// TIA Portal project "andres-c程序测试" (V14)

(* hardware
DEVICE "S7-1200 station_1"  S7-1200 Station
   slot 0: "Rack_0"  Rack  V1.0
   slot 1: "PLC_14工位_1200"  CPU 1215C DC/DC/DC  6ES7 215-1AG40-0XB0  V4.2
DEVICE "ET 200SP station_2"  ET 200SP-Station
   slot 0: "机架_0"  6ES5 710-8MAx1
   slot 0: "IO device_2"  IM155-6 PN ST  6ES7 155-6AU00-0BN0  V3.3
   slot 1: "DI 16x24VDC ST_1"  DI 16x24VDC ST  6ES7 131-6BH00-0BA0  V1.1
      slot 1: "DI 16x24VDC ST_1"  DI 16x24VDC ST
   slot 2: "DI 16x24VDC ST_2"  DI 16x24VDC ST  6ES7 131-6BH00-0BA0  V1.1
      slot 1: "DI 16x24VDC ST_2"  DI 16x24VDC ST
   slot 3: "DI 16x24VDC ST_3"  DI 16x24VDC ST  6ES7 131-6BH00-0BA0  V1.1
      slot 1: "DI 16x24VDC ST_3"  DI 16x24VDC ST
   slot 4: "DI 16x24VDC ST_4"  DI 16x24VDC ST  6ES7 131-6BH00-0BA0  V1.1
      slot 1: "DI 16x24VDC ST_4"  DI 16x24VDC ST
   slot 5: "DI 16x24VDC ST_5"  DI 16x24VDC ST  6ES7 131-6BH00-0BA0  V1.1
      slot 1: "DI 16x24VDC ST_5"  DI 16x24VDC ST
   slot 6: "DI 16x24VDC ST_6"  DI 16x24VDC ST  6ES7 131-6BH00-0BA0  V1.1
      slot 1: "DI 16x24VDC ST_6"  DI 16x24VDC ST
   slot 7: "DI 16x24VDC ST_7"  DI 16x24VDC ST  6ES7 131-6BH00-0BA0  V1.1
      slot 1: "DI 16x24VDC ST_7"  DI 16x24VDC ST
   slot 8: "DI 16x24VDC ST_8"  DI 16x24VDC ST  6ES7 131-6BH00-0BA0  V1.1
      slot 1: "DI 16x24VDC ST_8"  DI 16x24VDC ST
   slot 9: "DI 16x24VDC ST_9"  DI 16x24VDC ST  6ES7 131-6BH00-0BA0  V1.1
      slot 1: "DI 16x24VDC ST_9"  DI 16x24VDC ST
   slot 10: "DI 16x24VDC ST_10"  DI 16x24VDC ST  6ES7 131-6BH00-0BA0  V1.1
      slot 1: "DI 16x24VDC ST_10"  DI 16x24VDC ST
   slot 11: "DQ 16x24VDC/0.5A ST_2"  DQ 16x24VDC/0.5A ST  6ES7 132-6BH00-0BA0  V1.1
      slot 1: "DQ 16x24VDC/0.5A ST_2"  DQ 16x24VDC/0.5A ST
   slot 12: "DQ 16x24VDC/0.5A ST_3"  DQ 16x24VDC/0.5A ST  6ES7 132-6BH00-0BA0  V1.1
      slot 1: "DQ 16x24VDC/0.5A ST_3"  DQ 16x24VDC/0.5A ST
   slot 13: "DQ 16x24VDC/0.5A ST_4"  DQ 16x24VDC/0.5A ST  6ES7 132-6BH00-0BA0  V1.1
      slot 1: "DQ 16x24VDC/0.5A ST_4"  DQ 16x24VDC/0.5A ST
   slot 14: "DQ 16x24VDC/0.5A ST_5"  DQ 16x24VDC/0.5A ST  6ES7 132-6BH00-0BA0  V1.1
      slot 1: "DQ 16x24VDC/0.5A ST_5"  DQ 16x24VDC/0.5A ST
   slot 15: "DQ 16x24VDC/0.5A ST_6"  DQ 16x24VDC/0.5A ST  6ES7 132-6BH00-0BA0  V1.1
      slot 1: "DQ 16x24VDC/0.5A ST_6"  DQ 16x24VDC/0.5A ST
   slot 16: "DQ 16x24VDC/0.5A ST_1"  DQ 16x24VDC/0.5A ST  6ES7 132-6BH00-0BA0  V1.1
      slot 1: "DQ 16x24VDC/0.5A ST_1"  DQ 16x24VDC/0.5A ST
   slot 17: "DQ 16x24VDC/0.5A ST_7"  DQ 16x24VDC/0.5A ST  6ES7 132-6BH00-0BA0  V1.1
      slot 1: "DQ 16x24VDC/0.5A ST_7"  DQ 16x24VDC/0.5A ST
   slot 18: "DQ 16x24VDC/0.5A ST_8"  DQ 16x24VDC/0.5A ST  6ES7 132-6BH00-0BA0  V1.1
      slot 1: "DQ 16x24VDC/0.5A ST_8"  DQ 16x24VDC/0.5A ST
   slot 19: "AQ 4xU/I ST_1"  AQ 4xU/I ST  6ES7 135-6HD00-0BA1  V1.1
      slot 1: "AQ 4xU/I ST_1"  AQ 4xU/I ST
   slot 20: "服务器模块_1"  服务器模块  6ES7 193-6PA00-0AA0  V1.0
      slot 1: "服务器模块_1"  服务器模块
   slot 127: "PROFINET 总线适配器 CU"  PROFINET Interface  6ES7 193-6AR00-0AA0  V0.0
      slot 1: "Port_1"  6ES7 193-6AR00-0AA0  V0.0
      slot 2: "Port_2"  6ES7 193-6AR00-0AA0  V0.0
*)

// ===== PLC "PLC_14工位_1200"  CPU 1215C DC/DC/DC =====

VAR_GLOBAL   // PLC tag table "默认变量表"
   "Tag_1" AT %M0.0 : Bool;
   "初次扫描OB100保持位" AT %M0.1 : Bool;
   "给上位机发送数据" AT %M0.2 : Bool;
   "Tag_4" AT %M0.3 : Bool;
   "1#手动Z轴下降" AT %M10.0 : Bool;
   "14S01" AT %I0.0 : Bool;   // 1#机械手X轴定位接近1
   "14S02" AT %I0.1 : Bool;   // 1#机械手X轴定位接近2
   "14S03" AT %I0.2 : Bool;   // 1#机械手X轴减速接近
   "14L01" AT %I0.3 : Bool;   // 1#机械手X轴机械限位
   "14S04" AT %I0.4 : Bool;   // 1#机械手z轴原点光电
   "14L02" AT %I0.5 : Bool;   // 1#机械手z轴机械限位
   "14S05" AT %I0.6 : Bool;   // 1#机械手W轴原点光电
   "14L03" AT %I0.7 : Bool;   // 1#机械手W轴机械限位
   "14S06" AT %I1.0 : Bool;   // 1#机械手抓取光电
   "14S07" AT %I1.1 : Bool;   // 1#W轴上砖位
   "14S08" AT %I1.2 : Bool;   // 1#W轴停止位
   "14S09" AT %I1.3 : Bool;   // 1#机械手抓取极限光电
   "14P02" AT %I1.4 : Bool;   // 1#机械手负压检测1
   "14P03" AT %I1.5 : Bool;   // 1#机械手负压检测2
   "14P04" AT %I1.6 : Bool;   // 1#机械手负压检测3
   "14P05" AT %I1.7 : Bool;   // 1#机械手负压检测4
   "14S10" AT %I2.0 : Bool;   // 2#机械手X轴定位接近1
   "14S11" AT %I2.1 : Bool;   // 2#机械手X轴定位接近2
   "14S12" AT %I2.2 : Bool;   // 2#机械手X轴减速接近
   "14L04" AT %I2.3 : Bool;   // 2#机械手X轴机械限位
   "14S13" AT %I2.4 : Bool;   // 2#机械手z轴原点光电
   "14L05" AT %I2.5 : Bool;   // 2#机械手z轴机械限位
   "14S14" AT %I2.6 : Bool;   // 2#机械手W轴原点光电
   "14L06" AT %I2.7 : Bool;   // 2#机械手W轴机械限位
   "14S15" AT %I3.0 : Bool;   // 2#机械手抓取光电
   "14S16" AT %I3.1 : Bool;   // 2#机械手W上砖待命位
   "14S17" AT %I3.2 : Bool;   // 2#机械手W轴停止位
   "14S18" AT %I3.3 : Bool;   // 2#机械手抓取极限光电
   "14P06" AT %I3.4 : Bool;   // 2#机械手负压检测1
   "14P07" AT %I3.5 : Bool;   // 2#机械手负压检测2
   "14P08" AT %I3.6 : Bool;   // 2#机械手负压检测3
   "14P09" AT %I3.7 : Bool;   // 2#机械手负压检测4
   "14S19" AT %I4.0 : Bool;   // 3#机械手X轴定位接近1
   "14S20" AT %I4.1 : Bool;   // 3#机械手X轴定位接近2
   "14S21" AT %I4.2 : Bool;   // 3#机械手X轴减速接近
   "14L07" AT %I4.3 : Bool;   // 3#机械手X轴机械限位
   "14S22" AT %I4.4 : Bool;   // 3#机械手z轴原点光电
   "141L08" AT %I4.5 : Bool;   // 3#机械手z轴机械限位
   "14S23" AT %I4.6 : Bool;   // 3#机械手W轴原点光电
   "14L09" AT %I4.7 : Bool;   // 3#机械手W轴机械限位
   "14S24" AT %I5.0 : Bool;   // 3#机械手抓取光电
   "14S25" AT %I5.1 : Bool;   // 3#机械手W上砖待命位
   "14S26" AT %I5.2 : Bool;   // 3#机械手W停止位
   "14S27" AT %I5.3 : Bool;   // 3#机械手抓取极限光电
   "14P10" AT %I5.4 : Bool;   // 3#机械手负压检测1
   "14P11" AT %I5.5 : Bool;   // 3#机械手负压检测2
   "14P12" AT %I5.6 : Bool;   // 3#机械手负压检测3
   "14P13" AT %I5.7 : Bool;   // 3#机械手负压检测4
   "14S28" AT %I6.0 : Bool;   // 4#机械手X轴定位接近1
   "14S29" AT %I6.1 : Bool;   // 4#机械手X轴定位接近2
   "14S30" AT %I6.2 : Bool;   // 4#机械手X轴减速接近
   "14L10" AT %I6.3 : Bool;   // 4#机械手X轴机械限位
   "14S31" AT %I6.4 : Bool;   // 4#机械手z轴原点光电
   "14L11" AT %I6.5 : Bool;   // 4#机械手z轴机械限位
   "14S32" AT %I6.6 : Bool;   // 4#机械手W轴原点光电
   "14L12" AT %I6.7 : Bool;   // 4#机械手W轴机械限位
   "14S33" AT %I7.0 : Bool;   // 4#机械手抓取光电
   "14S34" AT %I7.1 : Bool;   // 4#机械手上砖待命位
   "14S35" AT %I7.2 : Bool;   // 4#机械手W停止位
   "14S36" AT %I7.3 : Bool;   // 4#机械手抓取极限光电
   "14P14" AT %I7.4 : Bool;   // 4#机械手负压检测1
   "14P15" AT %I7.5 : Bool;   // 4#机械手负压检测2
   "14P16" AT %I7.6 : Bool;   // 4#机械手负压检测3
   "14P17" AT %I7.7 : Bool;   // 4#机械手负压检测4
   "14SB1" AT %I8.0 : Bool;   // 一级品分级按钮
   "14SB2" AT %I8.1 : Bool;   // 二级品分级按钮
   "14SB3" AT %I8.2 : Bool;   // 换花色旋钮
   "14S37" AT %I8.3 : Bool;   // 队列光电1
   "14S38" AT %I8.4 : Bool;   // 队列光电2
   "14P01" AT %I8.5 : Bool;   // 设备压力检测
   "14S39" AT %I8.6 : Bool;   // 1#3#库位安全光电
   "14S40" AT %I8.7 : Bool;   // 2#4#库位安全光电
   "14S41" AT %I9.0 : Bool;   // 7#9#库位安全光电
   "14S42" AT %I9.1 : Bool;   // 8#10#库位安全光电
   "14S43" AT %I9.2 : Bool;   // 1#库位栈板检测光电
   "14S44" AT %I9.3 : Bool;   // 2#库位栈板检测光电
   "14S45" AT %I9.4 : Bool;   // 1#库位安全检测光电
   "14S46" AT %I9.5 : Bool;   // 2#库位安全检测光电
   "14SB7" AT %I9.6 : Bool;   // 1#库位按钮
   "14SB8" AT %I9.7 : Bool;   // 2#库位按钮
   "14S47" AT %I10.0 : Bool;   // 3#库位栈板检测光电
   "14S48" AT %I10.1 : Bool;   // 4#库位栈板检测光电
   "14S49" AT %I10.2 : Bool;   // 3#库位安全检测光电
   "14S50" AT %I10.3 : Bool;   // 4#库位安全检测光电
   "14SB9" AT %I10.4 : Bool;   // 3#库位按钮
   "14SB10" AT %I10.5 : Bool;   // 4#库位按钮
   "14S51" AT %I10.6 : Bool;   // 5#库位栈板检测光电
   "14S52" AT %I10.7 : Bool;   // 6#库位栈板检测光电
   "14S53" AT %I11.0 : Bool;   // 5#库位安全检测光电
   "14S54" AT %I11.1 : Bool;   // 6#库位安全检测光电
   "14SB11" AT %I11.2 : Bool;   // 5#库位按钮
   "14SB12" AT %I11.3 : Bool;   // 6#库位按钮
   "14S55" AT %I11.4 : Bool;   // 7#库位栈板检测光电
   "14S56" AT %I11.5 : Bool;   // 8#库位栈板检测光电
   "14S57" AT %I11.6 : Bool;   // 7#库位安全检测光电
   "14S58" AT %I11.7 : Bool;   // 8#库位安全检测光电
   "14SB13" AT %I12.0 : Bool;   // 7#库位按钮
   "14SB14" AT %I12.1 : Bool;   // 8#库位按钮
   "14SB25" AT %I12.2 : Bool;   // 输送线启动按钮
   "14S59" AT %I12.3 : Bool;   // 输送线对中光电
   "14SB26" AT %I12.4 : Bool;   // 输送线停止按钮
   "11S73" AT %I12.5 : Bool;   // 队列光电3
   "11S74" AT %I12.6 : Bool;   // 队列光电4
   "输送线变频器报警" AT %I12.7 : Bool;   // 输送线变频器报警
   "14M01MB" AT %I13.0 : Bool;   // M01变频器报警
   "14M02MB" AT %I13.1 : Bool;   // M02变频器报警
   "14M04MB" AT %I13.2 : Bool;   // M04变频器报警
   "14M05MB" AT %I13.3 : Bool;   // M05变频器报警
   "14M07MB" AT %I13.4 : Bool;   // M07变频器报警
   "14M08MB" AT %I13.5 : Bool;   // M08变频器报警
   "14M10MB" AT %I13.6 : Bool;   // M10变频器报警
   "14M11MB" AT %I13.7 : Bool;   // M11变频器报警
   "14SB15" AT %I14.0 : Bool;   // 主控柜启动按钮
   "14SB16" AT %I14.1 : Bool;   // 主控柜停止按钮
   "14SB17" AT %I14.2 : Bool;   // 主控柜复位按钮
   "14SB18" AT %I14.3 : Bool;   // 主控柜消音按钮
   "14EM" AT %M65.0 : Bool;   // 主控柜急停按钮
   "14SA01" AT %I14.5 : Bool;   // 主控柜启动激活
   "14SA02" AT %I14.6 : Bool;   // 主控柜停止激活
   "14SA03" AT %I14.7 : Bool;   // 主控柜复位激活
   "14M13MB" AT %I15.0 : Bool;   // M13变频器报警
   "14M14MB" AT %I15.1 : Bool;   // M14变频器报警
   "14M03MB" AT %I15.2 : Bool;   // M03伺服控制器报警
   "14M06MB" AT %I15.3 : Bool;   // M06伺服控制器报警
   "14M09MB" AT %I15.4 : Bool;   // M09伺服控制器报警
   "14M12MB" AT %I15.5 : Bool;   // M12伺服控制器报警
   "14M15MB" AT %I15.6 : Bool;   // M15伺服控制器报警
   "备用" AT %I15.7 : Bool;
   "视觉拍照光电" AT %I16.0 : Bool;
   "备用(2)" AT %I16.1 : Bool;
   "备用(3)" AT %I16.2 : Bool;
   "14S60" AT %I16.3 : Bool;   // 9#库位栈板检测
   "14S61" AT %I16.4 : Bool;   // 10#库位栈板检测
   "14S62" AT %I16.5 : Bool;   // 9#库位安全检测
   "14S63" AT %I16.6 : Bool;   // 10#库位安全检测
   "SB21" AT %I16.7 : Bool;   // 9#库位启动按钮
   "SB22" AT %I17.0 : Bool;   // 10#库位启动按钮
   "备用(4)" AT %I17.1 : Bool;
   "备用(5)" AT %I17.2 : Bool;
   "备用(6)" AT %I17.3 : Bool;
   "备用(7)" AT %I17.4 : Bool;
   "14EM02" AT %I17.5 : Bool;   // 输送线入口急停1
   "14EM03" AT %I17.6 : Bool;   // 输送线入口急停2
   "14EM04" AT %I17.7 : Bool;   // 输送线出口急停
   "KA1" AT %Q0.0 : Bool;   // 灯塔-红色
   "KA2" AT %Q0.1 : Bool;   // 灯塔-绿色
   "KA3" AT %Q0.2 : Bool;   // 灯塔-黄色
   "KA4" AT %Q0.3 : Bool;   // 灯塔-蓝色
   "KA5" AT %Q0.4 : Bool;   // 灯塔-蜂鸣器
   "%Q0.5" AT %Q0.5 : Bool;   // 主控柜开始按钮指示灯
   "%Q0.6" AT %Q0.6 : Bool;   // 主控柜停止按钮指示灯
   "%Q0.7" AT %Q0.7 : Bool;   // 主控柜复位按钮指示灯
   "%Q1.0" AT %Q1.0 : Bool;   // 对中气缸电磁阀
   "%Q1.1" AT %Q1.1 : Bool;   // 主控柜运行指示灯
   "%Q1.2" AT %Q1.2 : Bool;   // 主控柜停止指示灯
   "%Q1.3" AT %Q1.3 : Bool;   // 主控柜复位指示灯
   "%Q1.4" AT %Q1.4 : Bool;   // 输送线电机
   "%Q1.5" AT %Q1.5 : Bool;   // 输送线喷码机
   "%Q1.6" AT %Q1.6 : Bool;   // 输送线启动指示灯
   "%Q1.7" AT %Q1.7 : Bool;   // 输送线停止指示灯
   "14M01LI1" AT %Q2.0 : Bool;   // 1#机械手X轴正转
   "14M01LI2" AT %Q2.1 : Bool;   // 1#机械手X轴反转
   "14M01LI3" AT %Q2.2 : Bool;   // 1#机械手X轴低速
   "14M02FWD" AT %Q2.3 : Bool;   // 1#机械手Z轴正转
   "14M02REV" AT %Q2.4 : Bool;   // 1#机械手Z轴反转
   "14M02X1" AT %Q2.5 : Bool;   // 1#Z轴速度端子1
   "14M02X2" AT %Q2.6 : Bool;   // 1#Z轴速度端子2
   "14M02X3" AT %Q2.7 : Bool;   // 1#Z轴速度端子3
   "14KAV02" AT %Q3.0 : Bool;   // 1#机械手吸真空阀关
   "14KAV03" AT %Q3.1 : Bool;   // 1#机械手吸真空阀开
   "14M04LI1" AT %Q3.2 : Bool;   // 2#机械手X轴正转
   "14M04LI2" AT %Q3.3 : Bool;   // 2#机械手X轴反转
   "14M04LI3" AT %Q3.4 : Bool;   // 2#机械手X轴低速
   "14M05FWD" AT %Q3.5 : Bool;   // 2#机械手Z轴正转
   "14M05REV" AT %Q3.6 : Bool;   // 2#机械手Z轴反转
   "14M05X1" AT %Q3.7 : Bool;   // 2#Z轴速度端子1
   "14M05X2" AT %Q4.0 : Bool;   // 2#Z轴速度端子2
   "14M05X3" AT %Q4.1 : Bool;   // 2#Z轴速度端子3
   "14KAV05" AT %Q4.2 : Bool;   // 2#机械手吸真空阀关
   "14KAV06" AT %Q4.3 : Bool;   // 2#机械手吸真空阀开
   "14M07LI1" AT %Q4.4 : Bool;   // 3#机械手X轴正转
   "14M07LI2" AT %Q4.5 : Bool;   // 3#机械手X轴反转
   "14M07LI3" AT %Q4.6 : Bool;   // 3#机械手X轴低速
   "14M08FWD" AT %Q4.7 : Bool;   // 3#机械手Z轴正转
   "14M08REV" AT %Q5.0 : Bool;   // 3#机械手Z轴反转
   "14M08X1" AT %Q5.1 : Bool;   // 3#Z轴速度端子1
   "14M08X2" AT %Q5.2 : Bool;   // 3#Z轴速度端子2
   "14M08X3" AT %Q5.3 : Bool;   // 3#Z轴速度端子3
   "14KAV07" AT %Q5.4 : Bool;   // 3#机械手吸真空阀关
   "14KAV08" AT %Q5.5 : Bool;   // 3#机械手吸真空阀开
   "14M10LI1" AT %Q5.6 : Bool;   // 4#机械手X轴正转
   "14M10LI2" AT %Q5.7 : Bool;   // 4#机械手X轴反转
   "14M10LI3" AT %Q6.0 : Bool;   // 4#机械手X轴低速
   "14M11FWD" AT %Q6.1 : Bool;   // 4#机械手Z轴正转
   "14M11REV" AT %Q6.2 : Bool;   // 4#机械手Z轴反转
   "14M11X1" AT %Q6.3 : Bool;   // 4#Z轴速度端子1
   "14M11X2" AT %Q6.4 : Bool;   // 4#Z轴速度端子2
   "14M11X3" AT %Q6.5 : Bool;   // 4#Z轴速度端子3
   "14KAV09" AT %Q6.6 : Bool;   // 4#机械手吸真空阀关
   "14KAV10" AT %Q6.7 : Bool;   // 4#机械手吸真空阀开
   "14KAM01B" AT %Q7.0 : Bool;   // 1#机械手X轴抱闸
   "14KAM02B" AT %Q7.1 : Bool;   // 1#机械手Z轴抱闸
   "14KAM04B" AT %Q7.2 : Bool;   // 2#机械手X轴抱闸
   "14KAM05B" AT %Q7.3 : Bool;   // 2#机械手Z轴抱闸
   "14KAM07B" AT %Q7.4 : Bool;   // 3#机械手X轴抱闸
   "14KAM08B" AT %Q7.5 : Bool;   // 3#机械手Z轴抱闸
   "14KAM10B" AT %Q7.6 : Bool;   // 4#机械手X轴抱闸
   "14KAM11B" AT %Q7.7 : Bool;   // 4#机械手Z轴抱闸
   "11连锁" AT %Q8.0 : Bool;   // 11连锁
   "14HL2" AT %Q8.1 : Bool;   // 一级分级指示灯
   "14HL3" AT %Q8.2 : Bool;   // 二级分级指示灯
   "14HL4" AT %Q8.3 : Bool;   // 换花色指示灯
   "14HL5" AT %Q8.4 : Bool;   // 1#机械手库位按钮指示灯
   "14HL6" AT %Q8.5 : Bool;   // 2#机械手库位按钮指示灯
   "14HL7" AT %Q8.6 : Bool;   // 3#机械手库位按钮指示灯
   "14HL8" AT %Q8.7 : Bool;   // 4#机械手库位按钮指示灯
   "14HL9" AT %Q9.0 : Bool;   // 5#机械手库位按钮指示灯
   "14HL10" AT %Q9.1 : Bool;   // 6#机械手库位按钮指示灯
   "14HL11" AT %Q9.2 : Bool;   // 7#机械手库位按钮指示灯
   "14HL12" AT %Q9.3 : Bool;   // 8#机械手库位按钮指示灯
   "14HL13" AT %Q9.4 : Bool;   // 1#库位黄色灯
   "14HL14" AT %Q9.5 : Bool;   // 1#库位红色灯
   "14HL15" AT %Q9.6 : Bool;   // 2#库位黄色灯
   "14HL16" AT %Q9.7 : Bool;   // 2#库位红色灯
   "14HL17" AT %Q10.0 : Bool;   // 3#库位黄色灯
   "14HL18" AT %Q10.1 : Bool;   // 3#库位红色灯
   "14HL19" AT %Q10.2 : Bool;   // 4#库位黄色灯
   "14HL20" AT %Q10.3 : Bool;   // 4#库位红色灯
   "14HL21" AT %Q10.4 : Bool;   // 5#库位黄色灯
   "14HL22" AT %Q10.5 : Bool;   // 5#库位红色灯
   "14HL23" AT %Q10.6 : Bool;   // 6#库位黄色灯
   "14HL24" AT %Q10.7 : Bool;   // 6#库位红色灯
   "14HL25" AT %Q11.0 : Bool;   // 7#库位黄色灯
   "14HL26" AT %Q11.1 : Bool;   // 7#库位红色灯
   "14HL27" AT %Q11.2 : Bool;   // 8#库位黄色灯
   "14HL28" AT %Q11.3 : Bool;   // 8#库位红色灯
   "Q11.4" AT %Q11.4 : Bool;   // 1#伺服电机启动
   "Q11.5" AT %Q11.5 : Bool;   // 2#伺服电机启动
   "Q11.6" AT %Q11.6 : Bool;   // 3#伺服电机启动
   "Q11.7" AT %Q11.7 : Bool;   // 4#伺服电机启动
   "Q12.0" AT %Q12.0 : Bool;   // 5#伺服电机启动
   "14M13LI1" AT %Q12.1 : Bool;   // 5#机械手X轴正转
   "14M13LI2" AT %Q12.2 : Bool;   // 5#机械手X轴反转
   "14M13LI3" AT %Q12.3 : Bool;   // 5#机械手X轴低速
   "14M14FWD" AT %Q12.4 : Bool;   // 5#机械手Z轴正转
   "14M14REV" AT %Q12.5 : Bool;   // 5#机械手Z轴反转
   "14M14X1" AT %Q12.6 : Bool;   // 5#Z轴速度端子1
   "14M14X2" AT %Q12.7 : Bool;   // 5#Z轴速度端子2
   "14M14X3" AT %Q13.0 : Bool;   // 5#Z轴速度端子3
   "14KAV11" AT %Q13.1 : Bool;   // 5#机械手吸真空阀关
   "14KAV12" AT %Q13.2 : Bool;   // 5#机械手吸真空阀开
   "14HL38" AT %Q13.3 : Bool;   // 9#库位按钮指示灯
   "14HL39" AT %Q13.4 : Bool;   // 10#库位按钮指示灯
   "14HL40" AT %Q13.5 : Bool;   // 9#库位绿灯
   "14HL41" AT %Q13.6 : Bool;   // 9#库位红灯
   "14HL42" AT %Q13.7 : Bool;   // 10#库位绿灯
   "1#机械手Z轴速度写入值" AT %QW256 : Word;
   "2#机械手Z轴速度写入值" AT %QW258 : Word;
   "3#机械手Z轴速度写入值" AT %QW260 : Word;
   "4#机械手Z轴速度写入值" AT %QW262 : Word;
   "1#手动破真空阀开" AT %M11.0 : Bool;
   "2#手动破真空阀开" AT %M13.0 : Bool;
   "Tag_42" AT %M6.0 : Bool;
   "4#Z轴编码器清零" AT %M7.0 : Bool;
   "System_Byte" AT %MB1 : Byte;
   "FirstScan" AT %M1.0 : Bool;
   "DiagStatusUpdate" AT %M1.1 : Bool;
   "AlwaysTRUE" AT %M1.2 : Bool;
   "AlwaysFALSE" AT %M1.3 : Bool;
   "2#Z轴编码器清零" AT %M7.1 : Bool;
   "3#Z轴编码器清零" AT %M7.2 : Bool;
   "1#Z轴编码器清零" AT %M7.3 : Bool;
   "3#手动X轴1库移动" AT %M14.3 : Bool;
   "1#机械手系统运行标志" AT %M9.0 : Bool;
   "3#机械手系统运行标志" AT %M9.2 : Bool;
   "2#机械手系统运行标志" AT %M9.1 : Bool;
   "4#机械手系统运行标志" AT %M9.3 : Bool;
   "1#手动Z轴上升" AT %M10.1 : Bool;
   "1#手动X轴2库移动" AT %M10.2 : Bool;
   "1#手动X轴1库移动" AT %M10.3 : Bool;
   "1#手动W轴前移" AT %M10.4 : Bool;
   "1#手动W轴回原位" AT %M10.5 : Bool;
   "1#手动吸盘电磁阀打开" AT %M10.6 : Bool;
   "1#手动吸盘电磁阀关闭" AT %M10.7 : Bool;
   "2#手动Z轴下降" AT %M12.0 : Bool;
   "2#手动Z轴上升" AT %M12.1 : Bool;
   "2#手动X轴2库移动" AT %M12.2 : Bool;
   "2#手动X轴1库移动" AT %M12.3 : Bool;
   "2#手动W轴前移" AT %M12.4 : Bool;
   "2#手动W轴回原位" AT %M12.5 : Bool;
   "2#手动吸盘电磁阀打开" AT %M12.6 : Bool;
   "2#手动吸盘电磁阀关闭" AT %M12.7 : Bool;
   "3#手动Z轴下降" AT %M14.0 : Bool;
   "3#手动Z轴上升" AT %M14.1 : Bool;
   "3#手动X轴2库移动" AT %M14.2 : Bool;
   "3#手动W轴前移" AT %M14.4 : Bool;
   "3#手动W轴回原位" AT %M14.5 : Bool;
   "3#手动吸盘电磁阀打开" AT %M14.6 : Bool;
   "3#手动吸盘电磁阀关闭" AT %M14.7 : Bool;
   "3#手动破真空阀开" AT %M15.0 : Bool;
   "4#手动Z轴下降" AT %M16.0 : Bool;
   "4#手动Z轴上升" AT %M16.1 : Bool;
   "4#手动X轴2库移动" AT %M16.2 : Bool;
   "4#手动X轴1库移动" AT %M16.3 : Bool;
   "4#手动W轴前移" AT %M16.4 : Bool;
   "4#手动W轴回原位" AT %M16.5 : Bool;
   "4#手动吸盘电磁阀打开" AT %M16.6 : Bool;
   "4#手动吸盘电磁阀关闭" AT %M16.7 : Bool;
   "6#手动Z轴下降" AT %M17.0 : Bool;
   "1#手动Z轴撞击限位下" AT %M11.2 : Bool;
   "1#手动Z轴撞击限位上" AT %M11.3 : Bool;
   "1#手动X轴A库撞击限位" AT %M11.4 : Bool;
   "1#手动X轴B库撞击限位" AT %M11.5 : Bool;
   "1#手动W轴前撞击限位" AT %M11.6 : Bool;
   "1#手动W轴后撞击限位" AT %M11.7 : Bool;
   "Tag_7" AT %M13.1 : Bool;
   "Tag_19" AT %M13.2 : Bool;
   "Tag_62" AT %M13.3 : Bool;
   "Tag_63" AT %M13.4 : Bool;
   "Tag_66" AT %M13.5 : Bool;
   "Tag_68" AT %M13.6 : Bool;
   "Tag_69" AT %M15.1 : Bool;
   "Tag_72" AT %M15.2 : Bool;
   "Tag_73" AT %M15.3 : Bool;
   "Tag_74" AT %M15.4 : Bool;
   "Tag_75" AT %M15.5 : Bool;
   "Tag_76" AT %M15.6 : Bool;
   "6#手动Z轴上升" AT %M17.1 : Bool;
   "6#手动X轴2库移动" AT %M17.2 : Bool;
   "6#手动X轴1库移动" AT %M17.3 : Bool;
   "6#手动W轴前移" AT %M17.4 : Bool;
   "6#手动W轴回原位" AT %M17.5 : Bool;
   "6#手动吸盘电磁阀打开" AT %M17.6 : Bool;
   "1#机械手系统复位标志" AT %M9.4 : Bool;
   "2#机械手系统复位标志" AT %M9.5 : Bool;
   "3#机械手系统复位标志" AT %M9.6 : Bool;
   "4#机械手系统复位标志" AT %M9.7 : Bool;
   "Clock_Byte" AT %MB3 : Byte;
   "Clock_10Hz" AT %M3.0 : Bool;
   "Clock_5Hz" AT %M3.1 : Bool;
   "Clock_2.5Hz" AT %M3.2 : Bool;
   "Clock_2Hz" AT %M3.3 : Bool;
   "Clock_1.25Hz" AT %M3.4 : Bool;
   "Clock_1Hz" AT %M3.5 : Bool;
   "Clock_0.625Hz" AT %M3.6 : Bool;
   "Clock_0.5Hz" AT %M3.7 : Bool;
   "1#机械手系统急停限位标志" AT %M60.0 : Bool;
   "2#机械手系统急停限位标志" AT %M60.1 : Bool;
   "3#机械手系统急停限位标志" AT %M60.2 : Bool;
   "4#机械手系统急停限位标志" AT %M60.3 : Bool;
   "1#1压力开关报警" AT %M61.0 : Bool;
   "1#2压力开关报警" AT %M61.1 : Bool;
   "1#3压力开关报警" AT %M61.2 : Bool;
   "1#4压力开关报警" AT %M61.3 : Bool;
   "2#1压力开关报警" AT %M61.4 : Bool;
   "2#2压力开关报警" AT %M61.5 : Bool;
   "2#3压力开关报警" AT %M61.6 : Bool;
   "2#4压力开关报警" AT %M61.7 : Bool;
   "3#1压力开关报警" AT %M62.0 : Bool;
   "3#2压力开关报警" AT %M62.1 : Bool;
   "3#3压力开关报警" AT %M62.2 : Bool;
   "3#4压力开关报警" AT %M62.3 : Bool;
   "4#1压力开关报警" AT %M62.4 : Bool;
   "4#2压力开关报警" AT %M62.5 : Bool;
   "4#3压力开关报警" AT %M62.6 : Bool;
   "4#4压力开关报警" AT %M62.7 : Bool;
   "1#机械手单独复位标志位" AT %M63.0 : Bool;
   "2#机械手单独复位标志位" AT %M63.1 : Bool;
   "3#机械手单独复位标志位" AT %M63.2 : Bool;
   "4#机械手单独复位标志位" AT %M63.3 : Bool;
   "启动按钮激活标志位" AT %M64.0 : Bool;
   "停止按钮激活标志位" AT %M64.1 : Bool;
   "复位按钮激活标志位" AT %M64.2 : Bool;
   "复位按钮激活标志位复位" AT %M64.3 : Bool;
   "砖到分级位指示" AT %M66.0 : Bool;
   "Tag_100" AT %M66.1 : Bool;
   "1#库安全光电报警" AT %M68.0 : Bool;
   "2#库安全光电报警" AT %M68.1 : Bool;
   "3#库安全光电报警" AT %M68.2 : Bool;
   "4#库安全光电报警" AT %M68.3 : Bool;
   "6#库安全光电报警" AT %M68.5 : Bool;
   "5#库安全光电报警" AT %M68.4 : Bool;
   "7#库安全光电报警" AT %M68.6 : Bool;
   "8#库安全光电报警" AT %M68.7 : Bool;
   "1#找待命位速度" AT %M69.0 : Bool;
   "蜂鸣器报警标志位1" AT %M65.1 : Bool;
   "蜂鸣器报警标志位2" AT %M65.2 : Bool;
   "蜂鸣器报警标志位3" AT %M65.3 : Bool;
   "蜂鸣器报警标志位4" AT %M65.4 : Bool;
   "蜂鸣器报警标志位5" AT %M65.5 : Bool;
   "蜂鸣器报警标志位6" AT %M65.6 : Bool;
   "2#找待命位速度" AT %M69.1 : Bool;
   "3#找待命位速度" AT %M69.2 : Bool;
   "4#找待命位速度" AT %M69.3 : Bool;
   "14EM01" AT %I14.4 : Bool;   // 主控柜急停按钮
   "蜂鸣器报警标志位7" AT %M65.7 : Bool;
   "输送线停止" AT %M69.4 : Bool;
   "Tag_116" AT %M70.0 : Bool;
   "输送线启动标志位" AT %M70.1 : Bool;
   "漏砖喷码标志位" AT %M70.2 : Bool;
   "Tag_125" AT %M600.0 : Bool;
   "Tag_126" AT %M600.1 : Bool;
   "Tag_127" AT %M600.2 : Bool;
   "Tag_128" AT %M600.3 : Bool;
   "1#抓取编码值" AT %MD610 : DWord;
   "1#抓取输送线编码值" AT %MD614 : DWord;
   "2#抓取编码值" AT %MD618 : DWord;
   "2#抓取输送线编码值" AT %MD622 : DWord;
   "3#抓取编码值" AT %MD626 : DWord;
   "3#抓取输送线编码值" AT %MD630 : DWord;
   "4#抓取编码值" AT %MD634 : DWord;
   "4#抓取输送线编码值" AT %MD638 : DWord;
   "高速计数器1" AT %ID1000 : DWord;
   "高速计数器2" AT %ID1004 : DWord;
   "高速计数器3" AT %ID1008 : DWord;
   "高速计数器4" AT %ID1012 : DWord;
   "高速计数器5" AT %ID1016 : DWord;
   "高速计数器6" AT %ID1020 : DWord;
   "Tag_11" AT %MD24 : DInt;
   "Tag_13" AT %MD20 : DInt;
   "Tag_14" AT %MD28 : Real;
   "Tag_129" AT %MD32 : DWord;
   "输送线编码值清零" AT %M7.4 : Bool;
   "Tag_2" AT %MD36 : Real;
   "Tag_5" AT %M6.1 : Bool;
   "Tag_6" AT %M6.2 : Bool;
   "Tag_9" AT %M6.3 : Bool;
   "Tag_10" AT %M700.0 : Bool;
   "Tag_15" AT %MD702 : DInt;
   "Tag_16" AT %M700.1 : Bool;
   "Tag_17" AT %MD706 : DInt;
   "14S72" AT %I18.0 : Bool;   // 5#机械手X轴定位接近1
   "14S73" AT %I18.1 : Bool;   // 5#机械手X轴定位接近2
   "14S74" AT %I18.2 : Bool;   // 5#机械手X轴减速接近
   "14L16" AT %I18.3 : Bool;   // 5#机械手X轴机械限位
   "14S75" AT %I18.4 : Bool;   // 5#机械手z轴原点光电
   "14L17" AT %I18.5 : Bool;   // 5#机械手z轴机械限位
   "14L76" AT %I18.6 : Bool;   // 5#机械手W轴原点光电
   "14L18" AT %I18.7 : Bool;   // 5#机械手W轴机械限位
   "14S77" AT %I19.0 : Bool;   // 5#机械手抓取光电
   "14S78" AT %I19.1 : Bool;   // 5#机械手W上砖待命位
   "14S79" AT %I19.2 : Bool;   // 5#机械手W轴停止位
   "14S80" AT %I19.3 : Bool;   // 5#机械手抓取极限光电
   "14P22" AT %I19.4 : Bool;   // 5#机械手负压检测1
   "14P23" AT %I19.5 : Bool;   // 5#机械手负压检测2
   "14P24" AT %I19.6 : Bool;   // 5#机械手负压检测3
   "14P25" AT %I19.7 : Bool;   // 5#机械手负压检测4
   "14S81" AT %I20.0 : Bool;
   "14S82" AT %I20.1 : Bool;
   "14S83" AT %I20.2 : Bool;
   "14L19" AT %I20.3 : Bool;
   "14S84" AT %I20.4 : Bool;
   "14L20" AT %I20.5 : Bool;
   "14S85" AT %I20.6 : Bool;
   "14L21" AT %I20.7 : Bool;
   "14S86" AT %I21.0 : Bool;
   "14S87" AT %I21.1 : Bool;
   "14S88" AT %I21.2 : Bool;
   "14S89" AT %I21.3 : Bool;
   "14P26" AT %I21.4 : Bool;
   "14P27" AT %I21.5 : Bool;
   "14P28" AT %I21.6 : Bool;
   "14P29" AT %I21.7 : Bool;
   "14HL43" AT %Q14.0 : Bool;   // 备用
   "%Q14.1" AT %Q14.1 : Bool;   // 备用
   "%Q14.2" AT %Q14.2 : Bool;   // 5#机械手Z轴抱闸
   "%Q14.3" AT %Q14.3 : Bool;   // 5#伺服启停
   "%Q14.4" AT %Q14.4 : Bool;
   "%Q14.5" AT %Q14.5 : Bool;   // 10#库位红灯
   "%Q14.6" AT %Q14.6 : Bool;   // 5#机械手X轴抱闸
   "等级漏按蜂鸣器" AT %Q14.7 : Bool;
   "%Q15.0" AT %Q15.0 : Bool;
   "%Q15.1" AT %Q15.1 : Bool;
   "%Q15.2" AT %Q15.2 : Bool;
   "%Q15.3" AT %Q15.3 : Bool;
   "%Q15.4" AT %Q15.4 : Bool;
   "%Q15.5" AT %Q15.5 : Bool;
   "%Q15.6" AT %Q15.6 : Bool;
   "视觉拍照触发" AT %Q15.7 : Bool;
   "Tag_12" AT %MB510 : Byte;
   "5#Z轴编码器清零" AT %M7.5 : Bool;
   "5#机械手Z轴速度写入值" AT %QW264 : Word;
   "6#机械手Z轴速度写入值" AT %QW266 : Word;
   "7#机械手Z轴速度写入值" AT %QW268 : Word;
   "5#手动Z轴下降" AT %M18.0 : Bool;
   "5#手动Z轴上升" AT %M18.1 : Bool;
   "5#手动X轴2库移动" AT %M18.2 : Bool;
   "5#手动X轴1库移动" AT %M18.3 : Bool;
   "5#手动W轴前移" AT %M18.4 : Bool;
   "5#手动W轴回原位" AT %M18.5 : Bool;
   "5#手动吸盘电磁阀打开" AT %M18.6 : Bool;
   "5#手动吸盘电磁阀关闭" AT %M18.7 : Bool;
   "6#手动吸盘电磁阀关闭" AT %M17.7 : Bool;
   "7#手动Z轴下降" AT %M19.0 : Bool;
   "7#手动Z轴上升" AT %M19.1 : Bool;
   "7#手动X轴2库移动" AT %M19.2 : Bool;
   "7#手动X轴1库移动" AT %M19.3 : Bool;
   "7#手动W轴前移" AT %M19.4 : Bool;
   "7#手动W轴回原位" AT %M19.5 : Bool;
   "7#手动吸盘电磁阀打开" AT %M19.6 : Bool;
   "5#机械手单独复位标志位" AT %M63.4 : Bool;
   "5#机械手系统运行标志" AT %M8.0 : Bool;
   "5#机械手系统复位标志" AT %M8.4 : Bool;
   "5#机械手系统急停限位标志" AT %M60.4 : Bool;
   "5#1压力开关报警" AT %M71.0 : Bool;
   "5#2压力开关报警" AT %M71.1 : Bool;
   "5#3压力开关报警" AT %M71.2 : Bool;
   "5#4压力开关报警" AT %M71.3 : Bool;
   "9#库安全光电报警" AT %M80.0 : Bool;
   "10#库安全光电报警" AT %M80.1 : Bool;
   "7#手动吸盘电磁阀关闭" AT %M19.7 : Bool;
   "6#机械手单独复位标志位" AT %M63.5 : Bool;
   "6#机械手系统运行标志" AT %M8.1 : Bool;
   "6#机械手系统复位标志" AT %M8.5 : Bool;
   "6#机械手系统急停限位标志" AT %M60.5 : Bool;
   "6#1压力开关报警" AT %M71.4 : Bool;
   "6#2压力开关报警" AT %M71.5 : Bool;
   "6#3压力开关报警" AT %M71.6 : Bool;
   "6#4压力开关报警" AT %M71.7 : Bool;
   "11#库安全光电报警" AT %M80.2 : Bool;
   "12#库安全光电报警" AT %M80.3 : Bool;
   "7#机械手单独复位标志位" AT %M63.6 : Bool;
   "7#机械手系统运行标志" AT %M8.2 : Bool;
   "7#机械手系统复位标志" AT %M8.6 : Bool;
   "7#机械手系统急停限位标志" AT %M60.6 : Bool;
   "7#1压力开关报警" AT %M72.0 : Bool;
   "7#2压力开关报警" AT %M72.1 : Bool;
   "7#3压力开关报警" AT %M72.2 : Bool;
   "7#4压力开关报警" AT %M72.3 : Bool;
   "13#库安全光电报警" AT %M80.4 : Bool;
   "14#库安全光电报警" AT %M80.5 : Bool;
   "6#Z轴编码器清零" AT %M7.6 : Bool;
   "7#Z轴编码器清零" AT %M7.7 : Bool;
   "Tag_20" AT %ID100 : DInt;
   "Tag_8" AT %MD700 : DWord;
   "Tag_18" AT %MD710 : DWord;
   "Tag_21" AT %MD714 : DWord;
   "Tag_22" AT %MD718 : DWord;
   "Tag_23" AT %Q109.0 : Bool;
   "Tag_24" AT %Q108.0 : Bool;
   "Tag_25" AT %Q120.0 : Bool;
   "Tag_26" AT %Q121.0 : Bool;
   "Tag_27" AT %ID116 : DInt;
   "Tag_28" AT %MB500 : Byte;
   "16机拥堵" AT %MB501 : Byte;
   "16可否进砖=》14" AT %MB502 : Byte;
   "询问16可否砖放行" AT %MB511 : Byte;
   "Tag_29" AT %M650.0 : Bool;
   "Tag_30" AT %M650.1 : Bool;
   "Tag_31" AT %MD651 : DWord;
   "Tag_32" AT %M650.2 : Bool;
   "和18发送数据" AT %M0.4 : Bool;
   "Tag_3" AT %MD550 : DInt;
   "Tag_33" AT %MD554 : DInt;
   "Tag_34" AT %MB586 : Byte;
   "Tag_35" AT %MB587 : Byte;
   "Tag_36" AT %M580.0 : Bool;
   "Tag_37" AT %MD580 : DInt;
   "Tag_38" AT %MD584 : DInt;
   "Tag_39" AT %M590.0 : Bool;
   "Tag_40" AT %M590.1 : Bool;
   "Tag_41" AT %M595.0 : Bool;
   "Tag_43" AT %MB512 : Byte;
   "Tag_44" AT %M588.0 : Bool;
   "Tag_45" AT %M81.0 : Bool;
   "Tag_46" AT %M81.1 : Bool;
   "Tag_47" AT %M81.2 : Bool;
   "Tag_48" AT %M81.3 : Bool;
   "Tag_49" AT %M81.4 : Bool;
   "Tag_50" AT %M81.5 : Bool;
   "Tag_51" AT %M81.6 : Bool;
   "Tag_52" AT %M81.7 : Bool;
   "Tag_53" AT %M82.0 : Bool;
   "Tag_54" AT %M82.1 : Bool;
   "Tag_55" AT %M82.2 : Bool;
   "Tag_56" AT %M82.3 : Bool;
   "Tag_57" AT %M82.4 : Bool;
   "Tag_58" AT %M82.5 : Bool;
   "5#找待命位速度" AT %M69.5 : Bool;
   "Tag_59" AT %MB631 : Byte;
   "通讯发送" AT %M0.5 : Bool;
   "Tag_60" AT %MB600 : Byte;
   "Tag_61" AT %MB601 : Byte;
   "Tag_64" AT %MB602 : Byte;
   "Tag_65" AT %MB700 : Byte;
   "Tag_67" AT %MB701 : Byte;
   "Tag_70" AT %MB702 : Byte;
   "备用(1)" AT %Q16.0 : Bool;
   "Tag_71" AT %MB703 : Byte;
   "Tag_77" AT %MB705 : Byte;
   "Tag_78" AT %MB704 : Byte;
   "Tag_79" AT %MB509 : Byte;
   "Tag_80" AT %MB706 : Byte;
   "Tag_81" AT %MW800 : Int;
   "输送带运行给16" AT %QB212 : Byte;
   "询问16可否放砖" AT %QB211 : Byte;
   "16段机拥堵" AT %IB211 : Byte;
   "14是否能放砖到16" AT %IB212 : Byte;
   "Tag_82" AT %I210.0 : Bool;
   "Tag_83" AT %I210.1 : Bool;
END_VAR

DATA_BLOCK "定义时间继电器"   // DB14
{ S7_Optimized_Access := 'FALSE' }
VERSION : 0.1
   VAR
      T1 : IEC_TIMER;
      T_Time_1 : Time := T#1000ms;
      T2 : IEC_TIMER;
      T_Time_2 : Time := T#1000ms;
      T3 : IEC_TIMER;
      T_Time_3 : Time := T#0ms;
      T4 : IEC_TIMER;
      T_Time_4 : Time;
      T5 : IEC_TIMER;
      T200 : IEC_TIMER;   // 使用
      T_Time_200 : Time;
      T201 : IEC_TIMER;   // 使用
      T_Time_201 : Time;
      T202 : IEC_TIMER;   // 使用
      T_Time_202 : Time;
      T203 : IEC_TIMER;   // 使用
      T_Time_203 : Time;
      T204 : IEC_TIMER;   // 使用
      T_Time_204 : Time;
      T205 : IEC_TIMER;   // 使用
      T_Time_205 : Time;
      T206 : IEC_TIMER;
      T_Time_206 : Time;
      T207 : IEC_TIMER;   // 使用
      T_Time_207 : Time;
      T208 : IEC_TIMER;   // 使用
      T_Time_208 : Time;
      T209 : IEC_TIMER;   // 使用
      T_Time_209 : Time;
      T210 : IEC_TIMER;   // 使用
      T_Time_210 : Time;
      T211 : IEC_TIMER;   // 使用
      T_Time_211 : Time;
      T212 : IEC_TIMER;   // 使用
      T_Time_212 : Time;
      T213 : IEC_TIMER;   // 使用
      T_Time_213 : Time;
      T214 : IEC_TIMER;   // 使用
      T_Time_214 : Time;
      T215 : IEC_TIMER;   // 使用
      T_Time_215 : Time;
      T216 : IEC_TIMER;
      T_Time_216 : Time;
      T217 : IEC_TIMER;
      T_Time_217 : Time;
      T218 : IEC_TIMER;   // 使用
      T_Time_218 : Time;
      T219 : IEC_TIMER;   // 使用
      T_Time_219 : Time;
      T220 : IEC_TIMER;
      T_Time_220 : Time;
      T221 : IEC_TIMER;   // 使用
      T_Time_221 : Time;
      T222 : IEC_TIMER;   // 使用
      T_Time_222 : Time;
      T223 : IEC_TIMER;   // 使用
      T_Time_223 : Time;
      T224 : IEC_TIMER;   // 使用
      T_Time_224 : Time;
      T225 : IEC_TIMER;   // 使用
      T_Time_225 : Time;
      T226 : IEC_TIMER;   // 使用
      T_Time_226 : Time;
      T227 : IEC_TIMER;   // 使用
      T_Time_227 : Time;
      T228 : IEC_TIMER;   // 使用
      T_Time_228 : Time;
      T229 : IEC_TIMER;   // 使用
      T_Time_229 : Time;
      T230 : IEC_TIMER;   // 使用
      T_Time_230 : Time;
      T231 : IEC_TIMER;   // 使用
      T_Time_231 : Time;
      T232 : IEC_TIMER;   // 使用
      T_Time_232 : Time;
      T233 : IEC_TIMER;   // 使用
      T_Time_233 : Time;
      T234 : IEC_TIMER;   // 使用
      T_Time_234 : Time;
      T235 : IEC_TIMER;
      T_Time_235 : Time;
      T236 : IEC_TIMER;
      T_Time_236 : Time;
      T237 : IEC_TIMER;
      T_Time_237 : Time;
      T238 : IEC_TIMER;
      T_Time_238 : Time;
      T239 : IEC_TIMER;
      T_Time_239 : Time;
      T240 : IEC_TIMER;
      T_Time_240 : Time;
      T241 : IEC_TIMER;
      T_Time_241 : Time;
      T242 : IEC_TIMER;
      T_Time_242 : Time;
      T243 : IEC_TIMER;
      T_Time_243 : Time;
      T244 : IEC_TIMER;
      T_Time_244 : Time;
      T245 : IEC_TIMER;
      T_Time_245 : Time;
      T246 : IEC_TIMER;
      T_Time_246 : Time;
      T247 : IEC_TIMER;
      T_Time_247 : Time;
      T248 : IEC_TIMER;
      T_Time_248 : Time;
      T249 : IEC_TIMER;
      T_Time_249 : Time;
      T250 : IEC_TIMER;
      T_Time_250 : Time;
      T251 : IEC_TIMER;
      T_Time_251 : Time;
      T252 : IEC_TIMER;
      T_Time_252 : Time;
      T253 : IEC_TIMER;
      T_Time_253 : Time;
      T254 : IEC_TIMER;
      T_Time_254 : Time;
      T255 : IEC_TIMER;
      T_Time_255 : Time;
      T256 : IEC_TIMER;
      T_Time_256 : Time;
   END_VAR
BEGIN
END_DATA_BLOCK

DATA_BLOCK "P_N_"   // DB24
{ S7_Optimized_Access := 'FALSE' }
VERSION : 0.1
   VAR
      "P-" : Bool;   // 1
      P_ : Bool;   // 1
      "P-_1" : Bool;   // 1
      P_1 : Bool;   // 1
      "P-_2" : Bool;   // 1
      P_2 : Bool;   // 1
      "P-_3" : Bool;   // 1
      P_3 : Bool;   // 1
      "P-_4" : Bool;   // 1
      P_4 : Bool;   // 1
      "P-_5" : Bool;   // 1
      P_5 : Bool;   // 1
      "P-_6" : Bool;   // 1
      P_6 : Bool;   // 1
      "P-_7" : Bool;   // 1
      P_7 : Bool;   // 1
      "P-_8" : Bool;   // 1
      P_8 : Bool;   // 1
      "P-_9" : Bool;   // 1
      P_9 : Bool;   // 1
      "P-_10" : Bool;   // 1
      P_10 : Bool;
      "P-_11" : Bool;
      P_11 : Bool;
      "P-_12" : Bool;
      P_12 : Bool;
      "P-_13" : Bool;
      P_13 : Bool;
      "P-_14" : Bool;
      P_14 : Bool;
      P_15 : Bool;
      P_16 : Bool;
      P_17 : Bool;
      P_18 : Bool;
      P_19 : Bool;
      P_20 : Bool;
      P_21 : Bool;
      P_22 : Bool;
      P_23 : Bool;
      P_24 : Bool;
      P_25 : Bool;
      P_26 : Bool;
      P_27 : Bool;
      P_28 : Bool;
      P_29 : Bool;
      P_30 : Bool;
      P_31 : Bool;
      P_32 : Bool;   // 1
      P_33 : Bool;   // 1
      P_34 : Bool;   // 1
      P_35 : Bool;   // 1
      P_36 : Bool;
      P_37 : Bool;
      P_38 : Bool;
      P_39 : Bool;   // 1
      P_40 : Bool;   // 1
      P_41 : Bool;   // 1
      P_42 : Bool;   // 1
      P_43 : Bool;
      P_44 : Bool;   // 1
      P_45 : Bool;   // 1
      P_46 : Bool;   // 1
      P_47 : Bool;   // 1
      P_48 : Bool;   // 1
      P_49 : Bool;   // 1
      P_50 : Bool;
      P_51 : Bool;
      P_52 : Bool;
      P_53 : Bool;
      P_54 : Bool;
      Static_1 : Byte;
   END_VAR
BEGIN
END_DATA_BLOCK

// folder: 14工位

DATA_BLOCK "1#机械手_DB"   // DB10
{ S7_Optimized_Access := 'TRUE' }
VERSION : 0.1
// stored: InstanceOfName 库位动作流程
"库位动作流程"
BEGIN
END_DATA_BLOCK

DATA_BLOCK "2#机械手_DB"   // DB11
{ S7_Optimized_Access := 'TRUE' }
VERSION : 0.1
// stored: InstanceOfName 库位动作流程
"库位动作流程"
BEGIN
END_DATA_BLOCK

DATA_BLOCK "3#机械手_DB"   // DB12
{ S7_Optimized_Access := 'TRUE' }
VERSION : 0.1
// stored: InstanceOfName 库位动作流程
"库位动作流程"
BEGIN
END_DATA_BLOCK

DATA_BLOCK "4#机械手_DB"   // DB13
{ S7_Optimized_Access := 'TRUE' }
VERSION : 0.1
// stored: InstanceOfName 库位动作流程
"库位动作流程"
BEGIN
END_DATA_BLOCK

DATA_BLOCK "编码器参数数据"   // DB19
{ S7_Optimized_Access := 'FALSE' }
VERSION : 0.1
   VAR
      "1#busy" : Bool;
      "1#status" : Word;
      "2#busy" : Bool;
      "2#status" : Word;
      "3#busy" : Bool;
      "3#status" : Word;
      "4#busy" : Bool;
      "4#status" : Word;
      "5#busy" : Bool;
      "5#status" : Word;
      "6#busy" : Bool;
      "6#status" : Word;
      "通讯断开次数-上位机" : DInt;
   END_VAR
BEGIN
END_DATA_BLOCK

DATA_BLOCK "Z轴速度"   // DB21
{ S7_Optimized_Access := 'FALSE' }
VERSION : 0.1
   VAR
      X轴是否走曲线 : DInt;
   END_VAR
BEGIN
END_DATA_BLOCK

DATA_BLOCK "W轴速度"   // DB23
{ S7_Optimized_Access := 'FALSE' }
VERSION : 0.1
   VAR
      "1#W轴最大速" : Real := 100000.0;   // 最大速度 1#机械手
      "1#W轴设定速度" : Real;   // 速度设定 1#机械手
      VSET1 : Real;   // 1#机械手
      VSET2 : Real;   // 1#机械手
      VSET3 : Real;   // 1#机械手
      Vact : Real;   // 1#机械手
      "1#W轴加减速时间" : DInt;   // 加减速时间 1#机械手
      "A" : Real;   // 1#机械手
      p : Array[0..7] of Bool;   // 1#机械手
      start : Bool;   // 开关 1#机械手
      脉冲累计 : Real;   // 脉冲累计 1#机械手
      "1#步进回中间位脉冲值" : Real;
      "1#步进电机累计脉冲" : Real;
      备用 : DInt;
      备用_1 : DInt;
      备用_2 : DInt;
      备用_3 : DInt;
      "2#W轴最大速" : Real := 100000.0;   // 最大速度 2#机械手
      "2#W轴设定速度" : Real := 0.0;   // 速度设定 2#机械手
      VSET4 : Real := 0.0;   // 2#机械手
      VSET5 : Real := 0.0;   // 2#机械手
      VSET6 : Real := 0.0;   // 2#机械手
      Vact_1 : Real := 0.0;   // 2#机械手
      "2#W轴加减速时间" : DInt := 0;   // 加减速时间 2#机械手
      A_1 : Real := 0.0;   // 2#机械手
      p_1 : Array[0..7] of Bool;   // 2#机械手
      start_1 : Bool := false;   // 开关 2#机械手
      脉冲累计_1 : Real;   // 脉冲累计 2#机械手
      "2#步进回中间位脉冲值" : Real;
      "2#步进电机累计脉冲" : Real;
      备用_4 : DInt := 0;
      备用_5 : DInt := 0;
      备用_6 : DInt := 0;
      备用_7 : DInt := 0;
      "3#W轴最大速" : Real := 100000.0;   // 最大速度 3#机械手
      "3#W轴设定速度" : Real := 0.0;   // 速度设定 3#机械手
      VSET7 : Real := 0.0;   // 3#机械手
      VSET8 : Real := 0.0;   // 3#机械手
      VSET9 : Real := 0.0;   // 3#机械手
      Vact_2 : Real := 0.0;   // 3#机械手
      "3#W轴加减速时间" : DInt := 0;   // 加减速时间 3#机械手
      A_2 : Real := 0.0;   // 3#机械手
      p_2 : Array[0..7] of Bool;   // 3#机械手
      start_2 : Bool := false;   // 开关 3#机械手
      脉冲累计_12 : Real;   // 脉冲累计 3#机械手
      "3#步进回中间位脉冲值" : Real;
      "3#步进电机累计脉冲" : Real;
      备用_8 : DInt := 0;
      备用_9 : DInt := 0;
      备用_10 : DInt := 0;
      备用_11 : DInt := 0;
      "4#W轴最大速" : Real := 100000.0;   // 最大速度 4#机械手
      "4#W轴设定速度" : Real := 0.0;   // 速度设定 4#机械手
      VSET10 : Real := 0.0;   // 4#机械手
      VSET11 : Real := 0.0;   // 4#机械手
      VSET12 : Real := 0.0;   // 4#机械手
      Vact_3 : Real := 0.0;   // 4#机械手
      "4#W轴加减速时间" : DInt := 0;   // 加减速时间 4#机械手
      A_3 : Real := 0.0;   // 4#机械手
      p_3 : Array[0..7] of Bool;   // 4#机械手
      start_3 : Bool := false;   // 开关 4#机械手
      脉冲累计_18 : Real;   // 脉冲累计 4#机械手
      "4#步进回中间位脉冲值" : Real;
      "4#步进电机累计脉冲" : Real;
      备用_12 : DInt := 0;
      备用_13 : DInt := 0;
      备用_14 : DInt := 0;
      备用_15 : DInt := 0;
      步进电机同步线速度停止脉冲 : Real;
      步进电机前往取砖位脉冲 : Real;
      步进电机带载运行速度 : Real;
      步进电机空载运行速度 : Real;
      "伺服同步速度-暂时使用" : DInt := 6000;
   END_VAR
BEGIN
END_DATA_BLOCK

DATA_BLOCK "5#机械手_DB"   // DB27
{ S7_Optimized_Access := 'TRUE' }
VERSION : 0.1
// stored: InstanceOfName 库位动作流程
"库位动作流程"
BEGIN
END_DATA_BLOCK

DATA_BLOCK "1#手动_DB"   // DB37
{ S7_Optimized_Access := 'TRUE' }
VERSION : 0.1
// stored: InstanceOfName 手动
"手动"
BEGIN
END_DATA_BLOCK

DATA_BLOCK "2#手动_DB"   // DB38
{ S7_Optimized_Access := 'TRUE' }
VERSION : 0.1
// stored: InstanceOfName 手动
"手动"
BEGIN
END_DATA_BLOCK

DATA_BLOCK "3#手动_DB"   // DB39
{ S7_Optimized_Access := 'TRUE' }
VERSION : 0.1
// stored: InstanceOfName 手动
"手动"
BEGIN
END_DATA_BLOCK

DATA_BLOCK "4#手动_DB"   // DB40
{ S7_Optimized_Access := 'TRUE' }
VERSION : 0.1
// stored: InstanceOfName 手动
"手动"
BEGIN
END_DATA_BLOCK

DATA_BLOCK "5#手动_DB"   // DB41
{ S7_Optimized_Access := 'TRUE' }
VERSION : 0.1
// stored: InstanceOfName 手动
"手动"
BEGIN
END_DATA_BLOCK

// folder: System blocks/Program resources

DATA_BLOCK "14PLC_PC_1_DB"   // DB5
{ S7_Optimized_Access := 'TRUE' }
AUTHOR : SIMATIC
FAMILY : MC7Plus
NAME : TC_IP_v4
VERSION : 1.0
// stored: InstanceOfName TCON_IP_v4
"TCON_IP_v4"
BEGIN
   InterfaceId := 64;
   ID := 1;
   LocalPort := 2004;
   RemoteAddress.ADDR[1] := 192;
   RemoteAddress.ADDR[2] := 168;
   RemoteAddress.ADDR[4] := 100;
END_DATA_BLOCK

// folder: 通讯

DATA_BLOCK "数据接收"   // DB1
{ S7_Optimized_Access := 'FALSE' }
VERSION : 0.1
   VAR
      通信交换 : Bool;   // 交换位 (0、1变化)
      测试模式 : Bool;   // 测试模式（0、测试 1、正常）
      询问可否砖放行 : Bool;   // （1询问 0停止）
      输送手动调试 : Bool;   // 输送线手动
      PC状态 : Byte;   // PC状态（0正常1等待2手动）
      Z轴减速距离 : Int;   // Z轴机械手减速值 脉冲值
      Z轴待命值 : Int;   // Z轴起始位置 待命位置
      X轴提前回待命脉冲值 : Int;   // X轴提前回待命位脉冲
      Z轴提前下降脉冲值 : Int;   // 取砖X轴提前下降 脉冲设定
      备用1 : DInt;
      备用2 : DInt;
      备用3 : DInt;
      备用4 : DInt;
      库位方向_1 : Bool;   // 1号机械手抓取方向 （0《1-A》，0《1-B》）
      单独复位_1 : Bool;   // 1#机械手单独复位（0复位 1完成）
      库位满_1 : Bool;   // 1#库位库满（0满 1不满）
      库位满_2 : Bool;   // 2#库位库满（0满 1不满）
      条码读取状态_1 : Bool;   // 1#库条码读取（1成功0失败）
      条码读取状态_2 : Bool;   // 2#库条码读取（1成功0失败）
      手自动状态_1 : Bool;   // 1号机械手手动 （0手动，1自动）
      开真空_1 : Bool;   // 真空电磁阀 （0打开，1关闭）
      手动前后_1 : Byte;   // 伺服 （0.停止 1.前 2.后）
      手动左右_1 : Byte;   // X轴 （0.停止 1左，2右）
      手动上下_1 : Byte;   // Z轴 （0.停止 1上，2下）
      取砖完成等待_1 : Byte;   // 0等待，1放库位 2放皮带
      抓放指令_1 : Byte;   // 取放砖指令 （0.停止 1取，2放）
      Z轴高速转低速脉冲_1 : Int;   // 1#Z轴高速转低速脉冲
      抓放目标值_1 : DInt;   // 1#抓取目标脉冲（输送线脉冲）
      备用5 : DInt;
      备用6 : DInt;
      备用7 : DInt;
      备用8 : DInt;
      库位方向_2 : Bool;   // 2号机械手抓取方向 （0《1-A》，0《1-B》）
      单独复位_2 : Bool;   // 2#机械手单独复位（0复位 1完成）
      库位满_3 : Bool;   // 3#库位库满（0满 1不满）
      库位满_4 : Bool;   // 4#库位库满（0满 1不满）
      条码读取状态_3 : Bool;   // 3#库条码读取（1成功0失败）
      条码读取状态_4 : Bool;   // 4#库条码读取（1成功0失败）
      手自动状态_2 : Bool;   // 2号机械手手动 （0手动，1自动）
      开真空_2 : Bool;   // 真空电磁阀 （0打开，1关闭）
      手动前后_2 : Byte;   // 伺服 （0.停止 1.前 2.后）
      手动左右_2 : Byte;   // X轴 （0.停止 1左，2右）
      手动上下_2 : Byte;   // Z轴 （0.停止 1上，2下）
      取砖完成等待_2 : Byte;   // 0等待，1放库位 2放皮带
      抓放指令_2 : Byte;   // 取放砖指令 （0.停止 1取，2放）
      Z轴高速转低速脉冲_2 : Int;   // 2#Z轴高速转低速脉冲
      抓放目标值_2 : DInt;   // 2#抓取目标脉冲（输送线脉冲）
      备用9 : DInt;
      备用10 : DInt;
      备用11 : DInt;
      备用12 : DInt;
      库位方向_3 : Bool;   // 3号机械手抓取方向 （0《1-A》，0《1-B》）
      单独复位_3 : Bool;   // 3#机械手单独复位（0复位 1完成）
      库位满_5 : Bool;   // 5#库位库满（0满 1不满）
      库位满_6 : Bool;   // 6#库位库满（0满 1不满）
      条码读取状态_5 : Bool;   // 5#库条码读取（1成功0失败）
      条码读取状态_6 : Bool;   // 6#库条码读取（1成功0失败）
      手自动状态_3 : Bool;   // 3号机械手手动 （0手动，1自动）
      开真空_3 : Bool;   // 真空电磁阀 （0打开，1关闭）
      手动前后_3 : Byte;   // 伺服 （0.停止 1.前 2.后）
      手动左右_3 : Byte;   // X轴 （0.停止 1左，2右）
      手动上下_3 : Byte;   // Z轴 （0.停止 1上，2下）
      取砖完成等待_3 : Byte;   // 0等待，1放库位 2放皮带
      抓放指令_3 : Byte;   // 取放砖指令 （0.停止 1取，2放）
      Z轴高速转低速脉冲_3 : Int;   // 3#Z轴高速转低速脉冲
      抓放目标值_3 : DInt;   // 3#抓取目标脉冲（输送线脉冲）
      备用13 : DInt;
      备用14 : DInt;
      备用15 : DInt;
      备用16 : DInt;
      库位方向_4 : Bool;   // 4号机械手抓取方向 （0《1-A》，0《1-B》）
      单独复位_4 : Bool;   // 4#机械手单独复位（0复位 1完成）
      库位满_7 : Bool;   // 7#库位库满（0满 1不满）
      库位满_8 : Bool;   // 8#库位库满（0满 1不满）
      条码读取状态_7 : Bool;   // 7#库条码读取（1成功0失败）
      条码读取状态_8 : Bool;   // 8#库条码读取（1成功0失败）
      手自动状态_4 : Bool;   // 4号机械手手动 （0手动，1自动）
      开真空_4 : Bool;   // 真空电磁阀 （0打开，1关闭）
      手动前后_4 : Byte;   // 伺服 （0.停止 1.前 2.后）
      手动左右_4 : Byte;   // X轴 （0.停止 1左，2右）
      手动上下_4 : Byte;   // Z轴 （0.停止 1上，2下）
      取砖完成等待_4 : Byte;   // 0等待，1放库位 2放皮带
      抓放指令_4 : Byte;   // 取放砖指令 （0.停止 1取，2放）
      Z轴高速转低速脉冲_4 : Int;   // 4#Z轴高速转低速脉冲
      抓放目标值_4 : DInt;   // 4#抓取目标脉冲（输送线脉冲）
      备用17 : DInt;
      备用18 : DInt;
      备用19 : DInt;
      备用20 : DInt;
      库位方向_5 : Bool;   // 5号机械手抓取方向 （0《1-A》，0《1-B》）
      单独复位_5 : Bool;   // 5#机械手单独复位（0复位 1完成）
      库位满_9 : Bool;   // 9#库位库满（0满 1不满）
      库位满_10 : Bool;   // 10#库位库满（0满 1不满）
      条码读取状态_9 : Bool;   // 9#库条码读取（1成功0失败）
      条码读取状态_10 : Bool;   // 10#库条码读取（1成功0失败）
      手自动状态_5 : Bool;   // 5号机械手手动 （0手动，1自动）
      开真空_5 : Bool;   // 真空电磁阀 （0打开，1关闭）
      手动前后_5 : Byte;   // 伺服 （0.停止 1.前 2.后）
      手动左右_5 : Byte;   // X轴 （0.停止 1左，2右）
      手动上下_5 : Byte;   // Z轴 （0.停止 1上，2下）
      取砖完成等待_5 : Byte;   // 0等待，1放库位 2放皮带
      抓放指令_5 : Byte;   // 取放砖指令 （0.停止 1取，2放）
      Z轴高速转低速脉冲_5 : Int;   // 5#Z轴高速转低速脉冲
      抓放目标值_5 : DInt;   // 5#抓取目标脉冲（输送线脉冲）
      备用21 : DInt;
      备用22 : DInt;
      备用23 : DInt;
      备用24 : DInt;
   END_VAR
BEGIN
END_DATA_BLOCK

DATA_BLOCK "数据发送"   // DB2
{ S7_Optimized_Access := 'FALSE' }
VERSION : 0.1
   VAR
      队列光电1 : Bool;   // 输送线分级进砖光电
      队列光电2 : Bool;
      队列光电3 : Bool;
      队列光电4 : Bool;   // 输送线编码器记值光电（1有，0无）
      "16机连锁" : Bool;   // （1连锁 0解除）
      上位机是否放砖到16 : Bool;   // （0. 放砖 1.不能放砖）
      设备报警 : Array[0..15] of Bool;
      瓷砖等级 : Byte;   // 瓷砖等级判断（一级1二级2三级3）
      换花色 : Byte;   // 换花色
      系统状态 : Byte;   // 系统参数（1正常，2复位，3急停）
      进砖起始编码值 : DInt;   // 砖起始位置编码值
      输送线实时值 : DInt;   // 输送线编码器实时值（10万清零）
      备用 : DInt;
      备用_1 : DInt;
      备用_2 : DInt;
      备用_3 : DInt;
      放砖动作完成_1 : Bool;   // 1号机械手放砖完成（1有，0无）
      取砖动作完成_1 : Bool;   // 1号机械手吸取到位光电（1有0无）
      机械手就绪_1 : Bool;   // 1号机械手待命位置（1有0无）
      放砖确认等待_1 : Bool;   // 放砖模式（1#机械手放砖等待）给上位机1
      库位安全报警_1 : Bool;   // 1#库位安全光电报警
      库位安全报警_2 : Bool;   // 2#库位安全光电报警
      机械手报警_1 : Array[0..15] of Bool;
      机械手复位状态_1 : Byte;   // 1#机械手复位状态（1复位2完成3报警）
      Z轴编码实时值_1 : DInt;   // 1#机械手编码器实时值
      备用_4 : DInt;
      备用_5 : DInt;
      备用_6 : DInt;
      备用_7 : DInt;
      放砖动作完成_2 : Bool;   // 2号机械手放砖完成（1有，0无）
      取砖动作完成_2 : Bool;   // 2号机械手吸取到位光电（1有0无）
      机械手就绪_2 : Bool;   // 2号机械手待命位置（1有0无）
      放砖确认等待_2 : Bool;   // 放砖模式（1#机械手放砖等待）给上位机1
      库位安全报警_3 : Bool;   // 3#库位安全光电报警
      库位安全报警_4 : Bool;   // 4#库位安全光电报警
      机械手报警_2 : Array[0..15] of Bool;
      机械手复位状态_2 : Byte;   // 2#机械手复位状态（1复位2完成3报警）
      Z轴编码实时值_2 : DInt;   // 2#机械手编码器实时值
      备用_8 : DInt;
      备用_9 : DInt;
      备用_10 : DInt;
      备用_11 : DInt;
      放砖动作完成_3 : Bool;   // 3号机械手放砖完成（1有，0无）
      取砖动作完成_3 : Bool;   // 3号机械手吸取到位光电（1有0无）
      机械手就绪_3 : Bool;   // 3号机械手待命位置（1有0无）
      放砖确认等待_3 : Bool;   // 放砖模式（1#机械手放砖等待）给上位机1
      库位安全报警_5 : Bool;   // 5#库位安全光电报警
      库位安全报警_6 : Bool;   // 6#库位安全光电报警
      机械手报警_3 : Array[0..15] of Bool;
      机械手复位状态_3 : Byte;   // 3#机械手复位状态（1复位2完成3报警）
      Z轴编码实时值_3 : DInt;   // 3#机械手编码器实时值
      备用_12 : DInt;
      备用_13 : DInt;
      备用_14 : DInt;
      备用_15 : DInt;
      放砖动作完成_4 : Bool;   // 4号机械手放砖完成（1有，0无）
      取砖动作完成_4 : Bool;   // 4号机械手吸取到位光电（1有0无）
      机械手就绪_4 : Bool;   // 4号机械手待命位置（1有0无）
      放砖确认等待_4 : Bool;   // 放砖模式（1#机械手放砖等待）给上位机1
      库位安全报警_7 : Bool := 0;   // 7#库位安全光电报警
      库位安全报警_8 : Bool;   // 8#库位安全光电报警
      机械手报警_4 : Array[0..15] of Bool;
      机械手复位状态_4 : Byte;   // 4#机械手复位状态（1复位2完成3报警）
      Z轴编码实时值_4 : DInt;   // 4#机械手编码器实时值
      备用_16 : DInt;
      备用_17 : DInt;
      备用_18 : DInt;
      备用_19 : DInt;
      放砖动作完成_5 : Bool;   // 5号机械手放砖完成（1有，0无）
      取砖动作完成_5 : Bool;   // 5号机械手吸取到位光电（1有0无）
      机械手就绪_5 : Bool;   // 5号机械手待命位置（1有0无）
      放砖确认等待_5 : Bool;   // 放砖模式（1#机械手放砖等待）给上位机1
      库位安全报警_9 : Bool;   // 9#库位安全光电报警
      库位安全报警_10 : Bool;   // 10#库位安全光电报警
      机械手报警_5 : Array[0..15] of Bool;
      机械手复位状态_5 : Byte;   // 5#机械手复位状态（1复位2完成3报警）
      Z轴编码实时值_5 : DInt;   // 5#机械手编码器实时值
      备用_20 : DInt;
      备用_21 : DInt;
      备用_22 : DInt;
      备用_23 : DInt;
   END_VAR
BEGIN
END_DATA_BLOCK

DATA_BLOCK "端口数据1"   // DB3
{ S7_Optimized_Access := 'FALSE' }
VERSION : 0.1
   VAR
      TCON_DONE1 : Bool;   // 建立通讯1
      TCON_BUSY1 : Bool;   // 建立通讯1
      TCON_ERROR1 : Bool;   // 建立通讯1
      TCON_STATUS1 : Word;   // 建立通讯1
      TDISCON_DONE1 : Bool;   // 断开通讯1
      TDISCON_BUSY1 : Bool;   // 断开通讯1
      TDISCON_ERROR1 : Bool;   // 断开通讯1
      TDISCON_STATUS1 : Word;   // 断开通讯1
      TSEND_DONE1 : Bool;   // 发送数据1
      TSEND_BUSY1 : Bool;   // 发送数据1
      TSEND_ERROR1 : Bool;   // 发送数据1
      TSEND_STATUS1 : Word;   // 发送数据1
      TRCV_NDR1 : Bool;   // 接收数据1
      TRCV_BUSY1 : Bool;   // 接收数据1
      TRCV_ERROR1 : Bool;   // 接收数据1
      TRCV_STATUS1 : Word;   // 接收数据1
      TRCV_RCVD_LEN1 : Word;   // 接收数据1
      TCON_DONE2 : Bool;   // 建立通讯2
      TCON_BUSY2 : Bool;   // 建立通讯2
      TCON_ERROR2 : Bool;   // 建立通讯2
      TCON_STATUS2 : Word;   // 建立通讯2
      TSEND_DONE2 : Bool;   // 发送数据2
      TSEND_BUSY2 : Bool;   // 发送数据2
      TSEND_ERROR2 : Bool;   // 发送数据2
      TSEND_STATUS2 : Word;   // 发送数据2
      TRCV_NDR2 : Bool;   // 接收数据2
      TRCV_BUSY2 : Bool;   // 接收数据2
      TRCV_ERROR2 : Bool;   // 接收数据2
      TRCV_STATUS2 : Word;   // 接收数据2
      TRCV_RCVD_LEN2 : Word;   // 接收数据2
      TCON_DONE3 : Bool;
      TCON_BUSY3 : Bool;
      TCON_ERROR3 : Bool;
      TCON_STATUS3 : Word;
      TDISCON_DONE3 : Bool;
      TDISCON_BUSY3 : Bool;
      TDISCON_ERROR3 : Bool;
      TDISCON_STATUS3 : Word;
      TSEND_DONE3 : Bool;
      TSEND_BUSY3 : Bool;
      TSEND_ERROR3 : Bool;
      TSEND_STATUS3 : Word;
      TRCV_NDR3 : Bool;
      TRCV_BUSY3 : Bool;
      TRCV_ERROR3 : Bool;
      TRCV_STATUS3 : Word;
      TRCV_RCVD_LEN3 : Word;
   END_VAR
BEGIN
END_DATA_BLOCK

DATA_BLOCK "1#PLC交换PC_DB"   // DB33
{ S7_Optimized_Access := 'TRUE' }
VERSION : 0.1
// stored: InstanceOfName PLC交换PC
"PLC交换PC"
BEGIN
END_DATA_BLOCK

DATA_BLOCK "2#PLC交换PC_DB"   // DB34
{ S7_Optimized_Access := 'TRUE' }
VERSION : 0.1
// stored: InstanceOfName PLC交换PC
"PLC交换PC"
BEGIN
END_DATA_BLOCK

DATA_BLOCK "3#PLC交换PC_DB"   // DB35
{ S7_Optimized_Access := 'TRUE' }
VERSION : 0.1
// stored: InstanceOfName PLC交换PC
"PLC交换PC"
BEGIN
END_DATA_BLOCK

DATA_BLOCK "4#PLC交换PC_DB"   // DB36
{ S7_Optimized_Access := 'TRUE' }
VERSION : 0.1
// stored: InstanceOfName PLC交换PC
"PLC交换PC"
BEGIN
END_DATA_BLOCK

DATA_BLOCK "5#PLC交换PC_DB"   // DB44
{ S7_Optimized_Access := 'TRUE' }
VERSION : 0.1
// stored: InstanceOfName PLC交换PC
"PLC交换PC"
BEGIN
END_DATA_BLOCK

// folder: 通讯/射频通信/射频通信

DATA_BLOCK "SP通信79通信块"   // DB49
{ S7_Optimized_Access := 'TRUE' }
AUTHOR : SIMATIC
FAMILY : MC7Plus
NAME : TC_IP_v4
VERSION : 1.0
// stored: InstanceOfName TCON_IP_v4
"TCON_IP_v4"
BEGIN
   InterfaceId := 64;
   ID := 9;
   RemotePort := 32000;
   ActiveEstablished := true;
   RemoteAddress.ADDR[1] := 192;
   RemoteAddress.ADDR[2] := 168;
   RemoteAddress.ADDR[4] := 79;
END_DATA_BLOCK

DATA_BLOCK "SP通信80通信块"   // DB50
{ S7_Optimized_Access := 'TRUE' }
AUTHOR : SIMATIC
FAMILY : MC7Plus
NAME : TC_IP_v4
VERSION : 1.0
// stored: InstanceOfName TCON_IP_v4
"TCON_IP_v4"
BEGIN
   InterfaceId := 64;
   ID := 8;
   RemotePort := 32000;
   ActiveEstablished := true;
   RemoteAddress.ADDR[1] := 192;
   RemoteAddress.ADDR[2] := 168;
   RemoteAddress.ADDR[4] := 80;
END_DATA_BLOCK

DATA_BLOCK "SP通信81通信块"   // DB51
{ S7_Optimized_Access := 'TRUE' }
AUTHOR : SIMATIC
FAMILY : MC7Plus
NAME : TC_IP_v4
VERSION : 1.0
// stored: InstanceOfName TCON_IP_v4
"TCON_IP_v4"
BEGIN
   InterfaceId := 64;
   ID := 7;
   RemotePort := 32000;
   ActiveEstablished := true;
   RemoteAddress.ADDR[1] := 192;
   RemoteAddress.ADDR[2] := 168;
   RemoteAddress.ADDR[4] := 81;
END_DATA_BLOCK

DATA_BLOCK "库位编码值"   // DB53
{ S7_Optimized_Access := 'FALSE' }
VERSION : 0.1
   VAR
      IO1 : Array[0..5] of Byte;
      IO2 : Array[0..5] of Byte;
      IO3 : Array[0..5] of Byte;
      IO4 : Array[0..5] of Byte;
      IO5 : Array[0..5] of Byte;
      IO6 : Array[0..5] of Byte;
      IO7 : Array[0..5] of Byte;
      IO8 : Array[0..5] of Byte;
      IO9 : Array[0..5] of Byte;
      IO10 : Array[0..5] of Byte;
      IO11 : Array[0..5] of Byte;
      IO12 : Array[0..5] of Byte;
      IO13 : Array[0..5] of Byte;
      IO14 : Array[0..5] of Byte;
      IO15 : Array[0..5] of Byte;
      IO16 : Array[0..5] of Byte;
      KU1 : Byte;
      KU2 : Byte;
      KU3 : Byte;
      KU4 : Byte;
      KU5 : Byte;
      KU6 : Byte;
      KU7 : Byte;
      KU8 : Byte;
      KU9 : Byte;
      KU10 : Byte;
      KU11 : Byte;
      KU12 : Byte;
      KU13 : Byte;
      KU14 : Byte;
      KU15 : Byte;
      KU16 : Byte;
   END_VAR
BEGIN
END_DATA_BLOCK

DATA_BLOCK "射频读取切换_DB80"   // DB60
{ S7_Optimized_Access := 'FALSE' }
VERSION : 0.1
// stored: InstanceOfName F2射频读取切换功能块
"F2射频读取切换功能块"
BEGIN
END_DATA_BLOCK

DATA_BLOCK "射频读取切换_DB81"   // DB69
{ S7_Optimized_Access := 'FALSE' }
VERSION : 0.1
// stored: InstanceOfName F2射频读取切换功能块
"F2射频读取切换功能块"
BEGIN
END_DATA_BLOCK

DATA_BLOCK "DB通信数据块"   // DB76
{ S7_Optimized_Access := 'FALSE' }
VERSION : 0.1
   VAR
      发送清除指令_79 : Bool;
      发送读取指令_79 : Bool;
      发送读UID指令_79 : Bool;
      建立通讯_79 : Bool;
      中断通讯_79 : Bool;
      通讯建立_79 : Bool;
      发送完成_79 : Bool;
      发送清除指令_80 : Bool;
      发送读取指令_80 : Bool;
      发送读UID指令_80 : Bool;
      建立通讯_80 : Bool;
      中断通讯_80 : Bool;
      通讯建立_80 : Bool;
      发送完成_80 : Bool;
      发送清除指令_81 : Bool;
      发送读取指令_81 : Bool;
      发送读UID指令_81 : Bool;
      建立通讯_81 : Bool;
      中断通讯_81 : Bool;
      通讯建立_81 : Bool;
      发送完成_81 : Bool;
      发送清除指令_82 : Bool;
      发送读取指令_82 : Bool;
      发送读UID指令_82 : Bool;
      建立通讯_82 : Bool;
      中断通讯_82 : Bool;
      通讯建立_82 : Bool;
      发送完成_82 : Bool;
   END_VAR
BEGIN
END_DATA_BLOCK

DATA_BLOCK "PLC数据接收79"   // DB77
{ S7_Optimized_Access := 'FALSE' }
VERSION : 0.1
   VAR
      System : Array[0..7] of Byte;
      IO1_Sta : Array[0..15] of Bool;
      IO1 : Array[0..5] of Byte;
      IO1_1 : Array[0..27] of Byte;
      IO2_Sta : Array[0..15] of Bool;
      IO2 : Array[0..5] of Byte;
      IO2_1 : Array[0..27] of Byte;
      IO3_Sta : Array[0..15] of Bool;
      IO3 : Array[0..5] of Byte;
      IO3_1 : Array[0..27] of Byte;
      IO4_Sta : Array[0..15] of Bool;
      IO4 : Array[0..5] of Byte;
      IO4_1 : Array[0..27] of Byte;
   END_VAR
BEGIN
END_DATA_BLOCK

DATA_BLOCK "射频读取切换_DB79"   // DB78
{ S7_Optimized_Access := 'FALSE' }
VERSION : 0.1
// stored: InstanceOfName F2射频读取切换功能块
"F2射频读取切换功能块"
BEGIN
END_DATA_BLOCK

DATA_BLOCK "PLC发送配置信息"   // DB79
{ S7_Optimized_Access := 'FALSE' }
VERSION : 0.1
   VAR
      VAR1 : Byte := 16#01;
      VAR2 : Byte;
      VAR3 : Byte;
      VAR4 : Byte;
      VAR5 : Byte;
      VAR6 : Byte;
      VAR7 : Byte;
      VAR8 : Byte;
      VAR9 : Byte;
      VAR10 : Byte;
      VAR11 : Byte;
      VAR12 : Byte;
      VAR13 : Byte;
      VAR14 : Byte;
      VAR15 : Byte;
      VAR16 : Byte;
      VAR17 : Byte := 16#01;
      VAR18 : Byte := 16#0b;
      VAR19 : Byte := 16#C8;
      VAR20 : Byte := 16#04;
      VAR21 : Byte := 16#03;
      VAR22 : Byte;
      VAR23 : Byte;
      VAR24 : Byte;
      VAR25 : Byte := 16#02;
      VAR26 : Byte := 16#0b;
      VAR27 : Byte := 16#C8;
      VAR28 : Byte := 16#04;
      VAR29 : Byte := 16#03;
      VAR30 : Byte := 16#0;
      VAR31 : Byte := 16#0;
      VAR32 : Byte := 16#0;
      VAR33 : Byte := 16#03;
      VAR34 : Byte := 16#0b;
      VAR35 : Byte := 16#C8;
      VAR36 : Byte := 16#04;
      VAR37 : Byte := 16#03;
      VAR38 : Byte := 16#0;
      VAR39 : Byte := 16#0;
      VAR40 : Byte := 16#0;
      VAR41 : Byte := 16#04;
      VAR42 : Byte := 16#0b;
      VAR43 : Byte := 16#C8;
      VAR44 : Byte := 16#04;
      VAR45 : Byte := 16#03;
      VAR46 : Byte := 16#0;
      VAR47 : Byte := 16#0;
      VAR48 : Byte := 16#0;
   END_VAR
BEGIN
END_DATA_BLOCK

DATA_BLOCK "PLC发送读用户数据指令"   // DB80
{ S7_Optimized_Access := 'FALSE' }
VERSION : 0.1
   VAR
      System : Array[0..7] of Byte;
      IO1 : Array[0..35] of Byte;
      IO2 : Array[0..35] of Byte;
      IO3 : Array[0..35] of Byte;
      IO4 : Array[0..35] of Byte;
   END_VAR
BEGIN
   IO2[0] := 16#18;
   IO1[0] := 16#18;
   IO4[0] := 16#18;
   IO3[0] := 16#18;
   IO1[1] := 16#20;
   IO2[1] := 16#20;
   IO3[1] := 16#20;
   IO4[1] := 16#20;
   System[0] := 16#02;
END_DATA_BLOCK

DATA_BLOCK "PLC发送清除数据指令"   // DB85
{ S7_Optimized_Access := 'FALSE' }
VERSION : 0.1
   VAR
      System : Array[0..7] of Byte;
      IO1 : Array[0..35] of Byte;
      IO2 : Array[0..35] of Byte;
      IO3 : Array[0..35] of Byte;
      IO4 : Array[0..35] of Byte;
   END_VAR
BEGIN
   IO2[0] := 16#00;
   IO1[0] := 16#00;
   IO4[0] := 16#00;
   IO3[0] := 16#00;
   IO1[1] := 16#0;
   IO2[1] := 16#0;
   IO3[1] := 16#0;
   IO4[1] := 16#0;
   System[0] := 16#02;
END_DATA_BLOCK

DATA_BLOCK "射频读取切换_DB82"   // DB86
{ S7_Optimized_Access := 'FALSE' }
VERSION : 0.1
// stored: InstanceOfName F2射频读取切换功能块
"F2射频读取切换功能块"
BEGIN
END_DATA_BLOCK

DATA_BLOCK "PLC数据接收80"   // DB87
{ S7_Optimized_Access := 'FALSE' }
VERSION : 0.1
   VAR
      System : Array[0..7] of Byte;
      IO1_Sta : Array[0..15] of Bool;
      IO1 : Array[0..5] of Byte;
      IO1_1 : Array[0..27] of Byte;
      IO2_Sta : Array[0..15] of Bool;
      IO2 : Array[0..5] of Byte;
      IO2_1 : Array[0..27] of Byte;
      IO3_Sta : Array[0..15] of Bool;
      IO3 : Array[0..5] of Byte;
      IO3_1 : Array[0..27] of Byte;
      IO4_Sta : Array[0..15] of Bool;
      IO4 : Array[0..5] of Byte;
      IO4_1 : Array[0..27] of Byte;
   END_VAR
BEGIN
END_DATA_BLOCK

DATA_BLOCK "PLC数据接收81"   // DB88
{ S7_Optimized_Access := 'FALSE' }
VERSION : 0.1
   VAR
      System : Array[0..7] of Byte;
      IO1_Sta : Array[0..15] of Bool;
      IO1 : Array[0..5] of Byte;
      IO1_1 : Array[0..27] of Byte;
      IO2_Sta : Array[0..15] of Bool;
      IO2 : Array[0..5] of Byte;
      IO2_1 : Array[0..27] of Byte;
      IO3_Sta : Array[0..15] of Bool;
      IO3 : Array[0..5] of Byte;
      IO3_1 : Array[0..27] of Byte;
      IO4_Sta : Array[0..15] of Bool;
      IO4 : Array[0..5] of Byte;
      IO4_1 : Array[0..27] of Byte;
   END_VAR
BEGIN
END_DATA_BLOCK

DATA_BLOCK "PLC数据接收82"   // DB89
{ S7_Optimized_Access := 'FALSE' }
VERSION : 0.1
   VAR
      System : Array[0..7] of Byte;
      IO1_Sta : Array[0..15] of Bool;
      IO1 : Array[0..5] of Byte;
      IO1_1 : Array[0..27] of Byte;
      IO2_Sta : Array[0..15] of Bool;
      IO2 : Array[0..5] of Byte;
      IO2_1 : Array[0..27] of Byte;
      IO3_Sta : Array[0..15] of Bool;
      IO3 : Array[0..5] of Byte;
      IO3_1 : Array[0..27] of Byte;
      IO4_Sta : Array[0..15] of Bool;
      IO4 : Array[0..5] of Byte;
      IO4_1 : Array[0..27] of Byte;
   END_VAR
BEGIN
END_DATA_BLOCK

DATA_BLOCK "SP通信82通信块"   // DB90
{ S7_Optimized_Access := 'TRUE' }
AUTHOR : SIMATIC
FAMILY : MC7Plus
NAME : TC_IP_v4
VERSION : 1.0
// stored: InstanceOfName TCON_IP_v4
"TCON_IP_v4"
BEGIN
   InterfaceId := 64;
   ID := 6;
   RemotePort := 32000;
   ActiveEstablished := true;
   RemoteAddress.ADDR[1] := 192;
   RemoteAddress.ADDR[2] := 168;
   RemoteAddress.ADDR[4] := 82;
END_DATA_BLOCK

DATA_BLOCK "PLC发送读取UID指令"   // DB91
{ S7_Optimized_Access := 'FALSE' }
VERSION : 0.1
   VAR
      System : Array[0..7] of Byte;
      IO1 : Array[0..35] of Byte;
      IO2 : Array[0..35] of Byte;
      IO3 : Array[0..35] of Byte;
      IO4 : Array[0..35] of Byte;
   END_VAR
BEGIN
   IO2[0] := 16#28;
   IO1[0] := 16#28;
   IO4[0] := 16#28;
   IO3[0] := 16#28;
   IO1[1] := 16#0;
   IO2[1] := 16#0;
   IO3[1] := 16#0;
   IO4[1] := 16#0;
   System[0] := 16#02;
END_DATA_BLOCK

// folder: (top level)

ORGANIZATION_BLOCK "Main"   // OB1, LAD, ProgramCycle
TITLE = "Main Program Sweep (Cycle)"
{ S7_Optimized_Access := 'TRUE' }
VERSION : 0.1
   VAR_INPUT
      Initial_Call : Bool;   // Initial call of this OB
      Remanence : Bool;   // =True, if remanent data are available
   END_VAR
BEGIN

REGION Network 1: 调用1#手
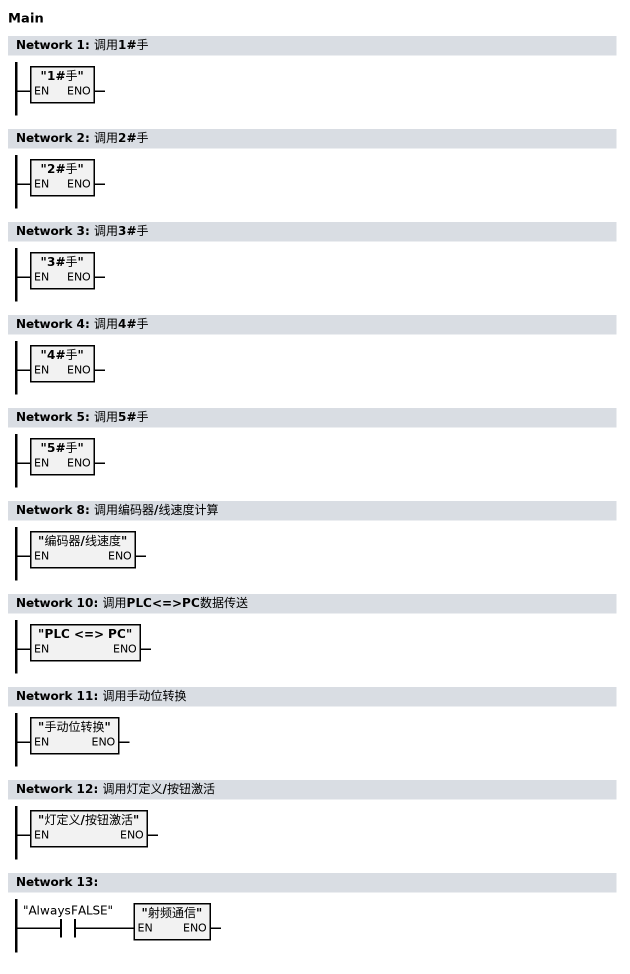
   RUNG wire#powerrail
      "1#手"()
   END_RUNG
   // the same network as SCL:
   "1#手"();
END_REGION

REGION Network 2: 调用2#手
   RUNG wire#powerrail
      "2#手"()
   END_RUNG
   // the same network as SCL:
   "2#手"();
END_REGION

REGION Network 3: 调用3#手
   RUNG wire#powerrail
      "3#手"()
   END_RUNG
   // the same network as SCL:
   "3#手"();
END_REGION

REGION Network 4: 调用4#手
   RUNG wire#powerrail
      "4#手"()
   END_RUNG
   // the same network as SCL:
   "4#手"();
END_REGION

REGION Network 5: 调用5#手
   RUNG wire#powerrail
      "5#手"()
   END_RUNG
   // the same network as SCL:
   "5#手"();
END_REGION

REGION Network 6: 调用6#手
END_REGION

REGION Network 7: 调用7#手
END_REGION

REGION Network 8: 调用编码器/线速度计算
   RUNG wire#powerrail
      "编码器/线速度"()
   END_RUNG
   // the same network as SCL:
   "编码器/线速度"();
END_REGION

REGION Network 9: 调用上位机通讯
END_REGION

REGION Network 10: 调用PLC<=>PC数据传送
   RUNG wire#powerrail
      "PLC <=> PC"()
   END_RUNG
   // the same network as SCL:
   "PLC <=> PC"();
END_REGION

REGION Network 11: 调用手动位转换
   RUNG wire#powerrail
      "手动位转换"()
   END_RUNG
   // the same network as SCL:
   "手动位转换"();
END_REGION

REGION Network 12: 调用灯定义/按钮激活
   RUNG wire#powerrail
      "灯定义/按钮激活"()
   END_RUNG
   // the same network as SCL:
   "灯定义/按钮激活"();
END_REGION

REGION Network 13
   RUNG wire#powerrail
      Contact( "AlwaysFALSE" )
      "射频通信"()
   END_RUNG
   // the same network as SCL:
   IF "AlwaysFALSE" THEN "射频通信"(); END_IF;
END_REGION
END_ORGANIZATION_BLOCK

ORGANIZATION_BLOCK "Cyclic interrupt_1"   // OB31, LAD, CyclicInterrupt
{ S7_Optimized_Access := 'TRUE' }
VERSION : 0.1
   VAR_INPUT
      Initial_Call : Bool;   // Initial call of this OB
      Event_Count : Int;   // Events discarded
   END_VAR
   VAR_TEMP   // added for the SCL form of the ladder/FBD networks
      _w1 : Bool;
   END_VAR
BEGIN

REGION Network 1
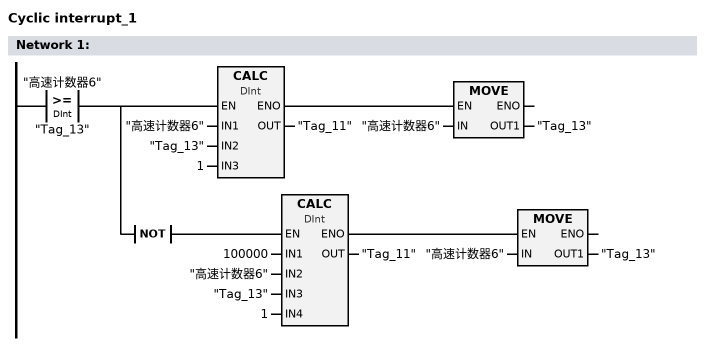
   #_w1 := "高速计数器6" >= "Tag_13";
   IF #_w1 THEN
       CALC(in1 := "高速计数器6", in2 := "Tag_13", in3 := 1, out => "Tag_11");
       "Tag_13" := "高速计数器6";
   END_IF;
   IF NOT #_w1 THEN
       CALC(in1 := 100000, in2 := "高速计数器6", in3 := "Tag_13", in4 := 1, out => "Tag_11");
       "Tag_13" := "高速计数器6";
   END_IF;
END_REGION
END_ORGANIZATION_BLOCK

ORGANIZATION_BLOCK "Rack or station failure"   // OB86, LAD, RackStationFailure
{ S7_Optimized_Access := 'TRUE' }
VERSION : 0.1
   VAR_INPUT
      LADDR : Hw_Io;   // Hardware identifier
      Event_Class : Byte;   // Event class
      Fault_ID : Byte;   // Fault identifier
   END_VAR
BEGIN
END_ORGANIZATION_BLOCK

ORGANIZATION_BLOCK "Startup"   // OB100, LAD, Startup
TITLE = "Complete Restart"
{ S7_Optimized_Access := 'TRUE' }
VERSION : 0.1
   VAR_INPUT
      LostRetentive : Bool;   // True if retentive data are lost
      LostRTC : Bool;   // True if date and time are lost
   END_VAR
BEGIN

REGION Network 1
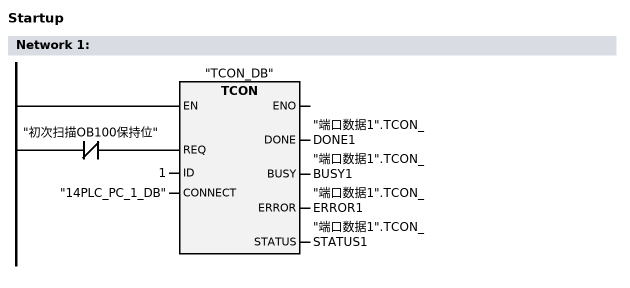
   "TCON_DB"(REQ := NOT "初次扫描OB100保持位",   // TCON
             ID := 1,
             CONNECT := "14PLC_PC_1_DB",
             DONE => "端口数据1".TCON_DONE1,
             BUSY => "端口数据1".TCON_BUSY1,
             ERROR => "端口数据1".TCON_ERROR1,
             STATUS => "端口数据1".TCON_STATUS1);
END_REGION
END_ORGANIZATION_BLOCK

// folder: 14工位

FUNCTION_BLOCK "库位动作流程"   // FB1, LAD
{ S7_Optimized_Access := 'TRUE' }
VERSION : 0.1
// 取砖流程    放砖流程  复位流程
   VAR_INPUT
      开始按钮 : Bool;
      停止按钮 : Bool;
      急停按钮 : Bool;
      复位按钮 : Bool;
      x轴定位接近1 : Bool;
      x轴定位接近2 : Bool;
      x轴减速光电 : Bool;
      X轴行程极限开关 : Bool;
      Z轴原点接近 : Bool;
      Z轴行程极限开关 : Bool;
      W轴原点接近 : Bool;
      W轴上砖待命位 : Bool;
      W轴运行停止位 : Bool;
      W轴吸取接近开关 : Bool;
      W轴吸取极限接近开关 : Bool;
      W轴行程极限开关 : Bool;
      W轴吸盘压力检测1 : Bool;
      W轴吸盘压力检测2 : Bool;
      W轴吸盘压力检测3 : Bool;
      W轴吸盘压力检测4 : Bool;
      A库位栈板检测 : Bool;
      A库位安全保护光电 : Bool;
      两A库间保护光电 : Bool;
      A库位启动按钮 : Bool;
      B库位栈板检测 : Bool;
      B库位安全保护光电 : Bool;
      两B库间保护光电 : Bool;
      B库位启动按钮 : Bool;
      上砖后正压打开时间 : Time;   // 放砖后正压打开时间定时器
      定位开关到位延时 : Time;   // x轴复位 定位开关到位延时
      "x轴复位 定位开关1无 定位开关2有延时" : Time;   // x轴复位 定位开关1无 定位开关2有 延时
      上砖取砖失败报警延时 : Time;   // 上砖取砖失败报警时间
      上砖去AB库取砖延时 : Time;   // 上砖去AB库取砖延时
      复位真空阀经时间后关闭延时 : Time;   // 复位流程真空阀经设定时间后关闭线圈
      皮带上方吸盘冲限位z轴上升时间 : Time;   // 皮带上方吸盘冲击限位z轴上升最大时间
      Z轴下降中途抱闸时间 : Time;   // Z轴下降中途抱闸时间
      "输送线上方停止按钮后 复位标志位时间" : Time;   // 输送线上方停止按钮后 复位标志位时间
      伺服停止后返回中间位延时 : Time;   // 伺服停止后返回中间位延时
      伺服库位放或取砖完成返回原点延时 : Time;   // 伺服电机库位放或取砖完成，返回原点位延时
      伺服同步线速延时输出时间 : Time;
      z轴下降抱闸延时打开时间 : Time;
      吸取到位稳定时间 : Time;
      机械手取放砖选择 : Byte;   // 机械手取放砖选择
      AB库抓取选择 : Bool;   // 1A库取放砖 2B库取放砖
      手动Z轴下降 : Bool;
      手动Z轴上升 : Bool;
      手动X轴2库移动 : Bool;
      手动X轴1库移动 : Bool;
      手动W轴前移 : Bool;
      手动W轴回原位 : Bool;
      手动吸盘电磁阀打开 : Bool;
      手动吸盘电磁阀关闭 : Bool;
      X轴变频器报警 : Bool;
      Z轴变频器报警 : Bool;
      W轴伺服报警 : Bool;
      输送线编码值抓取位置 : DInt;
      输送线编码器实时值 : DInt;
      Z轴编码器实时值 : DInt;
      Z轴待命位置编码值 : Int;
      机械手手自动标志 : Bool;
      Z轴高速转低速编码值 : DInt;
      X轴提前运行编码值 : DInt;
      机械手单独复位 : Bool;
      输送线变频器报警 : Bool;
      Z轴减速距离 : DInt;
      测试模式 : Bool;   // 1测试 2正常
      设备压力开关 : Bool;
      上位机状态 : Byte;
      "B#库满转" : Bool;
      "A#库满转" : Bool;
      取砖X轴提前下降设定值 : DInt;
      W轴伺服同步线速度值 : DInt;
      输送线启动 : Bool;
   END_VAR
   VAR_OUTPUT
      A库位启动按钮指示灯 : Bool;
      B库位启动按钮指示灯 : Bool;
      吸盘电磁阀打开 : Bool;
      吸盘电磁阀关闭 : Bool;
      x轴2库正转 : Bool;
      x轴1库反转 : Bool;
      x轴低速 : Bool;
      x轴抱闸 : Bool;
      z轴下降 : Bool;
      z轴上升 : Bool;
      z轴抱闸 : Bool;
      z轴1速 : Bool;
      z轴2速 : Bool;
      z轴3速 : Bool;
      "W轴伺服启动/停止" : Bool;
      W轴伺服速度模拟量 : Int;
      给上位机取砖成功寄存地址 : Bool;   // 给上位机发送取砖成功 1完成2未完成
      AB库给上位机发送放砖完成指令 : Bool;   // 给上位机发送放砖成功 1完成2未完成
      AB库放砖回原位完成给上位机发送完成指令 : Bool;   // 给上位机发送回原位成功 1完成2未完成
      放砖模式机械手放砖等待 : Bool;
      系统运行标志 : Bool;
      系统复位标志 : Bool;
      系统急停限位标志 : Bool;
      压力开关压力检测报警1 : Bool;
      压力开关压力检测报警2 : Bool;
      压力开关压力检测报警3 : Bool;
      压力开关压力检测报警4 : Bool;
      A库位安全光电报警 : Bool;
      B库位安全光电报警 : Bool;
      A库位安全光电报警toPC : Bool;
      B库位安全光电报警toPC : Bool;
      下砖周期标志位 : Bool;
      上砖周转标志位 : Bool;
      找待命位标志位 : Bool;
   END_VAR
   VAR
      下砖z轴待命位下降取砖 : Bool;
      z轴机械手取砖标志位 : Bool;
      z轴待命位置取砖到位中间变量 : Bool;
      下砖z轴抓取位置上升 : Bool;
      Z轴上升到位压力检测中间位 : Bool;
      吸盘压力开关检测 : Bool;
      真空阀打开标志位 : Bool;
      z轴取砖完成回待命位中间变量 : Bool;
      "X轴高速正转-待命位到2库" : Bool;   // 从待命位到A库
      x轴正转转低速中间变量 : Bool;
      "x轴正转转低速-待命位到2库" : Bool;
      x轴到达A库下方中间变量 : Bool;
      下砖z轴AB库位下降 : Bool;
      下砖z轴AB库位上升 : Bool;
      真空阀关闭标志位 : Bool;
      z轴A库上升到待命位中间变量 : Bool;
      x轴2库高速反转回工作位 : Bool;
      x轴A库回工作位转低速中间变量 : Bool;
      x轴2库回工作位反转转低速 : Bool;
      x轴A库回工作位到位中间变量 : Bool;
      x轴AB库回工作位完成标志位 : Bool;
      "X轴高速反转-待命位到1库" : Bool;
      "x轴反转转低速-待命位到1库" : Bool;
      x轴1库高速正转回工作位 : Bool;
      x轴1库回工作位正转转低速 : Bool;
      复位Z轴上升 : Bool;
      复位Z轴上升中间变量 : Bool;
      复位W轴回原位 : Bool;
      复位W轴回原位中间变量 : Bool;
      复位X轴回原位 : Bool;
      复位X轴回原位中间变量1 : Bool;
      复位X轴回原位中间变量2 : Bool;
      复位X轴经1库原点后回原位 : Bool;
      上砖X轴快速移动2库 : Bool;
      上砖X轴快速移动1库 : Bool;
      上砖x轴转低速中间变量1 : Bool;
      "上砖x轴正转转低速-待命位到2库" : Bool;
      "上砖x轴反转转低速-待命位到1库" : Bool;
      上砖x轴到达A库下方中间变量 : Bool;
      上砖z轴AB库位下降 : Bool;
      上砖z轴AB库置取砖到位中间变量 : Bool;
      上砖真空电磁阀打开 : Bool;
      上砖吸盘压力开关检测 : Bool;
      上砖Z轴取砖位置反转上升中间位 : Bool;
      上砖z轴AB库位位置上升 : Bool;
      上砖z轴取砖完成回待命位中间变量 : Bool;
      "上砖X轴高速反转2库-待命位" : Bool;
      "上砖X轴高速正转1库-待命位" : Bool;
      上砖x轴AB库回工作位转低速中间变量 : Bool;
      上砖x轴2库回工作位反转转低速 : Bool;
      上砖x轴1库回工作位正转转低速 : Bool;
      上砖x轴AB库回工作位到位中间变量 : Bool;
      上砖z轴待命位下降放砖 : Bool;
      上砖真空阀关闭标志位 : Bool;
      上抓z轴待命位下降到位中间变量 : Bool;
      上砖z轴待命位置上升 : Bool;
      上砖z轴待命位上升到位中间变量 : Bool;
      上砖设备放砖完成标志位 : Bool;
      设备报警标志位 : Bool;
      W轴待命位冲击限位处理 : Bool;
      设备启动标志位 : Bool;
      减速光电计数传送 : Word;
      X轴减速光电计数2次 : Bool;
      "2#库放砖标志位" : Bool;
      "1#库放砖标志位" : Bool;
      Z轴下降找待命位置 : Bool;
      z轴待命位正转下降取砖1 : Bool;
      Z轴上升找待命位置 : Bool;
      Z轴待命位置编码值范围 : DInt;
      z轴运行后不在找待命位 : Bool;
      输送线编码值抓取位置范围 : DInt;
      输送线编码值抓取位置范围超过5万 : DInt;
      X轴提前运行中间变量 : Bool;
      上砖z轴待命位下降放砖保持 : Bool;
      复位真空阀关闭 : Bool;
      Z轴下降中途抱闸标志位 : Bool;
      Z轴下降中途抱闸标志位上升沿 : Bool;
      Z轴下降中途抱闸编码值 : DInt;
      Z轴下降中途抱闸编码值范围 : DInt;
      吸盘压力开关检测上升沿 : Bool;
      X轴减速光电计数3次 : Bool;
      下砖Z轴提前下降中间变量 : Bool;
      下砖真空阀提前打开 : Bool;
      真空阀开上升沿 : Bool;   // 压力开关报警
      停止按钮记忆位 : Bool;
      停止按钮标志位 : Bool;
      A库光电报警SET位 : Bool;
      B库光电报警SET位 : Bool;
      上升沿_1 : Bool;
      上升沿_2 : Bool;
      上升沿_3 : Bool;
      X轴减速光电通断次数 : Int;
      下砖提前下降判断标志位 : Bool;
      Z轴上升转低速脉冲 : DInt;
      上砖切换W伺服去上砖位 : Bool;
      下砖切换W伺服回原位 : Bool;
      上位机发送自动就绪状态 : Bool;
      上下砖伺服同步线速度运行 : Bool;
      上下砖伺服返回下砖位置延时 : Bool;
      上下砖伺服返回下砖位置 : Bool;
      上下砖伺服回原点 : Bool;
      复位伺服回原点 : Bool;
      上砖正压打开时间定时器 : IEC_TIMER;
      下砖正压打开时间定时器 : IEC_TIMER;
      两定位开关到位延时定时器 : IEC_TIMER;
      x轴复位定位开关1无定位开关2有定时器 : IEC_TIMER;
      上砖取砖失败报警定时器 : IEC_TIMER;
      上砖去AB库取砖定时器 : IEC_TIMER;
      复位真空阀经设定时间关闭线圈定时器 : IEC_TIMER;
      皮带上吸盘冲限位z轴上升最大时间定时器 : IEC_TIMER;
      Z轴下降中途抱闸定时器 : IEC_TIMER;
      "输送线上停止按钮后 复位标志位定时器" : IEC_TIMER;
      伺服停止返回中间位定时器 : IEC_TIMER;
      "伺服库位放或取砖-返回原点定时器" : IEC_TIMER;
      伺服同步线速延时输出定时器 : IEC_TIMER;
      z轴下降抱闸打开延时定时器 : IEC_TIMER;
      周期时间定时器 : IEC_TIMER;
      下砖吸取接近稳定时间定时器 : IEC_TIMER;
      上砖吸取接近稳定时间定时器 : IEC_TIMER;
      上升沿 : Bool;
      上升沿_4 : Bool;
      上升沿_5 : Bool;
      上升沿_6 : Bool;
      上升沿_7 : Bool;
      上升沿_8 : Bool;
      上升沿_9 : Bool;
      上升沿_10 : Bool;
      上升沿_11 : Bool;
      上升沿_12 : Bool;
      上砖成功转换下砖模式标志位 : Bool;
      上砖成功转换下砖模式跳步标志位 : Bool;
      上砖z轴提前下降中间变量 : Bool;
      上砖提前下降判断标志位 : Bool;
      Z轴停止编码值 : DInt;
      Z轴停止编码值上限 : DInt;
      Z轴停止编码值下限 : DInt;
      周期时间定时器Q : Bool;
   END_VAR
   VAR_TEMP   // added for the SCL form of the ladder/FBD networks
      _w1 : Bool;
      _w2 : Bool;
      _w3 : Bool;
      _w4 : Bool;
      _w5 : Bool;
      _w6 : Bool;
      _w7 : Bool;
      _w8 : Bool;
      _w9 : Bool;
   END_VAR
BEGIN

REGION Network 1: PC改为手动模式 PC手动转换 机械手待命位置写自动写2 停止自动运行
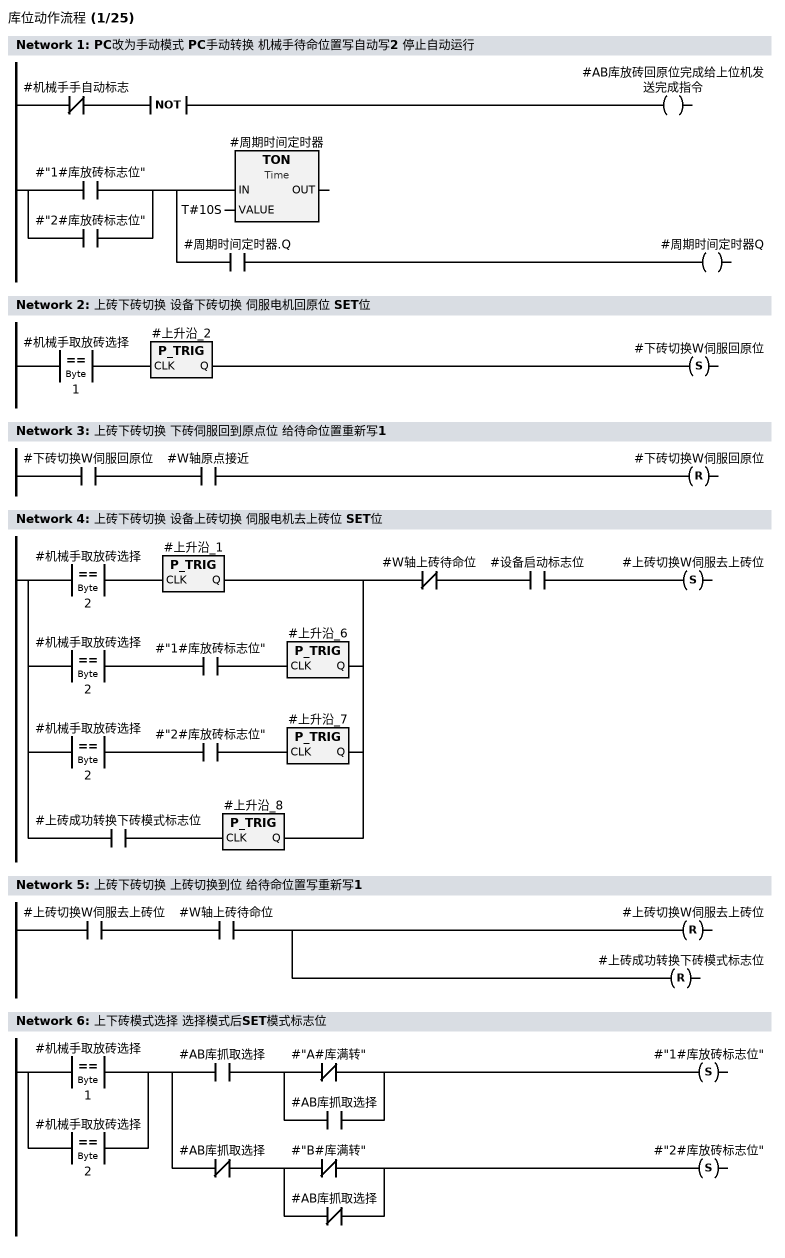
   #AB库放砖回原位完成给上位机发送完成指令 := NOT (NOT #机械手手自动标志);
   #_w1 := #"1#库放砖标志位" OR #"2#库放砖标志位";
   #周期时间定时器.TON(IN := #_w1, PT := T#10S);   // TON coil
   #周期时间定时器Q := #_w1 AND #周期时间定时器.Q;
END_REGION

REGION Network 2: 上砖下砖切换 设备下砖切换 伺服电机回原位 SET位
   RUNG wire#powerrail
      { S7_Templates := "SrcType := Byte" } EQ_Contact(in1 := #机械手取放砖选择, in2 := 1)
      P_Trig( #上升沿_2 )
      S_Coil( #下砖切换W伺服回原位 )
   END_RUNG
   // the same network as SCL:
   #_w1 := #机械手取放砖选择 = 1;
   #_w2 := #_w1 AND NOT #上升沿_2;   // rising edge
   #上升沿_2 := #_w1;
   IF #_w2 THEN #下砖切换W伺服回原位 := TRUE; END_IF;
END_REGION

REGION Network 3: 上砖下砖切换 下砖伺服回到原点位 给待命位置重新写1
   RUNG wire#powerrail
      Contact( #下砖切换W伺服回原位 )
      Contact( #W轴原点接近 )
      R_Coil( #下砖切换W伺服回原位 )
   END_RUNG
   // the same network as SCL:
   IF #下砖切换W伺服回原位 AND #W轴原点接近 THEN #下砖切换W伺服回原位 := FALSE; END_IF;
END_REGION

REGION Network 4: 上砖下砖切换 设备上砖切换 伺服电机去上砖位 SET位
   RUNG wire#powerrail
      { S7_Templates := "SrcType := Byte" } EQ_Contact(in1 := #机械手取放砖选择, in2 := 2)
      P_Trig( #上升沿_1 )
      wire#w1
      I_Contact( #W轴上砖待命位 )
      Contact( #设备启动标志位 )
      S_Coil( #上砖切换W伺服去上砖位 )
   END_RUNG
   RUNG wire#powerrail
      { S7_Templates := "SrcType := Byte" } EQ_Contact(in1 := #机械手取放砖选择, in2 := 2)
      Contact( #"1#库放砖标志位" )
      P_Trig( #上升沿_6 )
   END_RUNG wire#w1
   RUNG wire#powerrail
      { S7_Templates := "SrcType := Byte" } EQ_Contact(in1 := #机械手取放砖选择, in2 := 2)
      Contact( #"2#库放砖标志位" )
      P_Trig( #上升沿_7 )
   END_RUNG wire#w1
   RUNG wire#powerrail
      Contact( #上砖成功转换下砖模式标志位 )
      P_Trig( #上升沿_8 )
   END_RUNG wire#w1
   // the same network as SCL:
   #_w1 := #机械手取放砖选择 = 2;
   #_w2 := #_w1 AND NOT #上升沿_1;   // rising edge
   #上升沿_1 := #_w1;
   #_w3 := (#机械手取放砖选择 = 2) AND #"1#库放砖标志位";
   #_w4 := #_w3 AND NOT #上升沿_6;   // rising edge
   #上升沿_6 := #_w3;
   #_w5 := (#机械手取放砖选择 = 2) AND #"2#库放砖标志位";
   #_w6 := #_w5 AND NOT #上升沿_7;   // rising edge
   #上升沿_7 := #_w5;
   #_w7 := #上砖成功转换下砖模式标志位 AND NOT #上升沿_8;   // rising edge
   #上升沿_8 := #上砖成功转换下砖模式标志位;
   IF (#_w2 OR #_w4 OR #_w6 OR #_w7) AND NOT #W轴上砖待命位 AND #设备启动标志位 THEN #上砖切换W伺服去上砖位 := TRUE; END_IF;
END_REGION

REGION Network 5: 上砖下砖切换 上砖切换到位 给待命位置写重新写1
   RUNG wire#powerrail
      Contact( #上砖切换W伺服去上砖位 )
      Contact( #W轴上砖待命位 )
      wire#w1
      R_Coil( #上砖切换W伺服去上砖位 )
   END_RUNG
   RUNG wire#w1
      R_Coil( #上砖成功转换下砖模式标志位 )
   END_RUNG
   // the same network as SCL:
   #_w1 := #上砖切换W伺服去上砖位 AND #W轴上砖待命位;
   IF #_w1 THEN
       #上砖切换W伺服去上砖位 := FALSE;
       #上砖成功转换下砖模式标志位 := FALSE;
   END_IF;
END_REGION

REGION Network 6: 上下砖模式选择 选择模式后SET模式标志位
   RUNG wire#powerrail
      { S7_Templates := "SrcType := Byte" } EQ_Contact(in1 := #机械手取放砖选择, in2 := 1)
      wire#w1
      Contact( #AB库抓取选择 )
      wire#w2
      I_Contact( #"A#库满转" )
      wire#w3
      S_Coil( #"1#库放砖标志位" )
   END_RUNG
   RUNG wire#powerrail
      { S7_Templates := "SrcType := Byte" } EQ_Contact(in1 := #机械手取放砖选择, in2 := 2)
   END_RUNG wire#w1
   RUNG wire#w2
      Contact( #AB库抓取选择 )
   END_RUNG wire#w3
   RUNG wire#w1
      I_Contact( #AB库抓取选择 )
      wire#w4
      I_Contact( #"B#库满转" )
      wire#w5
      S_Coil( #"2#库放砖标志位" )
   END_RUNG
   RUNG wire#w4
      I_Contact( #AB库抓取选择 )
   END_RUNG wire#w5
   // the same network as SCL:
   #_w1 := (#机械手取放砖选择 = 1) OR (#机械手取放砖选择 = 2);
   IF #_w1 AND #AB库抓取选择 AND (NOT #"A#库满转" OR #AB库抓取选择) THEN #"1#库放砖标志位" := TRUE; END_IF;
   IF #_w1 AND NOT #AB库抓取选择 AND (NOT #"B#库满转" OR NOT #AB库抓取选择) THEN #"2#库放砖标志位" := TRUE; END_IF;
END_REGION

REGION Network 7: 设备上砖吸取成功，等待放砖， PC发指令回库位
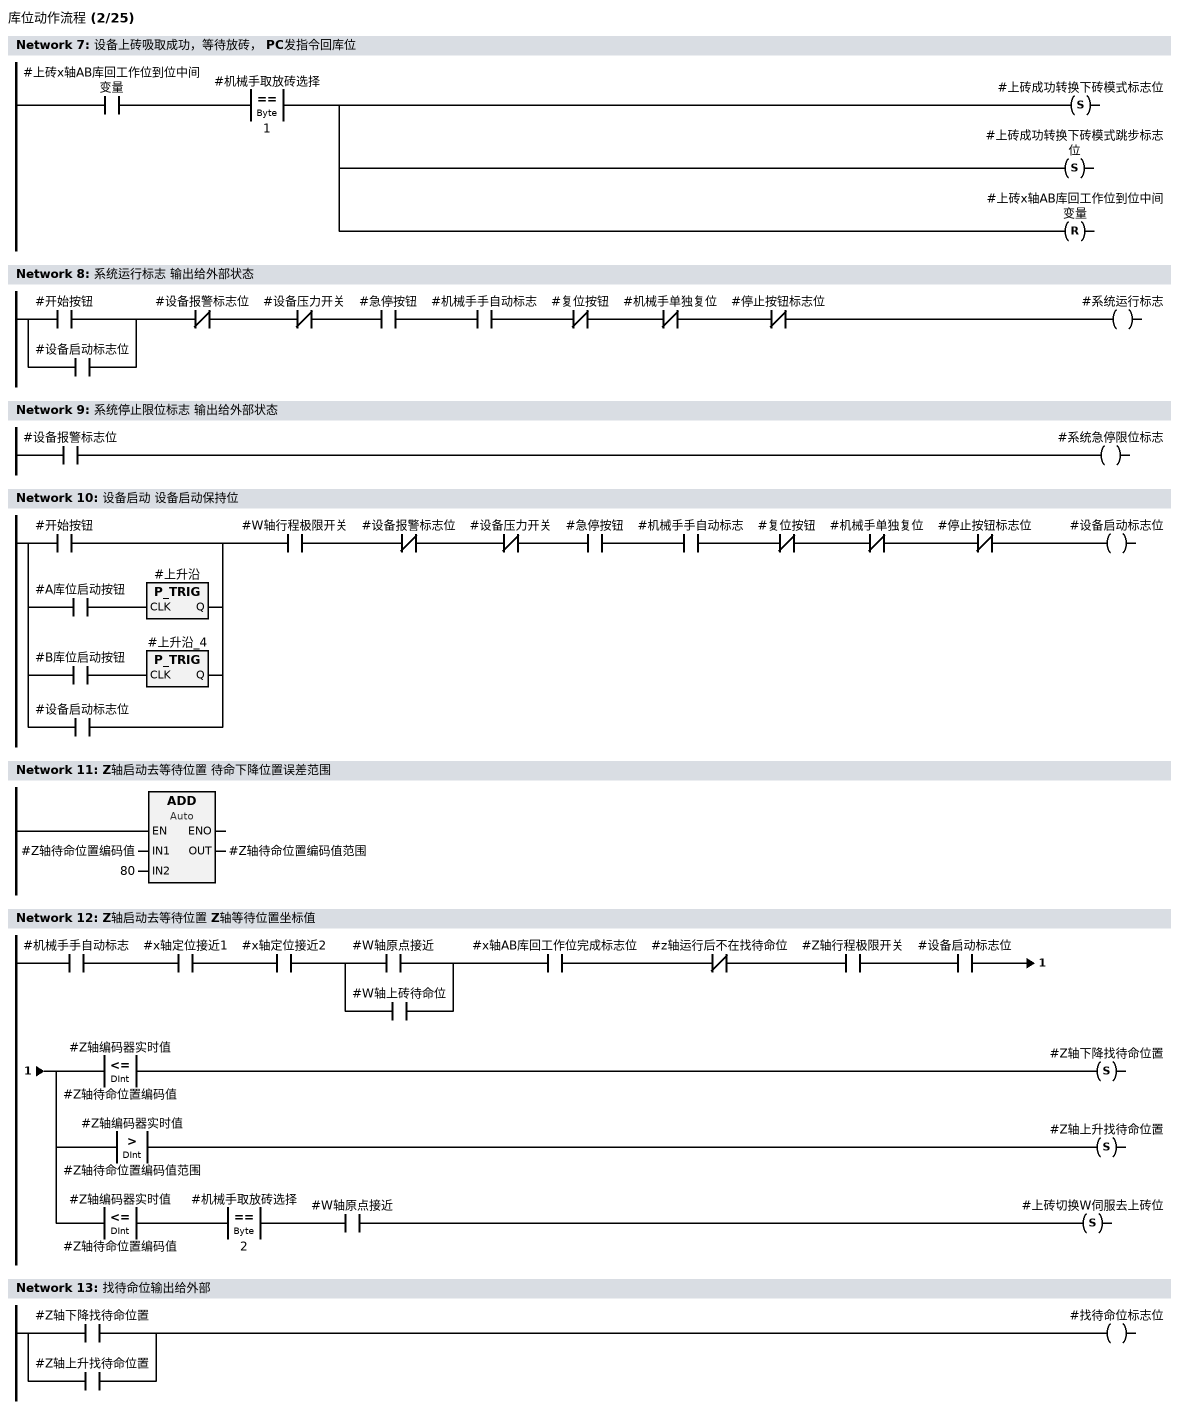
   RUNG wire#powerrail
      Contact( #上砖x轴AB库回工作位到位中间变量 )
      { S7_Templates := "SrcType := Byte" } EQ_Contact(in1 := #机械手取放砖选择, in2 := 1)
      wire#w1
      S_Coil( #上砖成功转换下砖模式标志位 )
   END_RUNG
   RUNG wire#w1
      S_Coil( #上砖成功转换下砖模式跳步标志位 )
   END_RUNG
   RUNG wire#w1
      R_Coil( #上砖x轴AB库回工作位到位中间变量 )
   END_RUNG
   // the same network as SCL:
   IF #上砖x轴AB库回工作位到位中间变量 AND (#机械手取放砖选择 = 1) THEN
       #上砖成功转换下砖模式标志位 := TRUE;
       #上砖成功转换下砖模式跳步标志位 := TRUE;
       #上砖x轴AB库回工作位到位中间变量 := FALSE;
   END_IF;
END_REGION

REGION Network 8: 系统运行标志 输出给外部状态
   RUNG wire#powerrail
      Contact( #开始按钮 )
      wire#w1
      I_Contact( #设备报警标志位 )
      I_Contact( #设备压力开关 )
      Contact( #急停按钮 )
      Contact( #机械手手自动标志 )
      I_Contact( #复位按钮 )
      I_Contact( #机械手单独复位 )
      I_Contact( #停止按钮标志位 )
      Coil( #系统运行标志 )
   END_RUNG
   RUNG wire#powerrail
      Contact( #设备启动标志位 )
   END_RUNG wire#w1
   // the same network as SCL:
   #系统运行标志 := (#开始按钮 OR #设备启动标志位) AND NOT #设备报警标志位 AND NOT #设备压力开关 AND #急停按钮 AND #机械手手自动标志 AND NOT #复位按钮 AND NOT #机械手单独复位 AND NOT #停止按钮标志位;
END_REGION

REGION Network 9: 系统停止限位标志 输出给外部状态
   RUNG wire#powerrail
      Contact( #设备报警标志位 )
      Coil( #系统急停限位标志 )
   END_RUNG
   // the same network as SCL:
   #系统急停限位标志 := #设备报警标志位;
END_REGION

REGION Network 10: 设备启动 设备启动保持位
   RUNG wire#powerrail
      Contact( #开始按钮 )
      wire#w1
      Contact( #W轴行程极限开关 )
      I_Contact( #设备报警标志位 )
      I_Contact( #设备压力开关 )
      Contact( #急停按钮 )
      Contact( #机械手手自动标志 )
      I_Contact( #复位按钮 )
      I_Contact( #机械手单独复位 )
      I_Contact( #停止按钮标志位 )
      Coil( #设备启动标志位 )
   END_RUNG
   RUNG wire#powerrail
      Contact( #A库位启动按钮 )
      P_Trig( #上升沿 )
   END_RUNG wire#w1
   RUNG wire#powerrail
      Contact( #B库位启动按钮 )
      P_Trig( #上升沿_4 )
   END_RUNG wire#w1
   RUNG wire#powerrail
      Contact( #设备启动标志位 )
   END_RUNG wire#w1
   // the same network as SCL:
   #_w1 := #A库位启动按钮 AND NOT #上升沿;   // rising edge
   #上升沿 := #A库位启动按钮;
   #_w2 := #B库位启动按钮 AND NOT #上升沿_4;   // rising edge
   #上升沿_4 := #B库位启动按钮;
   #设备启动标志位 := (#开始按钮 OR #_w1 OR #_w2 OR #设备启动标志位) AND #W轴行程极限开关 AND NOT #设备报警标志位 AND NOT #设备压力开关 AND #急停按钮 AND #机械手手自动标志 AND NOT #复位按钮 AND NOT #机械手单独复位 AND NOT #停止按钮标志位;
END_REGION

REGION Network 11: Z轴启动去等待位置 待命下降位置误差范围
   RUNG wire#powerrail
      Add(in1 := #Z轴待命位置编码值, in2 := 80, out => #Z轴待命位置编码值范围)
   END_RUNG
   // the same network as SCL:
   #Z轴待命位置编码值范围 := #Z轴待命位置编码值 + 80;
END_REGION

REGION Network 12: Z轴启动去等待位置 Z轴等待位置坐标值
   RUNG wire#powerrail
      Contact( #机械手手自动标志 )
      Contact( #x轴定位接近1 )
      Contact( #x轴定位接近2 )
      wire#w1
      Contact( #W轴原点接近 )
      wire#w2
      Contact( #x轴AB库回工作位完成标志位 )
      I_Contact( #z轴运行后不在找待命位 )
      Contact( #Z轴行程极限开关 )
      Contact( #设备启动标志位 )
      wire#w3
      { S7_Templates := "SrcType := DInt" } LE_Contact(in1 := #Z轴编码器实时值, in2 := #Z轴待命位置编码值)
      S_Coil( #Z轴下降找待命位置 )
   END_RUNG
   RUNG wire#w1
      Contact( #W轴上砖待命位 )
   END_RUNG wire#w2
   RUNG wire#w3
      { S7_Templates := "SrcType := DInt" } GT_Contact(in1 := #Z轴编码器实时值, in2 := #Z轴待命位置编码值范围)
      S_Coil( #Z轴上升找待命位置 )
   END_RUNG
   RUNG wire#w3
      { S7_Templates := "SrcType := DInt" } LE_Contact(in1 := #Z轴编码器实时值, in2 := #Z轴待命位置编码值)
      { S7_Templates := "SrcType := Byte" } EQ_Contact(in1 := #机械手取放砖选择, in2 := 2)
      Contact( #W轴原点接近 )
      S_Coil( #上砖切换W伺服去上砖位 )
   END_RUNG
   // the same network as SCL:
   #_w1 := #机械手手自动标志 AND #x轴定位接近1 AND #x轴定位接近2 AND (#W轴原点接近 OR #W轴上砖待命位) AND #x轴AB库回工作位完成标志位 AND NOT #z轴运行后不在找待命位 AND #Z轴行程极限开关 AND #设备启动标志位;
   IF #_w1 AND (#Z轴编码器实时值 <= #Z轴待命位置编码值) THEN #Z轴下降找待命位置 := TRUE; END_IF;
   IF #_w1 AND (#Z轴编码器实时值 > #Z轴待命位置编码值范围) THEN #Z轴上升找待命位置 := TRUE; END_IF;
   IF #_w1 AND (#Z轴编码器实时值 <= #Z轴待命位置编码值) AND (#机械手取放砖选择 = 2) AND #W轴原点接近 THEN #上砖切换W伺服去上砖位 := TRUE; END_IF;
END_REGION

REGION Network 13: 找待命位输出给外部
   RUNG wire#powerrail
      Contact( #Z轴下降找待命位置 )
      wire#w1
      Coil( #找待命位标志位 )
   END_RUNG
   RUNG wire#powerrail
      Contact( #Z轴上升找待命位置 )
   END_RUNG wire#w1
   // the same network as SCL:
   #找待命位标志位 := #Z轴下降找待命位置 OR #Z轴上升找待命位置;
END_REGION

REGION Network 14: Z轴启动去等待位置 复位待命位置下降
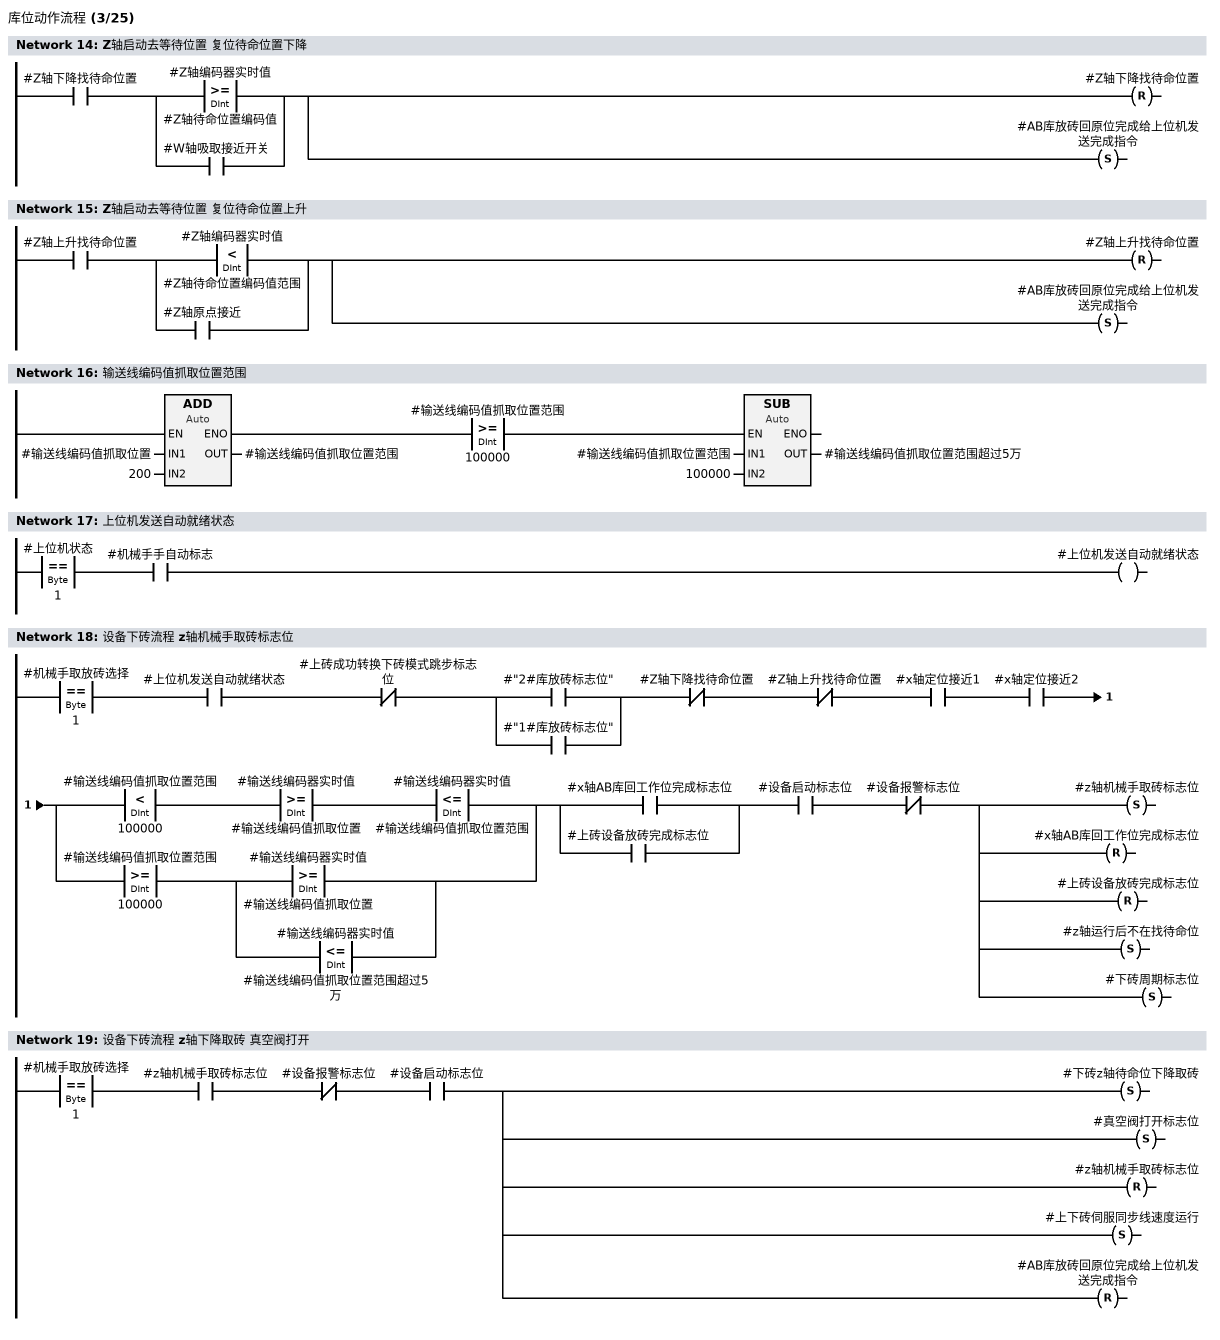
   RUNG wire#powerrail
      Contact( #Z轴下降找待命位置 )
      wire#w1
      { S7_Templates := "SrcType := DInt" } GE_Contact(in1 := #Z轴编码器实时值, in2 := #Z轴待命位置编码值)
      wire#w2
      R_Coil( #Z轴下降找待命位置 )
   END_RUNG
   RUNG wire#w1
      Contact( #W轴吸取接近开关 )
   END_RUNG wire#w2
   RUNG wire#w2
      S_Coil( #AB库放砖回原位完成给上位机发送完成指令 )
   END_RUNG
   // the same network as SCL:
   #_w1 := #Z轴下降找待命位置 AND ((#Z轴编码器实时值 >= #Z轴待命位置编码值) OR #W轴吸取接近开关);
   IF #_w1 THEN
       #Z轴下降找待命位置 := FALSE;
       #AB库放砖回原位完成给上位机发送完成指令 := TRUE;
   END_IF;
END_REGION

REGION Network 15: Z轴启动去等待位置 复位待命位置上升
   RUNG wire#powerrail
      Contact( #Z轴上升找待命位置 )
      wire#w1
      { S7_Templates := "SrcType := DInt" } LT_Contact(in1 := #Z轴编码器实时值, in2 := #Z轴待命位置编码值范围)
      wire#w2
      R_Coil( #Z轴上升找待命位置 )
   END_RUNG
   RUNG wire#w1
      Contact( #Z轴原点接近 )
   END_RUNG wire#w2
   RUNG wire#w2
      S_Coil( #AB库放砖回原位完成给上位机发送完成指令 )
   END_RUNG
   // the same network as SCL:
   #_w1 := #Z轴上升找待命位置 AND ((#Z轴编码器实时值 < #Z轴待命位置编码值范围) OR #Z轴原点接近);
   IF #_w1 THEN
       #Z轴上升找待命位置 := FALSE;
       #AB库放砖回原位完成给上位机发送完成指令 := TRUE;
   END_IF;
END_REGION

REGION Network 16: 输送线编码值抓取位置范围
   RUNG wire#powerrail
      Add(in1 := #输送线编码值抓取位置, in2 := 200, out => #输送线编码值抓取位置范围)
      { S7_Templates := "SrcType := DInt" } GE_Contact(in1 := #输送线编码值抓取位置范围, in2 := 100000)
      Sub(in1 := #输送线编码值抓取位置范围, in2 := 100000, out => #输送线编码值抓取位置范围超过5万)
   END_RUNG
   // the same network as SCL:
   #输送线编码值抓取位置范围 := #输送线编码值抓取位置 + 200;
   IF #输送线编码值抓取位置范围 >= 100000 THEN #输送线编码值抓取位置范围超过5万 := #输送线编码值抓取位置范围 - 100000; END_IF;
END_REGION

REGION Network 17: 上位机发送自动就绪状态
   RUNG wire#powerrail
      { S7_Templates := "SrcType := Byte" } EQ_Contact(in1 := #上位机状态, in2 := 1)
      Contact( #机械手手自动标志 )
      Coil( #上位机发送自动就绪状态 )
   END_RUNG
   // the same network as SCL:
   #上位机发送自动就绪状态 := (#上位机状态 = 1) AND #机械手手自动标志;
END_REGION

REGION Network 18: 设备下砖流程 z轴机械手取砖标志位
   RUNG wire#powerrail
      { S7_Templates := "SrcType := Byte" } EQ_Contact(in1 := #机械手取放砖选择, in2 := 1)
      Contact( #上位机发送自动就绪状态 )
      I_Contact( #上砖成功转换下砖模式跳步标志位 )
      wire#w1
      Contact( #"2#库放砖标志位" )
      wire#w2
      I_Contact( #Z轴下降找待命位置 )
      I_Contact( #Z轴上升找待命位置 )
      Contact( #x轴定位接近1 )
      Contact( #x轴定位接近2 )
      wire#w3
      { S7_Templates := "SrcType := DInt" } LT_Contact(in1 := #输送线编码值抓取位置范围, in2 := 100000)
      { S7_Templates := "SrcType := DInt" } GE_Contact(in1 := #输送线编码器实时值, in2 := #输送线编码值抓取位置)
      { S7_Templates := "SrcType := DInt" } LE_Contact(in1 := #输送线编码器实时值, in2 := #输送线编码值抓取位置范围)
      wire#w4
      Contact( #x轴AB库回工作位完成标志位 )
      wire#w6
      Contact( #设备启动标志位 )
      I_Contact( #设备报警标志位 )
      wire#w7
      S_Coil( #z轴机械手取砖标志位 )
   END_RUNG
   RUNG wire#w1
      Contact( #"1#库放砖标志位" )
   END_RUNG wire#w2
   RUNG wire#w3
      { S7_Templates := "SrcType := DInt" } GE_Contact(in1 := #输送线编码值抓取位置范围, in2 := 100000)
      wire#w5
      { S7_Templates := "SrcType := DInt" } GE_Contact(in1 := #输送线编码器实时值, in2 := #输送线编码值抓取位置)
   END_RUNG wire#w4
   RUNG wire#w5
      { S7_Templates := "SrcType := DInt" } LE_Contact(in1 := #输送线编码器实时值, in2 := #输送线编码值抓取位置范围超过5万)
   END_RUNG wire#w4
   RUNG wire#w4
      Contact( #上砖设备放砖完成标志位 )
   END_RUNG wire#w6
   RUNG wire#w7
      R_Coil( #x轴AB库回工作位完成标志位 )
   END_RUNG
   RUNG wire#w7
      R_Coil( #上砖设备放砖完成标志位 )
   END_RUNG
   RUNG wire#w7
      S_Coil( #z轴运行后不在找待命位 )
   END_RUNG
   RUNG wire#w7
      S_Coil( #下砖周期标志位 )
   END_RUNG
   // the same network as SCL:
   IF (#机械手取放砖选择 = 1) AND #上位机发送自动就绪状态 AND NOT #上砖成功转换下砖模式跳步标志位 AND (#"2#库放砖标志位" OR #"1#库放砖标志位") AND NOT #Z轴下降找待命位置 AND NOT #Z轴上升找待命位置 AND #x轴定位接近1 AND #x轴定位接近2 AND (((#输送线编码值抓取位置范围 < 100000) AND (#输送线编码器实时值 >= #输送线编码值抓取位置) AND (#输送线编码器实时值 <= #输送线编码值抓取位置范围)) OR ((#输送线编码值抓取位置范围 >= 100000) AND ((#输送线编码器实时值 >= #输送线编码值抓取位置) OR (#输送线编码器实时值 <= #输送线编码值抓取位置范围超过5万)))) AND (#x轴AB库回工作位完成标志位 OR #上砖设备放砖完成标志位) AND #设备启动标志位 AND NOT #设备报警标志位 THEN
       #z轴机械手取砖标志位 := TRUE;
   END_IF;
   #_w1 := (#机械手取放砖选择 = 1) AND #上位机发送自动就绪状态 AND NOT #上砖成功转换下砖模式跳步标志位 AND (#"2#库放砖标志位" OR #"1#库放砖标志位") AND NOT #Z轴下降找待命位置 AND NOT #Z轴上升找待命位置 AND #x轴定位接近1 AND #x轴定位接近2 AND (((#输送线编码值抓取位置范围 < 100000) AND (#输送线编码器实时值 >= #输送线编码值抓取位置) AND (#输送线编码器实时值 <= #输送线编码值抓取位置范围)) OR ((#输送线编码值抓取位置范围 >= 100000) AND ((#输送线编码器实时值 >= #输送线编码值抓取位置) OR (#输送线编码器实时值 <= #输送线编码值抓取位置范围超过5万)))) AND (#x轴AB库回工作位完成标志位 OR #上砖设备放砖完成标志位) AND #设备启动标志位 AND NOT #设备报警标志位;
   IF #_w1 THEN
       #x轴AB库回工作位完成标志位 := FALSE;
       #上砖设备放砖完成标志位 := FALSE;
       #z轴运行后不在找待命位 := TRUE;
       #下砖周期标志位 := TRUE;
   END_IF;
END_REGION

REGION Network 19: 设备下砖流程 z轴下降取砖 真空阀打开
   RUNG wire#powerrail
      { S7_Templates := "SrcType := Byte" } EQ_Contact(in1 := #机械手取放砖选择, in2 := 1)
      Contact( #z轴机械手取砖标志位 )
      I_Contact( #设备报警标志位 )
      Contact( #设备启动标志位 )
      wire#w1
      S_Coil( #下砖z轴待命位下降取砖 )
   END_RUNG
   RUNG wire#w1
      S_Coil( #真空阀打开标志位 )
   END_RUNG
   RUNG wire#w1
      R_Coil( #z轴机械手取砖标志位 )
   END_RUNG
   RUNG wire#w1
      S_Coil( #上下砖伺服同步线速度运行 )
   END_RUNG
   RUNG wire#w1
      R_Coil( #AB库放砖回原位完成给上位机发送完成指令 )
   END_RUNG
   // the same network as SCL:
   IF (#机械手取放砖选择 = 1) AND #z轴机械手取砖标志位 AND NOT #设备报警标志位 AND #设备启动标志位 THEN
       #下砖z轴待命位下降取砖 := TRUE;
       #真空阀打开标志位 := TRUE;
   END_IF;
   #_w1 := (#机械手取放砖选择 = 1) AND #z轴机械手取砖标志位 AND NOT #设备报警标志位 AND #设备启动标志位;
   IF #_w1 THEN
       #z轴机械手取砖标志位 := FALSE;
       #上下砖伺服同步线速度运行 := TRUE;
       #AB库放砖回原位完成给上位机发送完成指令 := FALSE;
   END_IF;
END_REGION

REGION Network 20: 设备下砖流程 到达取砖光电检测，Z轴停止
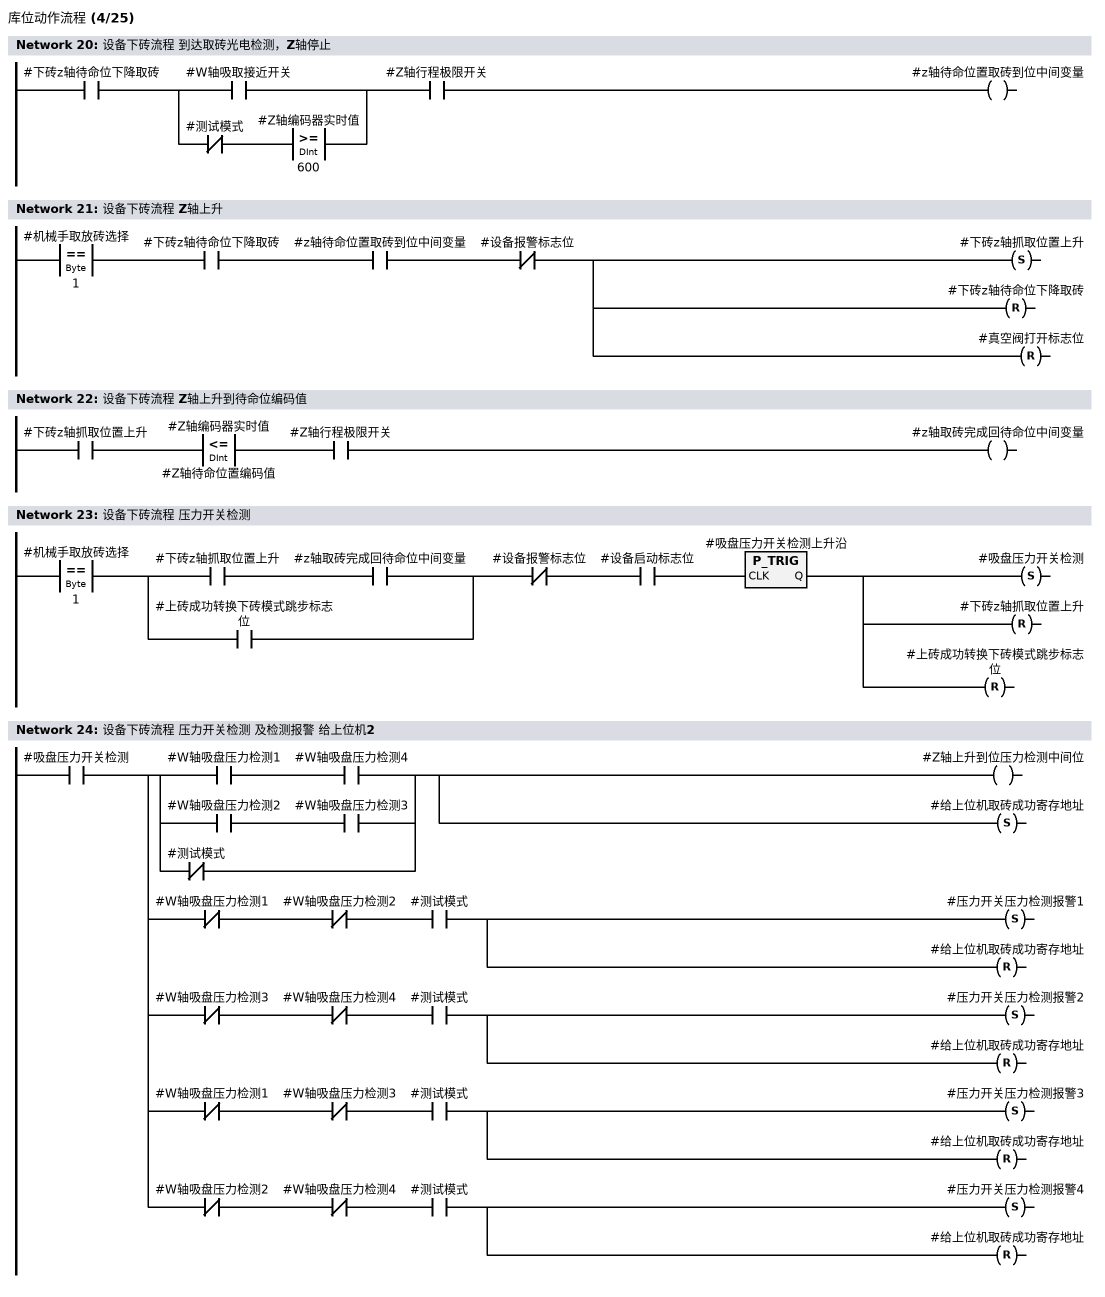
   RUNG wire#powerrail
      Contact( #下砖z轴待命位下降取砖 )
      wire#w1
      Contact( #W轴吸取接近开关 )
      wire#w2
      Contact( #Z轴行程极限开关 )
      Coil( #z轴待命位置取砖到位中间变量 )
   END_RUNG
   RUNG wire#w1
      I_Contact( #测试模式 )
      { S7_Templates := "SrcType := DInt" } GE_Contact(in1 := #Z轴编码器实时值, in2 := 600)
   END_RUNG wire#w2
   // the same network as SCL:
   #z轴待命位置取砖到位中间变量 := #下砖z轴待命位下降取砖 AND (#W轴吸取接近开关 OR (NOT #测试模式 AND (#Z轴编码器实时值 >= 600))) AND #Z轴行程极限开关;
END_REGION

REGION Network 21: 设备下砖流程 Z轴上升
   RUNG wire#powerrail
      { S7_Templates := "SrcType := Byte" } EQ_Contact(in1 := #机械手取放砖选择, in2 := 1)
      Contact( #下砖z轴待命位下降取砖 )
      Contact( #z轴待命位置取砖到位中间变量 )
      I_Contact( #设备报警标志位 )
      wire#w1
      S_Coil( #下砖z轴抓取位置上升 )
   END_RUNG
   RUNG wire#w1
      R_Coil( #下砖z轴待命位下降取砖 )
   END_RUNG
   RUNG wire#w1
      R_Coil( #真空阀打开标志位 )
   END_RUNG
   // the same network as SCL:
   IF (#机械手取放砖选择 = 1) AND #下砖z轴待命位下降取砖 AND #z轴待命位置取砖到位中间变量 AND NOT #设备报警标志位 THEN #下砖z轴抓取位置上升 := TRUE; END_IF;
   #_w1 := (#机械手取放砖选择 = 1) AND #下砖z轴待命位下降取砖 AND #z轴待命位置取砖到位中间变量 AND NOT #设备报警标志位;
   IF #_w1 THEN
       #下砖z轴待命位下降取砖 := FALSE;
       #真空阀打开标志位 := FALSE;
   END_IF;
END_REGION

REGION Network 22: 设备下砖流程 Z轴上升到待命位编码值
   RUNG wire#powerrail
      Contact( #下砖z轴抓取位置上升 )
      { S7_Templates := "SrcType := DInt" } LE_Contact(in1 := #Z轴编码器实时值, in2 := #Z轴待命位置编码值)
      Contact( #Z轴行程极限开关 )
      Coil( #z轴取砖完成回待命位中间变量 )
   END_RUNG
   // the same network as SCL:
   #z轴取砖完成回待命位中间变量 := #下砖z轴抓取位置上升 AND (#Z轴编码器实时值 <= #Z轴待命位置编码值) AND #Z轴行程极限开关;
END_REGION

REGION Network 23: 设备下砖流程 压力开关检测
   RUNG wire#powerrail
      { S7_Templates := "SrcType := Byte" } EQ_Contact(in1 := #机械手取放砖选择, in2 := 1)
      wire#w1
      Contact( #下砖z轴抓取位置上升 )
      Contact( #z轴取砖完成回待命位中间变量 )
      wire#w2
      I_Contact( #设备报警标志位 )
      Contact( #设备启动标志位 )
      P_Trig( #吸盘压力开关检测上升沿 )
      wire#w3
      S_Coil( #吸盘压力开关检测 )
   END_RUNG
   RUNG wire#w1
      Contact( #上砖成功转换下砖模式跳步标志位 )
   END_RUNG wire#w2
   RUNG wire#w3
      R_Coil( #下砖z轴抓取位置上升 )
   END_RUNG
   RUNG wire#w3
      R_Coil( #上砖成功转换下砖模式跳步标志位 )
   END_RUNG
   // the same network as SCL:
   #_w1 := (#机械手取放砖选择 = 1) AND ((#下砖z轴抓取位置上升 AND #z轴取砖完成回待命位中间变量) OR #上砖成功转换下砖模式跳步标志位) AND NOT #设备报警标志位 AND #设备启动标志位;
   #_w2 := #_w1 AND NOT #吸盘压力开关检测上升沿;   // rising edge
   #吸盘压力开关检测上升沿 := #_w1;
   IF #_w2 THEN
       #吸盘压力开关检测 := TRUE;
       #下砖z轴抓取位置上升 := FALSE;
       #上砖成功转换下砖模式跳步标志位 := FALSE;
   END_IF;
END_REGION

REGION Network 24: 设备下砖流程 压力开关检测 及检测报警 给上位机2
   RUNG wire#powerrail
      Contact( #吸盘压力开关检测 )
      wire#w1
      Contact( #W轴吸盘压力检测1 )
      Contact( #W轴吸盘压力检测4 )
      wire#w2
      Coil( #Z轴上升到位压力检测中间位 )
   END_RUNG
   RUNG wire#w1
      Contact( #W轴吸盘压力检测2 )
      Contact( #W轴吸盘压力检测3 )
   END_RUNG wire#w2
   RUNG wire#w1
      I_Contact( #测试模式 )
   END_RUNG wire#w2
   RUNG wire#w2
      S_Coil( #给上位机取砖成功寄存地址 )
   END_RUNG
   RUNG wire#w1
      I_Contact( #W轴吸盘压力检测1 )
      I_Contact( #W轴吸盘压力检测2 )
      Contact( #测试模式 )
      wire#w3
      S_Coil( #压力开关压力检测报警1 )
   END_RUNG
   RUNG wire#w3
      R_Coil( #给上位机取砖成功寄存地址 )
   END_RUNG
   RUNG wire#w1
      I_Contact( #W轴吸盘压力检测3 )
      I_Contact( #W轴吸盘压力检测4 )
      Contact( #测试模式 )
      wire#w4
      S_Coil( #压力开关压力检测报警2 )
   END_RUNG
   RUNG wire#w4
      R_Coil( #给上位机取砖成功寄存地址 )
   END_RUNG
   RUNG wire#w1
      I_Contact( #W轴吸盘压力检测1 )
      I_Contact( #W轴吸盘压力检测3 )
      Contact( #测试模式 )
      wire#w5
      S_Coil( #压力开关压力检测报警3 )
   END_RUNG
   RUNG wire#w5
      R_Coil( #给上位机取砖成功寄存地址 )
   END_RUNG
   RUNG wire#w1
      I_Contact( #W轴吸盘压力检测2 )
      I_Contact( #W轴吸盘压力检测4 )
      Contact( #测试模式 )
      wire#w6
      S_Coil( #压力开关压力检测报警4 )
   END_RUNG
   RUNG wire#w6
      R_Coil( #给上位机取砖成功寄存地址 )
   END_RUNG
   // the same network as SCL:
   #Z轴上升到位压力检测中间位 := #吸盘压力开关检测 AND ((#W轴吸盘压力检测1 AND #W轴吸盘压力检测4) OR (#W轴吸盘压力检测2 AND #W轴吸盘压力检测3) OR NOT #测试模式);
   IF #Z轴上升到位压力检测中间位 THEN #给上位机取砖成功寄存地址 := TRUE; END_IF;
   IF #吸盘压力开关检测 AND NOT #W轴吸盘压力检测1 AND NOT #W轴吸盘压力检测2 AND #测试模式 THEN
       #压力开关压力检测报警1 := TRUE;
       #给上位机取砖成功寄存地址 := FALSE;
   END_IF;
   IF #吸盘压力开关检测 AND NOT #W轴吸盘压力检测3 AND NOT #W轴吸盘压力检测4 AND #测试模式 THEN
       #压力开关压力检测报警2 := TRUE;
       #给上位机取砖成功寄存地址 := FALSE;
   END_IF;
   IF #吸盘压力开关检测 AND NOT #W轴吸盘压力检测1 AND NOT #W轴吸盘压力检测3 AND #测试模式 THEN
       #压力开关压力检测报警3 := TRUE;
       #给上位机取砖成功寄存地址 := FALSE;
   END_IF;
   IF #吸盘压力开关检测 AND NOT #W轴吸盘压力检测2 AND NOT #W轴吸盘压力检测4 AND #测试模式 THEN
       #压力开关压力检测报警4 := TRUE;
       #给上位机取砖成功寄存地址 := FALSE;
   END_IF;
END_REGION

REGION Network 25: 设备下砖流程 X轴正转高速A库 X轴反转高速B库
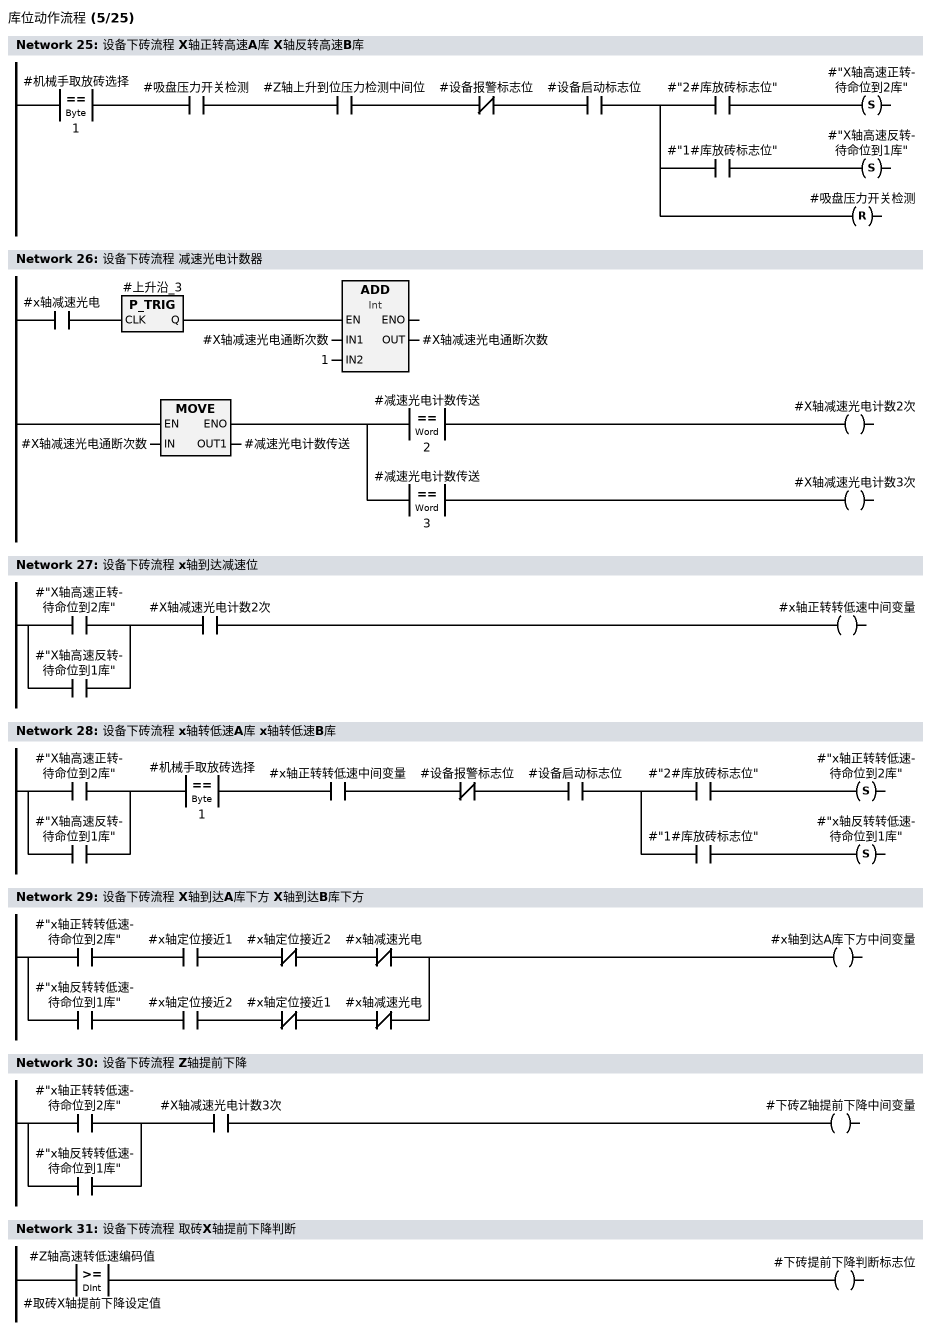
   RUNG wire#powerrail
      { S7_Templates := "SrcType := Byte" } EQ_Contact(in1 := #机械手取放砖选择, in2 := 1)
      Contact( #吸盘压力开关检测 )
      Contact( #Z轴上升到位压力检测中间位 )
      I_Contact( #设备报警标志位 )
      Contact( #设备启动标志位 )
      wire#w1
      Contact( #"2#库放砖标志位" )
      S_Coil( #"X轴高速正转-待命位到2库" )
   END_RUNG
   RUNG wire#w1
      Contact( #"1#库放砖标志位" )
      S_Coil( #"X轴高速反转-待命位到1库" )
   END_RUNG
   RUNG wire#w1
      R_Coil( #吸盘压力开关检测 )
   END_RUNG
   // the same network as SCL:
   #_w1 := (#机械手取放砖选择 = 1) AND #吸盘压力开关检测 AND #Z轴上升到位压力检测中间位 AND NOT #设备报警标志位 AND #设备启动标志位;
   IF #_w1 AND #"2#库放砖标志位" THEN #"X轴高速正转-待命位到2库" := TRUE; END_IF;
   IF #_w1 AND #"1#库放砖标志位" THEN #"X轴高速反转-待命位到1库" := TRUE; END_IF;
   IF #_w1 THEN #吸盘压力开关检测 := FALSE; END_IF;
END_REGION

REGION Network 26: 设备下砖流程 减速光电计数器
   RUNG wire#powerrail
      Contact( #x轴减速光电 )
      P_Trig( #上升沿_3 )
      { S7_Templates := "SrcType := Int" } Add(in1 := #X轴减速光电通断次数, in2 := 1, out => #X轴减速光电通断次数)
   END_RUNG
   RUNG wire#powerrail
      Move(in := #X轴减速光电通断次数, out1 => #减速光电计数传送)
      wire#w1
      { S7_Templates := "SrcType := Word" } EQ_Contact(in1 := #减速光电计数传送, in2 := 2)
      Coil( #X轴减速光电计数2次 )
   END_RUNG
   RUNG wire#w1
      { S7_Templates := "SrcType := Word" } EQ_Contact(in1 := #减速光电计数传送, in2 := 3)
      Coil( #X轴减速光电计数3次 )
   END_RUNG
   // the same network as SCL:
   #_w1 := #x轴减速光电 AND NOT #上升沿_3;   // rising edge
   #上升沿_3 := #x轴减速光电;
   IF #_w1 THEN #X轴减速光电通断次数 := #X轴减速光电通断次数 + 1; END_IF;
   #减速光电计数传送 := #X轴减速光电通断次数;
   #X轴减速光电计数2次 := #减速光电计数传送 = 2;
   #X轴减速光电计数3次 := #减速光电计数传送 = 3;
END_REGION

REGION Network 27: 设备下砖流程 x轴到达减速位
   RUNG wire#powerrail
      Contact( #"X轴高速正转-待命位到2库" )
      wire#w1
      Contact( #X轴减速光电计数2次 )
      Coil( #x轴正转转低速中间变量 )
   END_RUNG
   RUNG wire#powerrail
      Contact( #"X轴高速反转-待命位到1库" )
   END_RUNG wire#w1
   // the same network as SCL:
   #x轴正转转低速中间变量 := (#"X轴高速正转-待命位到2库" OR #"X轴高速反转-待命位到1库") AND #X轴减速光电计数2次;
END_REGION

REGION Network 28: 设备下砖流程 x轴转低速A库 x轴转低速B库
   RUNG wire#powerrail
      Contact( #"X轴高速正转-待命位到2库" )
      wire#w1
      { S7_Templates := "SrcType := Byte" } EQ_Contact(in1 := #机械手取放砖选择, in2 := 1)
      Contact( #x轴正转转低速中间变量 )
      I_Contact( #设备报警标志位 )
      Contact( #设备启动标志位 )
      wire#w2
      Contact( #"2#库放砖标志位" )
      S_Coil( #"x轴正转转低速-待命位到2库" )
   END_RUNG
   RUNG wire#powerrail
      Contact( #"X轴高速反转-待命位到1库" )
   END_RUNG wire#w1
   RUNG wire#w2
      Contact( #"1#库放砖标志位" )
      S_Coil( #"x轴反转转低速-待命位到1库" )
   END_RUNG
   // the same network as SCL:
   #_w1 := (#"X轴高速正转-待命位到2库" OR #"X轴高速反转-待命位到1库") AND (#机械手取放砖选择 = 1) AND #x轴正转转低速中间变量 AND NOT #设备报警标志位 AND #设备启动标志位;
   IF #_w1 AND #"2#库放砖标志位" THEN #"x轴正转转低速-待命位到2库" := TRUE; END_IF;
   IF #_w1 AND #"1#库放砖标志位" THEN #"x轴反转转低速-待命位到1库" := TRUE; END_IF;
END_REGION

REGION Network 29: 设备下砖流程 X轴到达A库下方 X轴到达B库下方
   RUNG wire#powerrail
      Contact( #"x轴正转转低速-待命位到2库" )
      Contact( #x轴定位接近1 )
      I_Contact( #x轴定位接近2 )
      I_Contact( #x轴减速光电 )
      wire#w1
      Coil( #x轴到达A库下方中间变量 )
   END_RUNG
   RUNG wire#powerrail
      Contact( #"x轴反转转低速-待命位到1库" )
      Contact( #x轴定位接近2 )
      I_Contact( #x轴定位接近1 )
      I_Contact( #x轴减速光电 )
   END_RUNG wire#w1
   // the same network as SCL:
   #x轴到达A库下方中间变量 := (#"x轴正转转低速-待命位到2库" AND #x轴定位接近1 AND NOT #x轴定位接近2 AND NOT #x轴减速光电) OR (#"x轴反转转低速-待命位到1库" AND #x轴定位接近2 AND NOT #x轴定位接近1 AND NOT #x轴减速光电);
END_REGION

REGION Network 30: 设备下砖流程 Z轴提前下降
   RUNG wire#powerrail
      Contact( #"x轴正转转低速-待命位到2库" )
      wire#w1
      Contact( #X轴减速光电计数3次 )
      Coil( #下砖Z轴提前下降中间变量 )
   END_RUNG
   RUNG wire#powerrail
      Contact( #"x轴反转转低速-待命位到1库" )
   END_RUNG wire#w1
   // the same network as SCL:
   #下砖Z轴提前下降中间变量 := (#"x轴正转转低速-待命位到2库" OR #"x轴反转转低速-待命位到1库") AND #X轴减速光电计数3次;
END_REGION

REGION Network 31: 设备下砖流程 取砖X轴提前下降判断
   RUNG wire#powerrail
      { S7_Templates := "SrcType := DInt" } GE_Contact(in1 := #Z轴高速转低速编码值, in2 := #取砖X轴提前下降设定值)
      Coil( #下砖提前下降判断标志位 )
   END_RUNG
   // the same network as SCL:
   #下砖提前下降判断标志位 := #Z轴高速转低速编码值 >= #取砖X轴提前下降设定值;
END_REGION

REGION Network 32: 设备下砖流程 Z轴提前下降
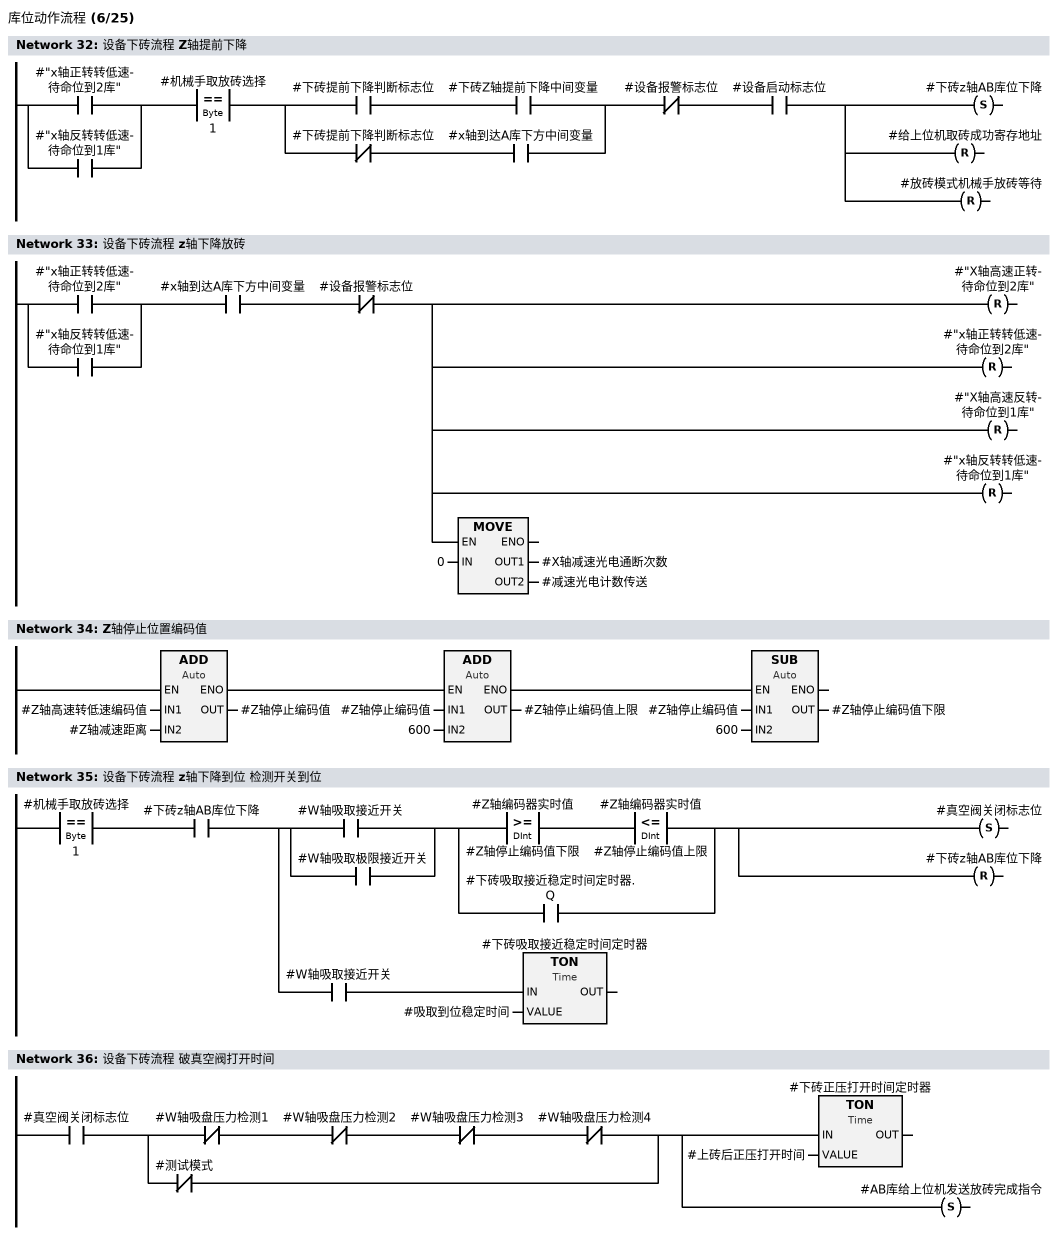
   RUNG wire#powerrail
      Contact( #"x轴正转转低速-待命位到2库" )
      wire#w1
      { S7_Templates := "SrcType := Byte" } EQ_Contact(in1 := #机械手取放砖选择, in2 := 1)
      wire#w2
      Contact( #下砖提前下降判断标志位 )
      Contact( #下砖Z轴提前下降中间变量 )
      wire#w3
      I_Contact( #设备报警标志位 )
      Contact( #设备启动标志位 )
      wire#w4
      S_Coil( #下砖z轴AB库位下降 )
   END_RUNG
   RUNG wire#powerrail
      Contact( #"x轴反转转低速-待命位到1库" )
   END_RUNG wire#w1
   RUNG wire#w2
      I_Contact( #下砖提前下降判断标志位 )
      Contact( #x轴到达A库下方中间变量 )
   END_RUNG wire#w3
   RUNG wire#w4
      R_Coil( #给上位机取砖成功寄存地址 )
   END_RUNG
   RUNG wire#w4
      R_Coil( #放砖模式机械手放砖等待 )
   END_RUNG
   // the same network as SCL:
   IF (#"x轴正转转低速-待命位到2库" OR #"x轴反转转低速-待命位到1库") AND (#机械手取放砖选择 = 1) AND ((#下砖提前下降判断标志位 AND #下砖Z轴提前下降中间变量) OR (NOT #下砖提前下降判断标志位 AND #x轴到达A库下方中间变量)) AND NOT #设备报警标志位 AND #设备启动标志位 THEN
       #下砖z轴AB库位下降 := TRUE;
       #给上位机取砖成功寄存地址 := FALSE;
       #放砖模式机械手放砖等待 := FALSE;
   END_IF;
END_REGION

REGION Network 33: 设备下砖流程 z轴下降放砖
   RUNG wire#powerrail
      Contact( #"x轴正转转低速-待命位到2库" )
      wire#w1
      Contact( #x轴到达A库下方中间变量 )
      I_Contact( #设备报警标志位 )
      wire#w2
      R_Coil( #"X轴高速正转-待命位到2库" )
   END_RUNG
   RUNG wire#powerrail
      Contact( #"x轴反转转低速-待命位到1库" )
   END_RUNG wire#w1
   RUNG wire#w2
      R_Coil( #"x轴正转转低速-待命位到2库" )
   END_RUNG
   RUNG wire#w2
      R_Coil( #"X轴高速反转-待命位到1库" )
   END_RUNG
   RUNG wire#w2
      R_Coil( #"x轴反转转低速-待命位到1库" )
   END_RUNG
   RUNG wire#w2
      Move(in := 0, out1 => #X轴减速光电通断次数, out2 => #减速光电计数传送)
   END_RUNG
   // the same network as SCL:
   IF (#"x轴正转转低速-待命位到2库" OR #"x轴反转转低速-待命位到1库") AND #x轴到达A库下方中间变量 AND NOT #设备报警标志位 THEN
       #"X轴高速正转-待命位到2库" := FALSE;
   END_IF;
   #_w1 := (#"x轴正转转低速-待命位到2库" OR #"x轴反转转低速-待命位到1库") AND #x轴到达A库下方中间变量 AND NOT #设备报警标志位;
   IF #_w1 THEN
       #"x轴正转转低速-待命位到2库" := FALSE;
       #"X轴高速反转-待命位到1库" := FALSE;
       #"x轴反转转低速-待命位到1库" := FALSE;
       #X轴减速光电通断次数 := 0;
       #减速光电计数传送 := 0;
   END_IF;
END_REGION

REGION Network 34: Z轴停止位置编码值
   RUNG wire#powerrail
      Add(in1 := #Z轴高速转低速编码值, in2 := #Z轴减速距离, out => #Z轴停止编码值)
      Add(in1 := #Z轴停止编码值, in2 := 600, out => #Z轴停止编码值上限)
      Sub(in1 := #Z轴停止编码值, in2 := 600, out => #Z轴停止编码值下限)
   END_RUNG
   // the same network as SCL:
   #Z轴停止编码值 := #Z轴高速转低速编码值 + #Z轴减速距离;
   #Z轴停止编码值上限 := #Z轴停止编码值 + 600;
   #Z轴停止编码值下限 := #Z轴停止编码值 - 600;
END_REGION

REGION Network 35: 设备下砖流程 z轴下降到位 检测开关到位
   #_w1 := (#机械手取放砖选择 = 1) AND #下砖z轴AB库位下降;
   IF #_w1 AND (#W轴吸取接近开关 OR #W轴吸取极限接近开关) AND (((#Z轴编码器实时值 >= #Z轴停止编码值下限) AND (#Z轴编码器实时值 <= #Z轴停止编码值上限)) OR #下砖吸取接近稳定时间定时器.Q) THEN
       #真空阀关闭标志位 := TRUE;
       #下砖z轴AB库位下降 := FALSE;
   END_IF;
   #下砖吸取接近稳定时间定时器.TON(IN := #_w1 AND #W轴吸取接近开关, PT := #吸取到位稳定时间);   // TON coil
END_REGION

REGION Network 36: 设备下砖流程 破真空阀打开时间
   #_w1 := #真空阀关闭标志位 AND ((NOT #W轴吸盘压力检测1 AND NOT #W轴吸盘压力检测2 AND NOT #W轴吸盘压力检测3 AND NOT #W轴吸盘压力检测4) OR NOT #测试模式);
   #下砖正压打开时间定时器.TON(IN := #_w1, PT := #上砖后正压打开时间);   // TON coil
   IF #_w1 THEN #AB库给上位机发送放砖完成指令 := TRUE; END_IF;
END_REGION

REGION Network 37: 设备下砖流程 A库放砖完成，给上位机发送放砖完成指令，Z轴上升
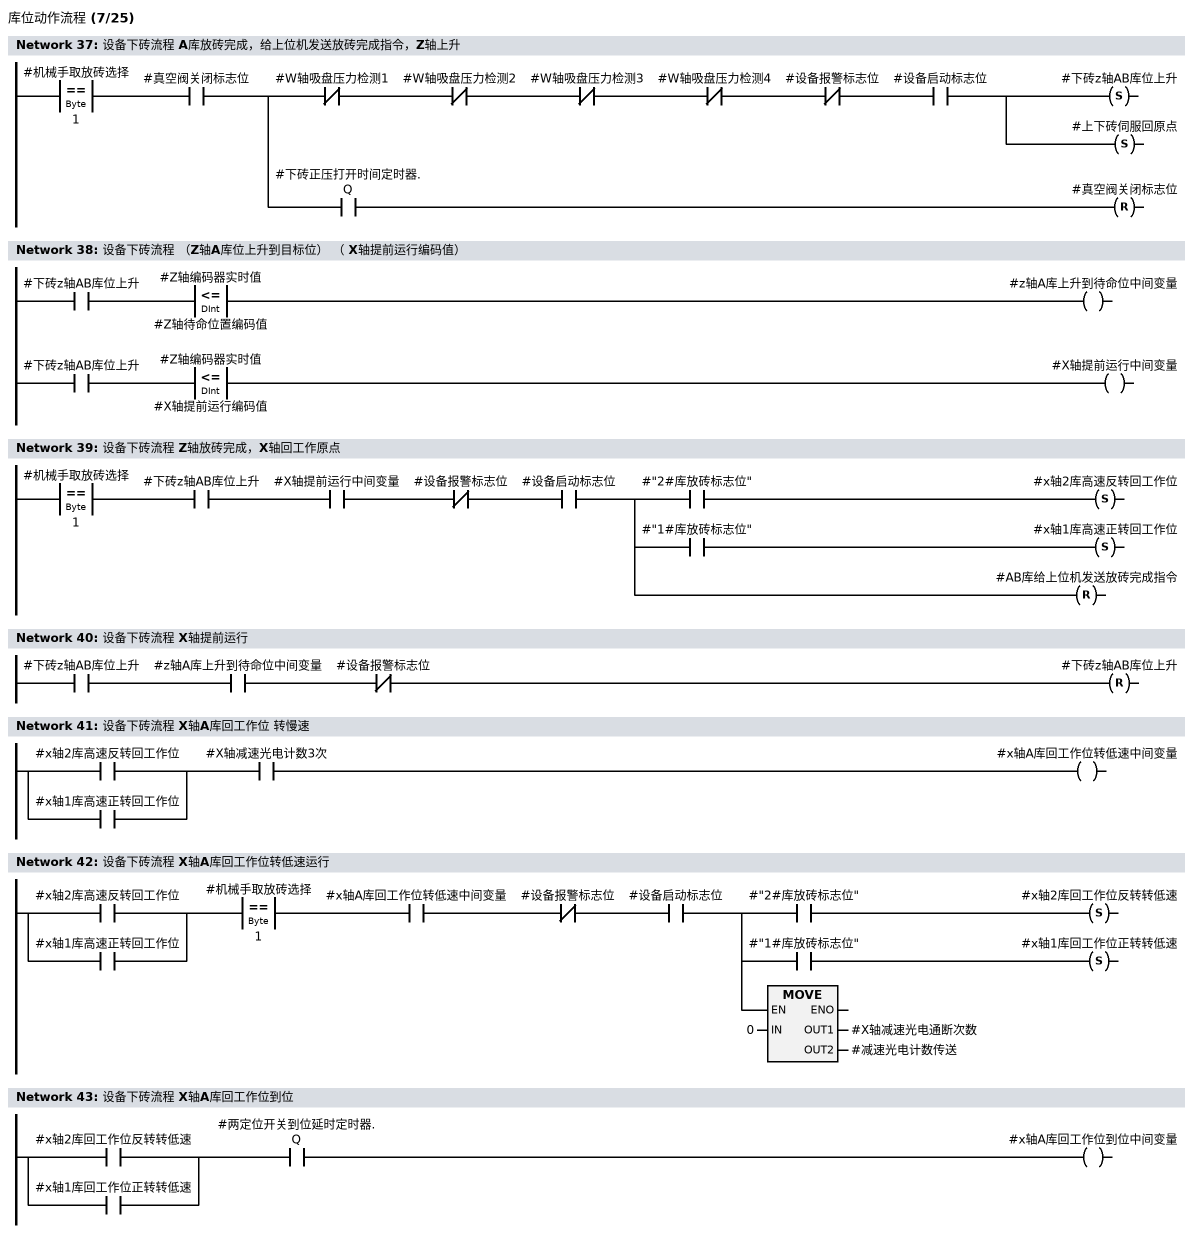
   RUNG wire#powerrail
      { S7_Templates := "SrcType := Byte" } EQ_Contact(in1 := #机械手取放砖选择, in2 := 1)
      Contact( #真空阀关闭标志位 )
      wire#w1
      I_Contact( #W轴吸盘压力检测1 )
      I_Contact( #W轴吸盘压力检测2 )
      I_Contact( #W轴吸盘压力检测3 )
      I_Contact( #W轴吸盘压力检测4 )
      I_Contact( #设备报警标志位 )
      Contact( #设备启动标志位 )
      wire#w2
      S_Coil( #下砖z轴AB库位上升 )
   END_RUNG
   RUNG wire#w2
      S_Coil( #上下砖伺服回原点 )
   END_RUNG
   RUNG wire#w1
      Contact( #下砖正压打开时间定时器.Q )
      R_Coil( #真空阀关闭标志位 )
   END_RUNG
   // the same network as SCL:
   #_w1 := (#机械手取放砖选择 = 1) AND #真空阀关闭标志位;
   IF #_w1 AND NOT #W轴吸盘压力检测1 AND NOT #W轴吸盘压力检测2 AND NOT #W轴吸盘压力检测3 AND NOT #W轴吸盘压力检测4 AND NOT #设备报警标志位 AND #设备启动标志位 THEN
       #下砖z轴AB库位上升 := TRUE;
       #上下砖伺服回原点 := TRUE;
   END_IF;
   IF #_w1 AND #下砖正压打开时间定时器.Q THEN #真空阀关闭标志位 := FALSE; END_IF;
END_REGION

REGION Network 38: 设备下砖流程 （Z轴A库位上升到目标位） （ X轴提前运行编码值）
   RUNG wire#powerrail
      Contact( #下砖z轴AB库位上升 )
      { S7_Templates := "SrcType := DInt" } LE_Contact(in1 := #Z轴编码器实时值, in2 := #Z轴待命位置编码值)
      Coil( #z轴A库上升到待命位中间变量 )
   END_RUNG
   RUNG wire#powerrail
      Contact( #下砖z轴AB库位上升 )
      { S7_Templates := "SrcType := DInt" } LE_Contact(in1 := #Z轴编码器实时值, in2 := #X轴提前运行编码值)
      Coil( #X轴提前运行中间变量 )
   END_RUNG
   // the same network as SCL:
   #z轴A库上升到待命位中间变量 := #下砖z轴AB库位上升 AND (#Z轴编码器实时值 <= #Z轴待命位置编码值);
   #X轴提前运行中间变量 := #下砖z轴AB库位上升 AND (#Z轴编码器实时值 <= #X轴提前运行编码值);
END_REGION

REGION Network 39: 设备下砖流程 Z轴放砖完成，X轴回工作原点
   RUNG wire#powerrail
      { S7_Templates := "SrcType := Byte" } EQ_Contact(in1 := #机械手取放砖选择, in2 := 1)
      Contact( #下砖z轴AB库位上升 )
      Contact( #X轴提前运行中间变量 )
      I_Contact( #设备报警标志位 )
      Contact( #设备启动标志位 )
      wire#w1
      Contact( #"2#库放砖标志位" )
      S_Coil( #x轴2库高速反转回工作位 )
   END_RUNG
   RUNG wire#w1
      Contact( #"1#库放砖标志位" )
      S_Coil( #x轴1库高速正转回工作位 )
   END_RUNG
   RUNG wire#w1
      R_Coil( #AB库给上位机发送放砖完成指令 )
   END_RUNG
   // the same network as SCL:
   #_w1 := (#机械手取放砖选择 = 1) AND #下砖z轴AB库位上升 AND #X轴提前运行中间变量 AND NOT #设备报警标志位 AND #设备启动标志位;
   IF #_w1 AND #"2#库放砖标志位" THEN #x轴2库高速反转回工作位 := TRUE; END_IF;
   IF #_w1 AND #"1#库放砖标志位" THEN #x轴1库高速正转回工作位 := TRUE; END_IF;
   IF #_w1 THEN #AB库给上位机发送放砖完成指令 := FALSE; END_IF;
END_REGION

REGION Network 40: 设备下砖流程 X轴提前运行
   RUNG wire#powerrail
      Contact( #下砖z轴AB库位上升 )
      Contact( #z轴A库上升到待命位中间变量 )
      I_Contact( #设备报警标志位 )
      R_Coil( #下砖z轴AB库位上升 )
   END_RUNG
   // the same network as SCL:
   IF #下砖z轴AB库位上升 AND #z轴A库上升到待命位中间变量 AND NOT #设备报警标志位 THEN #下砖z轴AB库位上升 := FALSE; END_IF;
END_REGION

REGION Network 41: 设备下砖流程 X轴A库回工作位 转慢速
   RUNG wire#powerrail
      Contact( #x轴2库高速反转回工作位 )
      wire#w1
      Contact( #X轴减速光电计数3次 )
      Coil( #x轴A库回工作位转低速中间变量 )
   END_RUNG
   RUNG wire#powerrail
      Contact( #x轴1库高速正转回工作位 )
   END_RUNG wire#w1
   // the same network as SCL:
   #x轴A库回工作位转低速中间变量 := (#x轴2库高速反转回工作位 OR #x轴1库高速正转回工作位) AND #X轴减速光电计数3次;
END_REGION

REGION Network 42: 设备下砖流程 X轴A库回工作位转低速运行
   RUNG wire#powerrail
      Contact( #x轴2库高速反转回工作位 )
      wire#w1
      { S7_Templates := "SrcType := Byte" } EQ_Contact(in1 := #机械手取放砖选择, in2 := 1)
      Contact( #x轴A库回工作位转低速中间变量 )
      I_Contact( #设备报警标志位 )
      Contact( #设备启动标志位 )
      wire#w2
      Contact( #"2#库放砖标志位" )
      S_Coil( #x轴2库回工作位反转转低速 )
   END_RUNG
   RUNG wire#powerrail
      Contact( #x轴1库高速正转回工作位 )
   END_RUNG wire#w1
   RUNG wire#w2
      Contact( #"1#库放砖标志位" )
      S_Coil( #x轴1库回工作位正转转低速 )
   END_RUNG
   RUNG wire#w2
      Move(in := 0, out1 => #X轴减速光电通断次数, out2 => #减速光电计数传送)
   END_RUNG
   // the same network as SCL:
   #_w1 := (#x轴2库高速反转回工作位 OR #x轴1库高速正转回工作位) AND (#机械手取放砖选择 = 1) AND #x轴A库回工作位转低速中间变量 AND NOT #设备报警标志位 AND #设备启动标志位;
   IF #_w1 AND #"2#库放砖标志位" THEN #x轴2库回工作位反转转低速 := TRUE; END_IF;
   IF #_w1 AND #"1#库放砖标志位" THEN #x轴1库回工作位正转转低速 := TRUE; END_IF;
   IF #_w1 THEN
       #X轴减速光电通断次数 := 0;
       #减速光电计数传送 := 0;
   END_IF;
END_REGION

REGION Network 43: 设备下砖流程 X轴A库回工作位到位
   RUNG wire#powerrail
      Contact( #x轴2库回工作位反转转低速 )
      wire#w1
      Contact( #两定位开关到位延时定时器.Q )
      Coil( #x轴A库回工作位到位中间变量 )
   END_RUNG
   RUNG wire#powerrail
      Contact( #x轴1库回工作位正转转低速 )
   END_RUNG wire#w1
   // the same network as SCL:
   #x轴A库回工作位到位中间变量 := (#x轴2库回工作位反转转低速 OR #x轴1库回工作位正转转低速) AND #两定位开关到位延时定时器.Q;
END_REGION

REGION Network 44: 设备下砖流程 X轴A库回工作位完成标志 给上位机发送“1”回原位完成指令
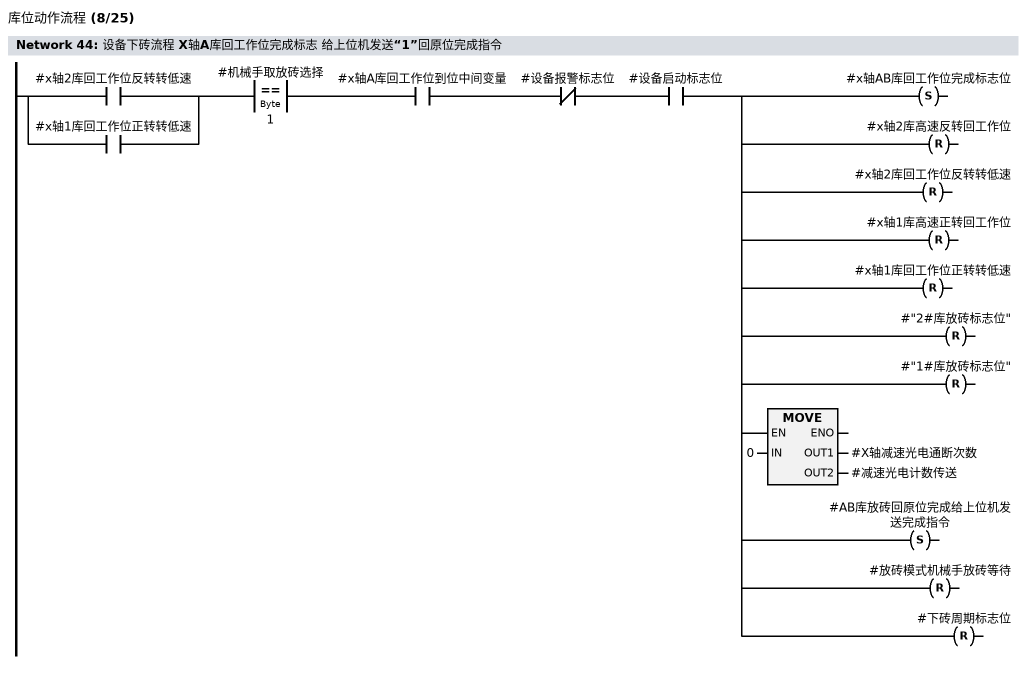
   RUNG wire#powerrail
      Contact( #x轴2库回工作位反转转低速 )
      wire#w1
      { S7_Templates := "SrcType := Byte" } EQ_Contact(in1 := #机械手取放砖选择, in2 := 1)
      Contact( #x轴A库回工作位到位中间变量 )
      I_Contact( #设备报警标志位 )
      Contact( #设备启动标志位 )
      wire#w2
      S_Coil( #x轴AB库回工作位完成标志位 )
   END_RUNG
   RUNG wire#powerrail
      Contact( #x轴1库回工作位正转转低速 )
   END_RUNG wire#w1
   RUNG wire#w2
      R_Coil( #x轴2库高速反转回工作位 )
   END_RUNG
   RUNG wire#w2
      R_Coil( #x轴2库回工作位反转转低速 )
   END_RUNG
   RUNG wire#w2
      R_Coil( #x轴1库高速正转回工作位 )
   END_RUNG
   RUNG wire#w2
      R_Coil( #x轴1库回工作位正转转低速 )
   END_RUNG
   RUNG wire#w2
      R_Coil( #"2#库放砖标志位" )
   END_RUNG
   RUNG wire#w2
      R_Coil( #"1#库放砖标志位" )
   END_RUNG
   RUNG wire#w2
      Move(in := 0, out1 => #X轴减速光电通断次数, out2 => #减速光电计数传送)
   END_RUNG
   RUNG wire#w2
      S_Coil( #AB库放砖回原位完成给上位机发送完成指令 )
   END_RUNG
   RUNG wire#w2
      R_Coil( #放砖模式机械手放砖等待 )
   END_RUNG
   RUNG wire#w2
      R_Coil( #下砖周期标志位 )
   END_RUNG
   // the same network as SCL:
   IF (#x轴2库回工作位反转转低速 OR #x轴1库回工作位正转转低速) AND (#机械手取放砖选择 = 1) AND #x轴A库回工作位到位中间变量 AND NOT #设备报警标志位 AND #设备启动标志位 THEN
       #x轴AB库回工作位完成标志位 := TRUE;
       #x轴2库高速反转回工作位 := FALSE;
   END_IF;
   #_w1 := (#x轴2库回工作位反转转低速 OR #x轴1库回工作位正转转低速) AND (#机械手取放砖选择 = 1) AND #x轴A库回工作位到位中间变量 AND NOT #设备报警标志位 AND #设备启动标志位;
   IF #_w1 THEN
       #x轴2库回工作位反转转低速 := FALSE;
       #x轴1库高速正转回工作位 := FALSE;
       #x轴1库回工作位正转转低速 := FALSE;
       #"2#库放砖标志位" := FALSE;
       #"1#库放砖标志位" := FALSE;
       #X轴减速光电通断次数 := 0;
       #减速光电计数传送 := 0;
       #AB库放砖回原位完成给上位机发送完成指令 := TRUE;
       #放砖模式机械手放砖等待 := FALSE;
       #下砖周期标志位 := FALSE;
   END_IF;
END_REGION

REGION Network 46: 设备上砖流程 X轴快速往AB库取砖
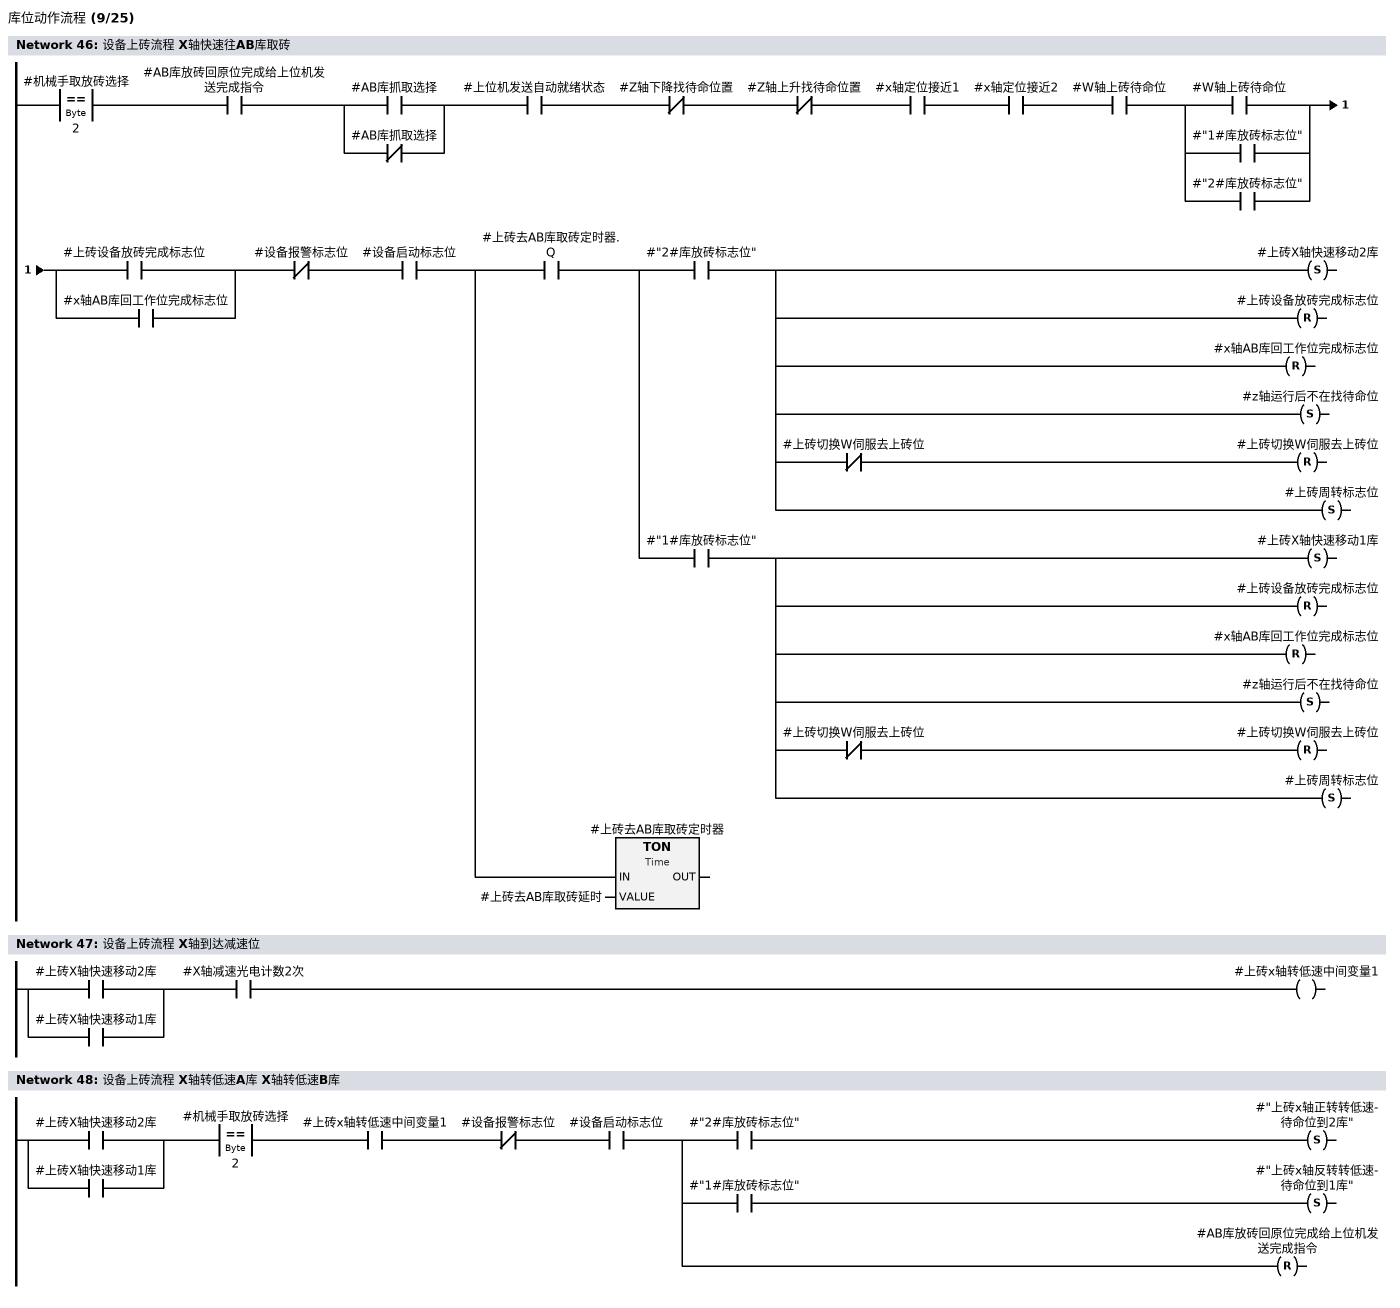
   #_w1 := (#机械手取放砖选择 = 2) AND #AB库放砖回原位完成给上位机发送完成指令 AND (#AB库抓取选择 OR NOT #AB库抓取选择) AND #上位机发送自动就绪状态 AND NOT #Z轴下降找待命位置 AND NOT #Z轴上升找待命位置 AND #x轴定位接近1 AND #x轴定位接近2 AND #W轴上砖待命位 AND (#W轴上砖待命位 OR #"1#库放砖标志位" OR #"2#库放砖标志位") AND (#上砖设备放砖完成标志位 OR #x轴AB库回工作位完成标志位) AND NOT #设备报警标志位 AND #设备启动标志位;
   #_w2 := #_w1 AND #上砖去AB库取砖定时器.Q;
   #_w3 := #_w2 AND #"2#库放砖标志位";
   IF #_w3 THEN
       #上砖X轴快速移动2库 := TRUE;
       #上砖设备放砖完成标志位 := FALSE;
       #x轴AB库回工作位完成标志位 := FALSE;
       #z轴运行后不在找待命位 := TRUE;
   END_IF;
   IF #_w3 AND NOT #上砖切换W伺服去上砖位 THEN #上砖切换W伺服去上砖位 := FALSE; END_IF;
   IF #_w3 THEN #上砖周转标志位 := TRUE; END_IF;
   #_w4 := #_w2 AND #"1#库放砖标志位";
   IF #_w4 THEN
       #上砖X轴快速移动1库 := TRUE;
       #上砖设备放砖完成标志位 := FALSE;
       #x轴AB库回工作位完成标志位 := FALSE;
       #z轴运行后不在找待命位 := TRUE;
   END_IF;
   IF #_w4 AND NOT #上砖切换W伺服去上砖位 THEN #上砖切换W伺服去上砖位 := FALSE; END_IF;
   IF #_w4 THEN #上砖周转标志位 := TRUE; END_IF;
   #上砖去AB库取砖定时器.TON(IN := #_w1, PT := #上砖去AB库取砖延时);   // TON coil
END_REGION

REGION Network 47: 设备上砖流程 X轴到达减速位
   RUNG wire#powerrail
      Contact( #上砖X轴快速移动2库 )
      wire#w1
      Contact( #X轴减速光电计数2次 )
      Coil( #上砖x轴转低速中间变量1 )
   END_RUNG
   RUNG wire#powerrail
      Contact( #上砖X轴快速移动1库 )
   END_RUNG wire#w1
   // the same network as SCL:
   #上砖x轴转低速中间变量1 := (#上砖X轴快速移动2库 OR #上砖X轴快速移动1库) AND #X轴减速光电计数2次;
END_REGION

REGION Network 48: 设备上砖流程 X轴转低速A库 X轴转低速B库
   RUNG wire#powerrail
      Contact( #上砖X轴快速移动2库 )
      wire#w1
      { S7_Templates := "SrcType := Byte" } EQ_Contact(in1 := #机械手取放砖选择, in2 := 2)
      Contact( #上砖x轴转低速中间变量1 )
      I_Contact( #设备报警标志位 )
      Contact( #设备启动标志位 )
      wire#w2
      Contact( #"2#库放砖标志位" )
      S_Coil( #"上砖x轴正转转低速-待命位到2库" )
   END_RUNG
   RUNG wire#powerrail
      Contact( #上砖X轴快速移动1库 )
   END_RUNG wire#w1
   RUNG wire#w2
      Contact( #"1#库放砖标志位" )
      S_Coil( #"上砖x轴反转转低速-待命位到1库" )
   END_RUNG
   RUNG wire#w2
      R_Coil( #AB库放砖回原位完成给上位机发送完成指令 )
   END_RUNG
   // the same network as SCL:
   #_w1 := (#上砖X轴快速移动2库 OR #上砖X轴快速移动1库) AND (#机械手取放砖选择 = 2) AND #上砖x轴转低速中间变量1 AND NOT #设备报警标志位 AND #设备启动标志位;
   IF #_w1 AND #"2#库放砖标志位" THEN #"上砖x轴正转转低速-待命位到2库" := TRUE; END_IF;
   IF #_w1 AND #"1#库放砖标志位" THEN #"上砖x轴反转转低速-待命位到1库" := TRUE; END_IF;
   IF #_w1 THEN #AB库放砖回原位完成给上位机发送完成指令 := FALSE; END_IF;
END_REGION

REGION Network 49: 设备上砖流程 X轴到达A库下方 X轴到达B库下方
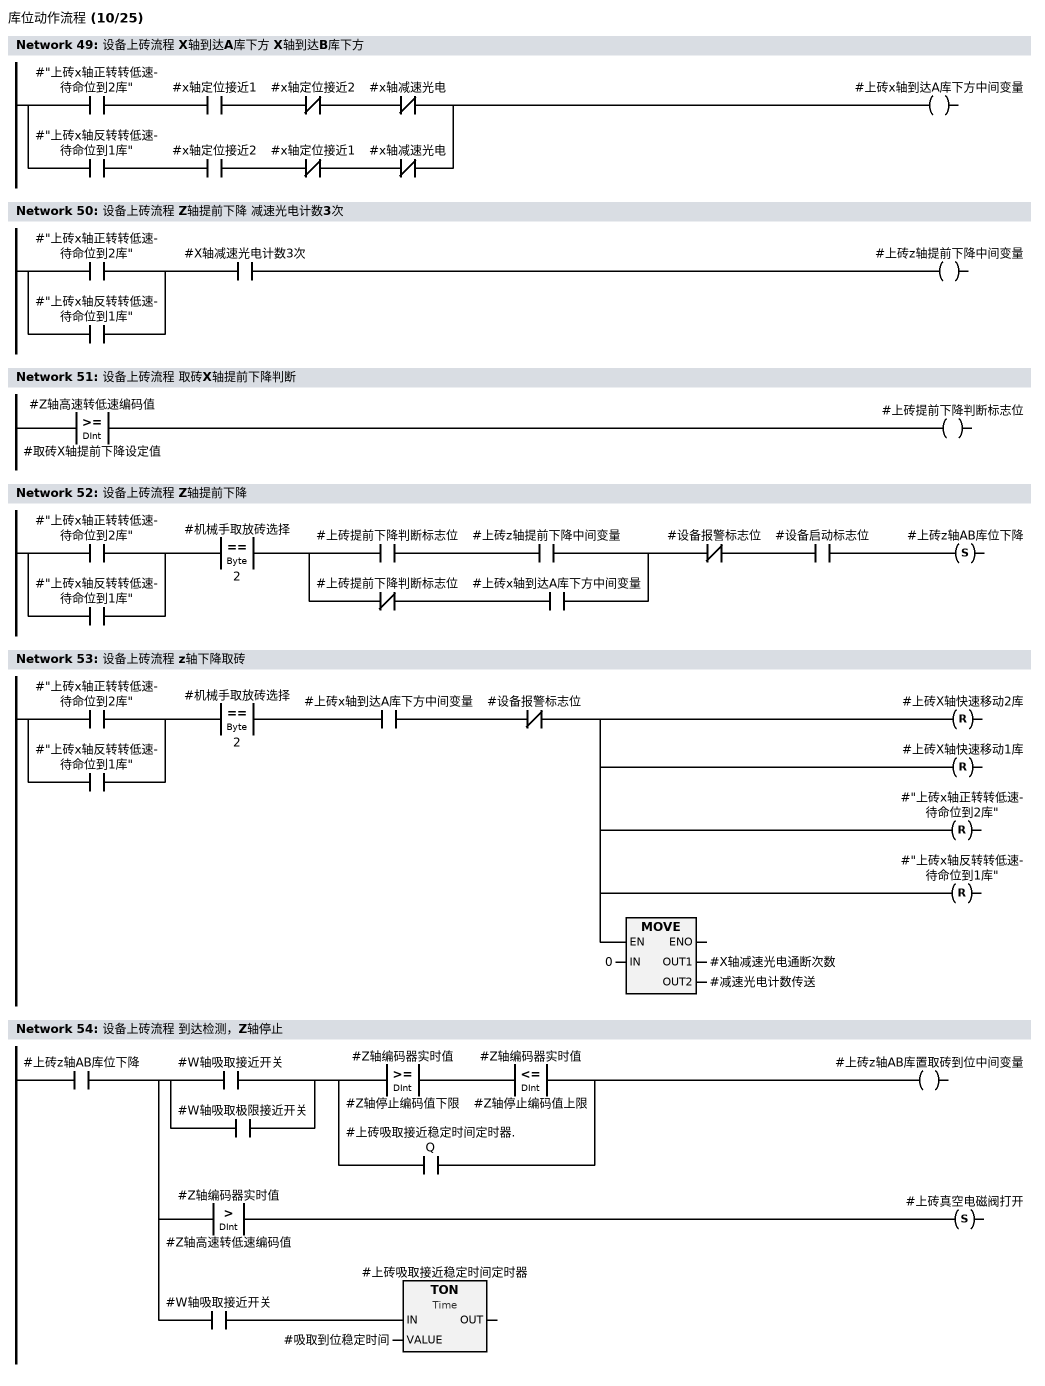
   RUNG wire#powerrail
      Contact( #"上砖x轴正转转低速-待命位到2库" )
      Contact( #x轴定位接近1 )
      I_Contact( #x轴定位接近2 )
      I_Contact( #x轴减速光电 )
      wire#w1
      Coil( #上砖x轴到达A库下方中间变量 )
   END_RUNG
   RUNG wire#powerrail
      Contact( #"上砖x轴反转转低速-待命位到1库" )
      Contact( #x轴定位接近2 )
      I_Contact( #x轴定位接近1 )
      I_Contact( #x轴减速光电 )
   END_RUNG wire#w1
   // the same network as SCL:
   #上砖x轴到达A库下方中间变量 := (#"上砖x轴正转转低速-待命位到2库" AND #x轴定位接近1 AND NOT #x轴定位接近2 AND NOT #x轴减速光电) OR (#"上砖x轴反转转低速-待命位到1库" AND #x轴定位接近2 AND NOT #x轴定位接近1 AND NOT #x轴减速光电);
END_REGION

REGION Network 50: 设备上砖流程 Z轴提前下降 减速光电计数3次
   RUNG wire#powerrail
      Contact( #"上砖x轴正转转低速-待命位到2库" )
      wire#w1
      Contact( #X轴减速光电计数3次 )
      Coil( #上砖z轴提前下降中间变量 )
   END_RUNG
   RUNG wire#powerrail
      Contact( #"上砖x轴反转转低速-待命位到1库" )
   END_RUNG wire#w1
   // the same network as SCL:
   #上砖z轴提前下降中间变量 := (#"上砖x轴正转转低速-待命位到2库" OR #"上砖x轴反转转低速-待命位到1库") AND #X轴减速光电计数3次;
END_REGION

